REGION Network 35 (SCL): OPENVALVE
   IF "MODE SELECTION DB"."MODE BUFF" <> 0 AND "TRANSFER DB".BUFF."PREMIXING TO MFG WITH INLINE FILTER PRES" = 2
       AND NOT "TRANSFER DB".PAUSE."PREMIXING TO MFG WITH INLINE FILTER PRES" 
       AND "CONTINUE DB"."PREMIXING PROCESS ERROR" = 0 AND "LEVEL BUFF"."PREMIXING_LOAD CELL" = 0 THEN
       "TRANSFER DB".BIT."PREMIXING TO MFG WITH INLINE FILTER PRES"."PFBV-17 TANK OUTLET VALVE" := TRUE;
       "TRANSFER DB".BIT."PREMIXING TO MFG WITH INLINE FILTER PRES"."PBV-93 TANK OUTLET TO INLINE HOMOGENIZER LINE" := TRUE;
       "TRANSFER DB".BIT."PREMIXING TO MFG WITH INLINE FILTER PRES"."PBV-95 TANK OUTLET TO FILTER PRESS LINE" := TRUE;
       "TRANSFER DB".BIT."PREMIXING TO MFG WITH INLINE FILTER PRES"."FILTER PRESS MOTOR 2 RUN" := TRUE;
       "TRANSFER DB".BIT."PREMIXING TO MFG WITH INLINE FILTER PRES"."PBV-100 FILTER PRESS INLET" := TRUE;
       "TRANSFER DB".BIT."PREMIXING TO MFG WITH INLINE FILTER PRES"."PBV-97 FILTER PRESS OUTLET" := TRUE;
       "TRANSFER DB".BIT."PREMIXING TO MFG WITH INLINE FILTER PRES"."PBV-98 INLINE HOMOGENIZER TO FILTER PRESS OUTLET LINE" := TRUE;
       "TRANSFER DB".BIT."PREMIXING TO MFG WITH INLINE FILTER PRES"."PBV-91 PREMIX TO MFG TRANSFER LINE" := TRUE;
       "TRANSFER DB".BIT."PREMIXING TO MFG WITH INLINE FILTER PRES"."PBV-102 PREMIX TO MFG TRANSFER (TOP DISH)" := TRUE;

   ELSE
       "TRANSFER DB".BIT."PREMIXING TO MFG WITH INLINE FILTER PRES"."PFBV-17 TANK OUTLET VALVE" := FALSE;
       "TRANSFER DB".BIT."PREMIXING TO MFG WITH INLINE FILTER PRES"."PBV-93 TANK OUTLET TO INLINE HOMOGENIZER LINE" := FALSE;
       "TRANSFER DB".BIT."PREMIXING TO MFG WITH INLINE FILTER PRES"."PBV-95 TANK OUTLET TO FILTER PRESS LINE" := FALSE;
       "TRANSFER DB".BIT."PREMIXING TO MFG WITH INLINE FILTER PRES"."FILTER PRESS MOTOR 2 RUN" := FALSE;
       "TRANSFER DB".BIT."PREMIXING TO MFG WITH INLINE FILTER PRES"."PBV-100 FILTER PRESS INLET" := FALSE;
       "TRANSFER DB".BIT."PREMIXING TO MFG WITH INLINE FILTER PRES"."PBV-97 FILTER PRESS OUTLET" := FALSE;
       "TRANSFER DB".BIT."PREMIXING TO MFG WITH INLINE FILTER PRES"."PBV-98 INLINE HOMOGENIZER TO FILTER PRESS OUTLET LINE" := FALSE;
       "TRANSFER DB".BIT."PREMIXING TO MFG WITH INLINE FILTER PRES"."PBV-91 PREMIX TO MFG TRANSFER LINE" := FALSE;
       "TRANSFER DB".BIT."PREMIXING TO MFG WITH INLINE FILTER PRES"."PBV-102 PREMIX TO MFG TRANSFER (TOP DISH)" := FALSE;
       ;
   END_IF;
END_REGION

REGION Network 36: LOAD CELL_CUTOFF
   RUNG wire#powerrail
      { S7_Templates := "SrcType := Int" } NE_Contact(in1 := "MODE SELECTION DB"."MODE BUFF", in2 := 0)
      { S7_Templates := "SrcType := Int" } EQ_Contact(in1 := "TRANSFER DB".BUFF."PREMIXING TO MFG WITH INLINE FILTER PRES", in2 := 2)
      I_Contact( "TRANSFER DB".PAUSE."PREMIXING TO MFG WITH INLINE FILTER PRES" )
      { S7_Templates := "SrcType := Int" } NE_Contact(in1 := "CONTINUE DB"."PREMIXING PROCESS ERROR", in2 := 1)
      { S7_Templates := "SrcType := Int" } EQ_Contact(in1 := "LEVEL BUFF"."PREMIXING_LOAD CELL", in2 := 1)
      Move(in := 3, out1 => "TRANSFER DB".BUFF."PREMIXING TO MFG WITH INLINE FILTER PRES")
   END_RUNG
   // the same network as SCL:
   IF ("MODE SELECTION DB"."MODE BUFF" <> 0) AND ("TRANSFER DB".BUFF."PREMIXING TO MFG WITH INLINE FILTER PRES" = 2) AND NOT "TRANSFER DB".PAUSE."PREMIXING TO MFG WITH INLINE FILTER PRES" AND ("CONTINUE DB"."PREMIXING PROCESS ERROR" <> 1) AND ("LEVEL BUFF"."PREMIXING_LOAD CELL" = 1) THEN
       "TRANSFER DB".BUFF."PREMIXING TO MFG WITH INLINE FILTER PRES" := 3;
   END_IF;
END_REGION

REGION Network 37: PROCESS OVER & STOP
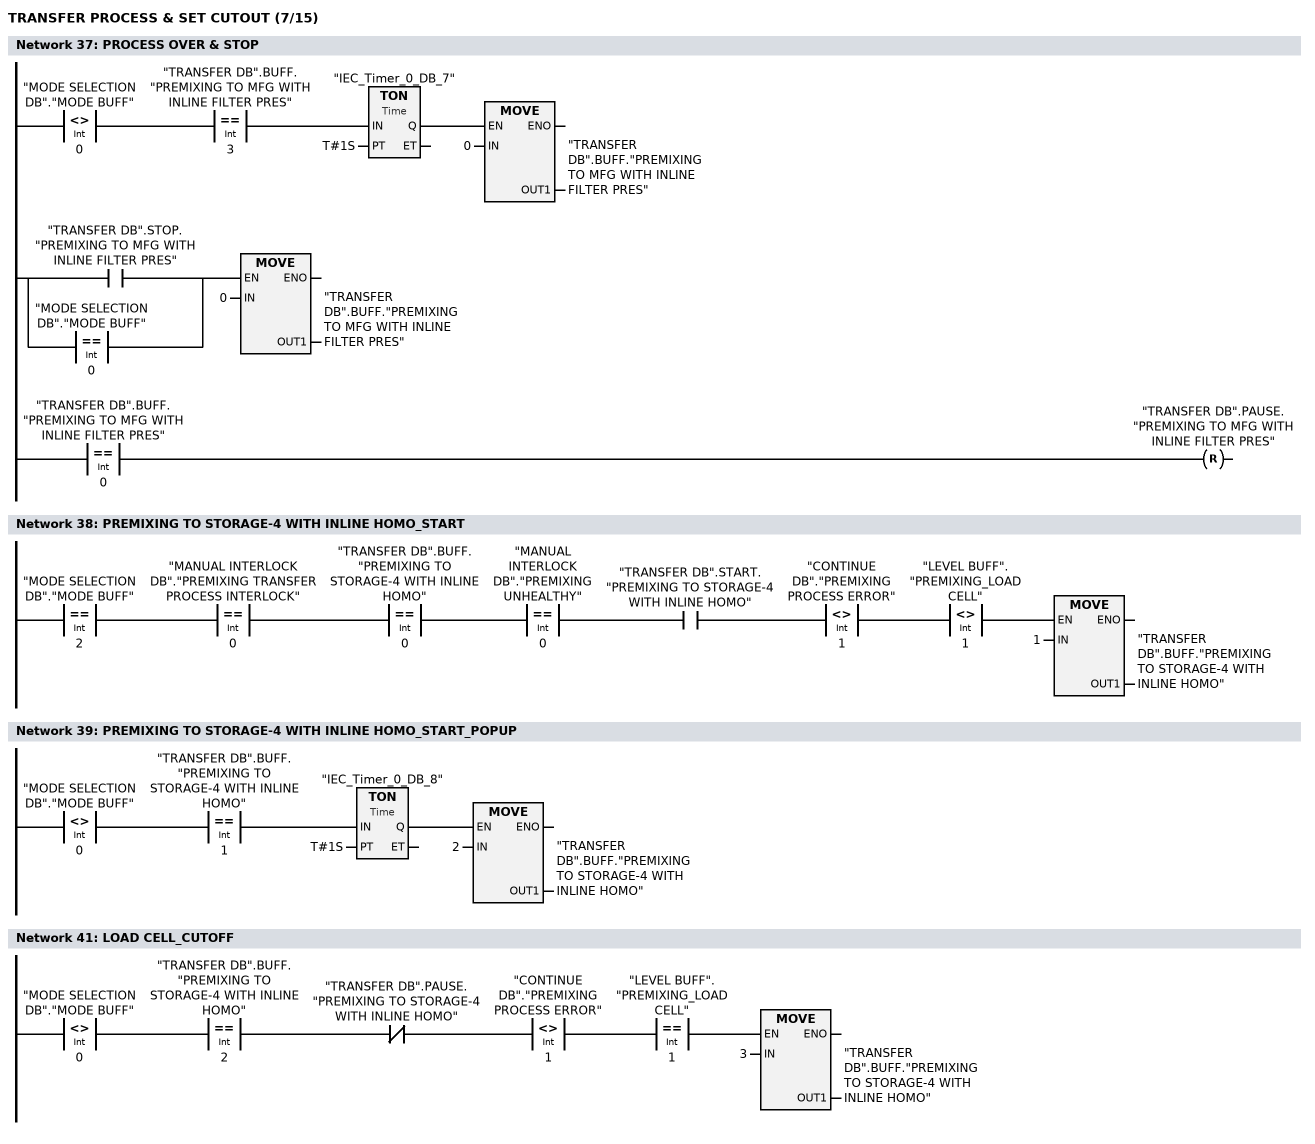
   RUNG wire#powerrail
      { S7_Templates := "SrcType := Int" } NE_Contact(in1 := "MODE SELECTION DB"."MODE BUFF", in2 := 0)
      { S7_Templates := "SrcType := Int" } EQ_Contact(in1 := "TRANSFER DB".BUFF."PREMIXING TO MFG WITH INLINE FILTER PRES", in2 := 3)
      { S7_Templates := "time_type := Time" } "IEC_Timer_0_DB_7".TON(pt := T#1S, et =>)
      Move(in := 0, out1 => "TRANSFER DB".BUFF."PREMIXING TO MFG WITH INLINE FILTER PRES")
   END_RUNG
   RUNG wire#powerrail
      Contact( "TRANSFER DB".STOP."PREMIXING TO MFG WITH INLINE FILTER PRES" )
      wire#w1
      Move(in := 0, out1 => "TRANSFER DB".BUFF."PREMIXING TO MFG WITH INLINE FILTER PRES")
   END_RUNG
   RUNG wire#powerrail
      { S7_Templates := "SrcType := Int" } EQ_Contact(in1 := "MODE SELECTION DB"."MODE BUFF", in2 := 0)
   END_RUNG wire#w1
   RUNG wire#powerrail
      { S7_Templates := "SrcType := Int" } EQ_Contact(in1 := "TRANSFER DB".BUFF."PREMIXING TO MFG WITH INLINE FILTER PRES", in2 := 0)
      R_Coil( "TRANSFER DB".PAUSE."PREMIXING TO MFG WITH INLINE FILTER PRES" )
   END_RUNG
   // the same network as SCL:
   "IEC_Timer_0_DB_7".TON(IN := ("MODE SELECTION DB"."MODE BUFF" <> 0) AND ("TRANSFER DB".BUFF."PREMIXING TO MFG WITH INLINE FILTER PRES" = 3),
                          PT := T#1S);
   IF "IEC_Timer_0_DB_7".Q THEN "TRANSFER DB".BUFF."PREMIXING TO MFG WITH INLINE FILTER PRES" := 0; END_IF;
   IF "TRANSFER DB".STOP."PREMIXING TO MFG WITH INLINE FILTER PRES" OR ("MODE SELECTION DB"."MODE BUFF" = 0) THEN
       "TRANSFER DB".BUFF."PREMIXING TO MFG WITH INLINE FILTER PRES" := 0;
   END_IF;
   IF "TRANSFER DB".BUFF."PREMIXING TO MFG WITH INLINE FILTER PRES" = 0 THEN
       "TRANSFER DB".PAUSE."PREMIXING TO MFG WITH INLINE FILTER PRES" := FALSE;
   END_IF;
END_REGION

REGION Network 38: PREMIXING TO STORAGE-4 WITH INLINE HOMO_START
   RUNG wire#powerrail
      { S7_Templates := "SrcType := Int" } EQ_Contact(in1 := "MODE SELECTION DB"."MODE BUFF", in2 := 2)
      { S7_Templates := "SrcType := Int" } EQ_Contact(in1 := "MANUAL INTERLOCK DB"."PREMIXING TRANSFER PROCESS INTERLOCK", in2 := 0)
      { S7_Templates := "SrcType := Int" } EQ_Contact(in1 := "TRANSFER DB".BUFF."PREMIXING TO STORAGE-4 WITH INLINE HOMO", in2 := 0)
      { S7_Templates := "SrcType := Int" } EQ_Contact(in1 := "MANUAL INTERLOCK DB"."PREMIXING UNHEALTHY", in2 := 0)
      Contact( "TRANSFER DB".START."PREMIXING TO STORAGE-4 WITH INLINE HOMO" )
      { S7_Templates := "SrcType := Int" } NE_Contact(in1 := "CONTINUE DB"."PREMIXING PROCESS ERROR", in2 := 1)
      { S7_Templates := "SrcType := Int" } NE_Contact(in1 := "LEVEL BUFF"."PREMIXING_LOAD CELL", in2 := 1)
      Move(in := 1, out1 => "TRANSFER DB".BUFF."PREMIXING TO STORAGE-4 WITH INLINE HOMO")
   END_RUNG
   // the same network as SCL:
   IF ("MODE SELECTION DB"."MODE BUFF" = 2) AND ("MANUAL INTERLOCK DB"."PREMIXING TRANSFER PROCESS INTERLOCK" = 0) AND ("TRANSFER DB".BUFF."PREMIXING TO STORAGE-4 WITH INLINE HOMO" = 0) AND ("MANUAL INTERLOCK DB"."PREMIXING UNHEALTHY" = 0) AND "TRANSFER DB".START."PREMIXING TO STORAGE-4 WITH INLINE HOMO" AND ("CONTINUE DB"."PREMIXING PROCESS ERROR" <> 1) AND ("LEVEL BUFF"."PREMIXING_LOAD CELL" <> 1) THEN
       "TRANSFER DB".BUFF."PREMIXING TO STORAGE-4 WITH INLINE HOMO" := 1;
   END_IF;
END_REGION

REGION Network 39: PREMIXING TO STORAGE-4 WITH INLINE HOMO_START_POPUP
   RUNG wire#powerrail
      { S7_Templates := "SrcType := Int" } NE_Contact(in1 := "MODE SELECTION DB"."MODE BUFF", in2 := 0)
      { S7_Templates := "SrcType := Int" } EQ_Contact(in1 := "TRANSFER DB".BUFF."PREMIXING TO STORAGE-4 WITH INLINE HOMO", in2 := 1)
      { S7_Templates := "time_type := Time" } "IEC_Timer_0_DB_8".TON(pt := T#1S, et =>)
      Move(in := 2, out1 => "TRANSFER DB".BUFF."PREMIXING TO STORAGE-4 WITH INLINE HOMO")
   END_RUNG
   // the same network as SCL:
   "IEC_Timer_0_DB_8".TON(IN := ("MODE SELECTION DB"."MODE BUFF" <> 0) AND ("TRANSFER DB".BUFF."PREMIXING TO STORAGE-4 WITH INLINE HOMO" = 1),
                          PT := T#1S);
   IF "IEC_Timer_0_DB_8".Q THEN "TRANSFER DB".BUFF."PREMIXING TO STORAGE-4 WITH INLINE HOMO" := 2; END_IF;
END_REGION

REGION Network 40 (SCL): OPENVALVE
   IF "MODE SELECTION DB"."MODE BUFF" <> 0 AND "TRANSFER DB".BUFF."PREMIXING TO STORAGE-4 WITH INLINE HOMO" = 2
       AND NOT "TRANSFER DB".PAUSE."PREMIXING TO STORAGE-4 WITH INLINE HOMO"
       AND "CONTINUE DB"."PREMIXING PROCESS ERROR" = 0 AND "LEVEL BUFF"."PREMIXING_LOAD CELL" = 0 THEN
       "TRANSFER DB".BIT."PREMIXING TO STORAGE-4 WITH INLINE HOMO"."PFBV-17 TANK OUTLET VALVE" := TRUE;
       "TRANSFER DB".BIT."PREMIXING TO STORAGE-4 WITH INLINE HOMO"."PBV-93 TANK OUTLET TO INLINE HOMOGENIZER LINE" := TRUE;
       "TRANSFER DB".BIT."PREMIXING TO STORAGE-4 WITH INLINE HOMO"."PBV-94 INLINE HOMOGENIZER INLET LINE" := TRUE;
       "TRANSFER DB".BIT."PREMIXING TO STORAGE-4 WITH INLINE HOMO"."INLINE 2 HOMOGENIZER MOTOR 2 RUN" := TRUE;
       "TRANSFER DB".BIT."PREMIXING TO STORAGE-4 WITH INLINE HOMO"."PBV-96 INLINE HOMOGENIZER RECIRCULATION LINE" := TRUE;
       "TRANSFER DB".BIT."PREMIXING TO STORAGE-4 WITH INLINE HOMO"."PBV-92 PREMIX TO STORAGE – 4 TRANSFER LINE" := TRUE;

   ELSE
       "TRANSFER DB".BIT."PREMIXING TO STORAGE-4 WITH INLINE HOMO"."PFBV-17 TANK OUTLET VALVE" := FALSE;
       "TRANSFER DB".BIT."PREMIXING TO STORAGE-4 WITH INLINE HOMO"."PBV-93 TANK OUTLET TO INLINE HOMOGENIZER LINE" := FALSE;
       "TRANSFER DB".BIT."PREMIXING TO STORAGE-4 WITH INLINE HOMO"."PBV-94 INLINE HOMOGENIZER INLET LINE" := FALSE;
       "TRANSFER DB".BIT."PREMIXING TO STORAGE-4 WITH INLINE HOMO"."INLINE 2 HOMOGENIZER MOTOR 2 RUN" := FALSE;
       "TRANSFER DB".BIT."PREMIXING TO STORAGE-4 WITH INLINE HOMO"."PBV-96 INLINE HOMOGENIZER RECIRCULATION LINE" := FALSE;
       "TRANSFER DB".BIT."PREMIXING TO STORAGE-4 WITH INLINE HOMO"."PBV-92 PREMIX TO STORAGE – 4 TRANSFER LINE" := FALSE;
       ;
   END_IF;
END_REGION

REGION Network 41: LOAD CELL_CUTOFF
   RUNG wire#powerrail
      { S7_Templates := "SrcType := Int" } NE_Contact(in1 := "MODE SELECTION DB"."MODE BUFF", in2 := 0)
      { S7_Templates := "SrcType := Int" } EQ_Contact(in1 := "TRANSFER DB".BUFF."PREMIXING TO STORAGE-4 WITH INLINE HOMO", in2 := 2)
      I_Contact( "TRANSFER DB".PAUSE."PREMIXING TO STORAGE-4 WITH INLINE HOMO" )
      { S7_Templates := "SrcType := Int" } NE_Contact(in1 := "CONTINUE DB"."PREMIXING PROCESS ERROR", in2 := 1)
      { S7_Templates := "SrcType := Int" } EQ_Contact(in1 := "LEVEL BUFF"."PREMIXING_LOAD CELL", in2 := 1)
      Move(in := 3, out1 => "TRANSFER DB".BUFF."PREMIXING TO STORAGE-4 WITH INLINE HOMO")
   END_RUNG
   // the same network as SCL:
   IF ("MODE SELECTION DB"."MODE BUFF" <> 0) AND ("TRANSFER DB".BUFF."PREMIXING TO STORAGE-4 WITH INLINE HOMO" = 2) AND NOT "TRANSFER DB".PAUSE."PREMIXING TO STORAGE-4 WITH INLINE HOMO" AND ("CONTINUE DB"."PREMIXING PROCESS ERROR" <> 1) AND ("LEVEL BUFF"."PREMIXING_LOAD CELL" = 1) THEN
       "TRANSFER DB".BUFF."PREMIXING TO STORAGE-4 WITH INLINE HOMO" := 3;
   END_IF;
END_REGION

REGION Network 42: PROCESS OVER & STOP
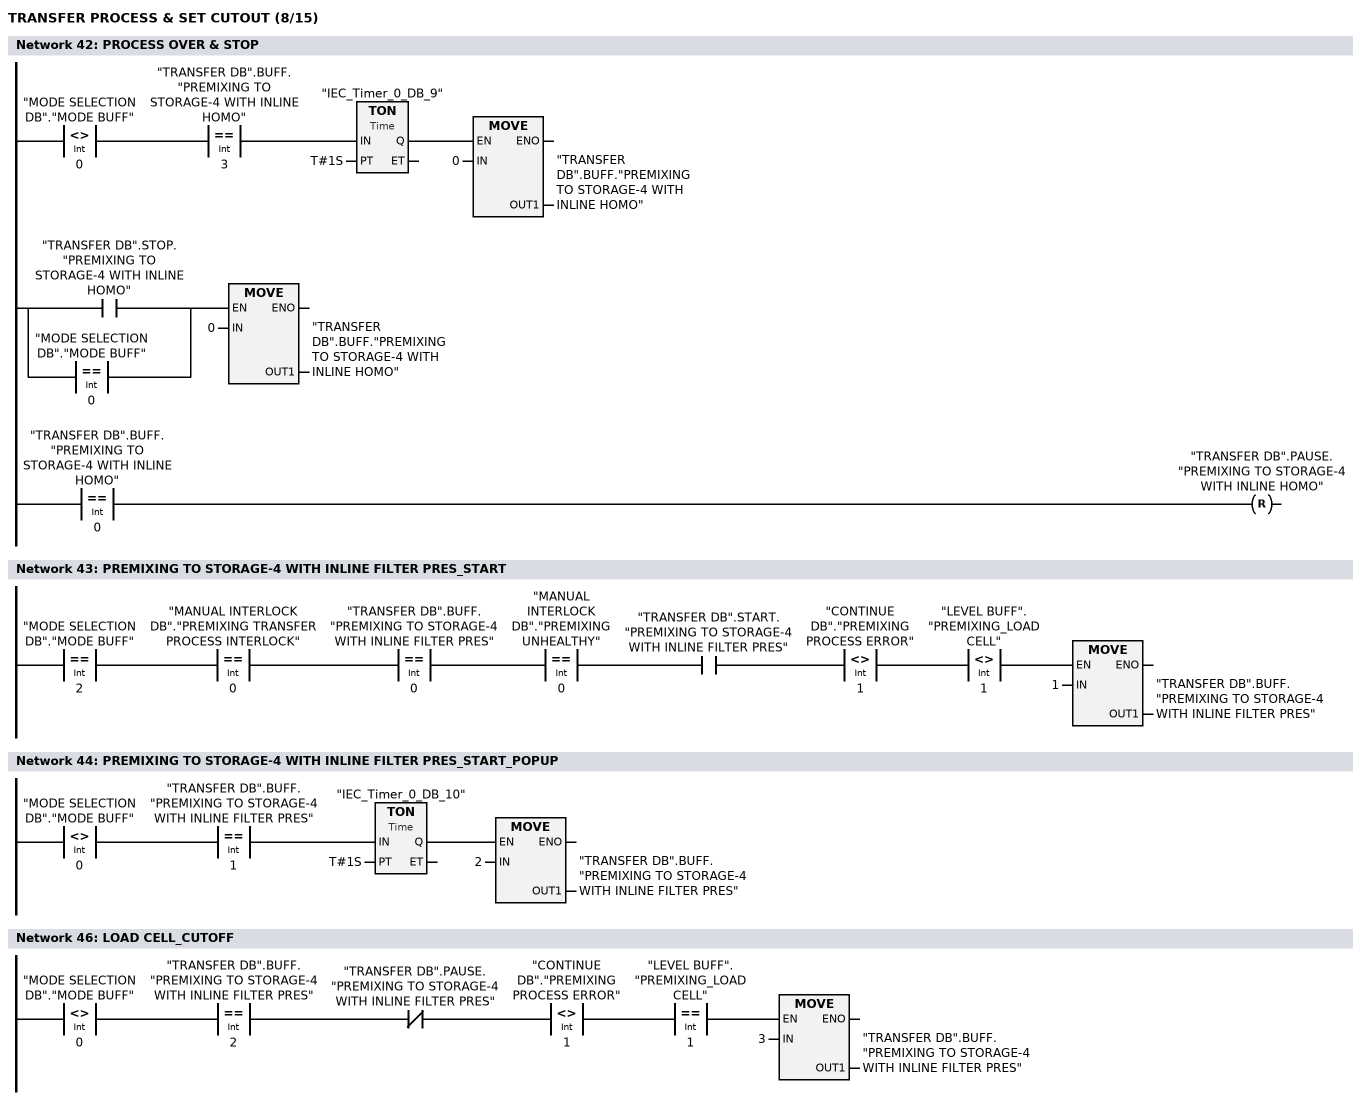
   RUNG wire#powerrail
      { S7_Templates := "SrcType := Int" } NE_Contact(in1 := "MODE SELECTION DB"."MODE BUFF", in2 := 0)
      { S7_Templates := "SrcType := Int" } EQ_Contact(in1 := "TRANSFER DB".BUFF."PREMIXING TO STORAGE-4 WITH INLINE HOMO", in2 := 3)
      { S7_Templates := "time_type := Time" } "IEC_Timer_0_DB_9".TON(pt := T#1S, et =>)
      Move(in := 0, out1 => "TRANSFER DB".BUFF."PREMIXING TO STORAGE-4 WITH INLINE HOMO")
   END_RUNG
   RUNG wire#powerrail
      Contact( "TRANSFER DB".STOP."PREMIXING TO STORAGE-4 WITH INLINE HOMO" )
      wire#w1
      Move(in := 0, out1 => "TRANSFER DB".BUFF."PREMIXING TO STORAGE-4 WITH INLINE HOMO")
   END_RUNG
   RUNG wire#powerrail
      { S7_Templates := "SrcType := Int" } EQ_Contact(in1 := "MODE SELECTION DB"."MODE BUFF", in2 := 0)
   END_RUNG wire#w1
   RUNG wire#powerrail
      { S7_Templates := "SrcType := Int" } EQ_Contact(in1 := "TRANSFER DB".BUFF."PREMIXING TO STORAGE-4 WITH INLINE HOMO", in2 := 0)
      R_Coil( "TRANSFER DB".PAUSE."PREMIXING TO STORAGE-4 WITH INLINE HOMO" )
   END_RUNG
   // the same network as SCL:
   "IEC_Timer_0_DB_9".TON(IN := ("MODE SELECTION DB"."MODE BUFF" <> 0) AND ("TRANSFER DB".BUFF."PREMIXING TO STORAGE-4 WITH INLINE HOMO" = 3),
                          PT := T#1S);
   IF "IEC_Timer_0_DB_9".Q THEN "TRANSFER DB".BUFF."PREMIXING TO STORAGE-4 WITH INLINE HOMO" := 0; END_IF;
   IF "TRANSFER DB".STOP."PREMIXING TO STORAGE-4 WITH INLINE HOMO" OR ("MODE SELECTION DB"."MODE BUFF" = 0) THEN
       "TRANSFER DB".BUFF."PREMIXING TO STORAGE-4 WITH INLINE HOMO" := 0;
   END_IF;
   IF "TRANSFER DB".BUFF."PREMIXING TO STORAGE-4 WITH INLINE HOMO" = 0 THEN
       "TRANSFER DB".PAUSE."PREMIXING TO STORAGE-4 WITH INLINE HOMO" := FALSE;
   END_IF;
END_REGION

REGION Network 43: PREMIXING TO STORAGE-4 WITH INLINE FILTER PRES_START
   RUNG wire#powerrail
      { S7_Templates := "SrcType := Int" } EQ_Contact(in1 := "MODE SELECTION DB"."MODE BUFF", in2 := 2)
      { S7_Templates := "SrcType := Int" } EQ_Contact(in1 := "MANUAL INTERLOCK DB"."PREMIXING TRANSFER PROCESS INTERLOCK", in2 := 0)
      { S7_Templates := "SrcType := Int" } EQ_Contact(in1 := "TRANSFER DB".BUFF."PREMIXING TO STORAGE-4 WITH INLINE FILTER PRES", in2 := 0)
      { S7_Templates := "SrcType := Int" } EQ_Contact(in1 := "MANUAL INTERLOCK DB"."PREMIXING UNHEALTHY", in2 := 0)
      Contact( "TRANSFER DB".START."PREMIXING TO STORAGE-4 WITH INLINE FILTER PRES" )
      { S7_Templates := "SrcType := Int" } NE_Contact(in1 := "CONTINUE DB"."PREMIXING PROCESS ERROR", in2 := 1)
      { S7_Templates := "SrcType := Int" } NE_Contact(in1 := "LEVEL BUFF"."PREMIXING_LOAD CELL", in2 := 1)
      Move(in := 1, out1 => "TRANSFER DB".BUFF."PREMIXING TO STORAGE-4 WITH INLINE FILTER PRES")
   END_RUNG
   // the same network as SCL:
   IF ("MODE SELECTION DB"."MODE BUFF" = 2) AND ("MANUAL INTERLOCK DB"."PREMIXING TRANSFER PROCESS INTERLOCK" = 0) AND ("TRANSFER DB".BUFF."PREMIXING TO STORAGE-4 WITH INLINE FILTER PRES" = 0) AND ("MANUAL INTERLOCK DB"."PREMIXING UNHEALTHY" = 0) AND "TRANSFER DB".START."PREMIXING TO STORAGE-4 WITH INLINE FILTER PRES" AND ("CONTINUE DB"."PREMIXING PROCESS ERROR" <> 1) AND ("LEVEL BUFF"."PREMIXING_LOAD CELL" <> 1) THEN
       "TRANSFER DB".BUFF."PREMIXING TO STORAGE-4 WITH INLINE FILTER PRES" := 1;
   END_IF;
END_REGION

REGION Network 44: PREMIXING TO STORAGE-4 WITH INLINE FILTER PRES_START_POPUP
   RUNG wire#powerrail
      { S7_Templates := "SrcType := Int" } NE_Contact(in1 := "MODE SELECTION DB"."MODE BUFF", in2 := 0)
      { S7_Templates := "SrcType := Int" } EQ_Contact(in1 := "TRANSFER DB".BUFF."PREMIXING TO STORAGE-4 WITH INLINE FILTER PRES", in2 := 1)
      { S7_Templates := "time_type := Time" } "IEC_Timer_0_DB_10".TON(pt := T#1S, et =>)
      Move(in := 2, out1 => "TRANSFER DB".BUFF."PREMIXING TO STORAGE-4 WITH INLINE FILTER PRES")
   END_RUNG
   // the same network as SCL:
   "IEC_Timer_0_DB_10".TON(IN := ("MODE SELECTION DB"."MODE BUFF" <> 0) AND ("TRANSFER DB".BUFF."PREMIXING TO STORAGE-4 WITH INLINE FILTER PRES" = 1),
                           PT := T#1S);
   IF "IEC_Timer_0_DB_10".Q THEN
       "TRANSFER DB".BUFF."PREMIXING TO STORAGE-4 WITH INLINE FILTER PRES" := 2;
   END_IF;
END_REGION

REGION Network 45 (SCL): OPENVALVE
   IF "MODE SELECTION DB"."MODE BUFF" <> 0 AND "TRANSFER DB".BUFF."PREMIXING TO STORAGE-4 WITH INLINE FILTER PRES" = 2
       AND NOT "TRANSFER DB".PAUSE."PREMIXING TO STORAGE-4 WITH INLINE FILTER PRES" 
       AND "CONTINUE DB"."PREMIXING PROCESS ERROR" = 0 AND "LEVEL BUFF"."PREMIXING_LOAD CELL" = 0 THEN
       "TRANSFER DB".BIT."PREMIXING TO STORAGE-4 WITH INLINE FILTER PRES"."PFBV-17 TANK OUTLET VALVE" := TRUE;
       "TRANSFER DB".BIT."PREMIXING TO STORAGE-4 WITH INLINE FILTER PRES"."PBV-93 TANK OUTLET TO INLINE HOMOGENIZER LINE" := TRUE;
       "TRANSFER DB".BIT."PREMIXING TO STORAGE-4 WITH INLINE FILTER PRES"."PBV-95 TANK OUTLET TO FILTER PRESS LINE" := TRUE;
       "TRANSFER DB".BIT."PREMIXING TO STORAGE-4 WITH INLINE FILTER PRES"."FILTER PRESS MOTOR 2 RUN" := TRUE;
       "TRANSFER DB".BIT."PREMIXING TO STORAGE-4 WITH INLINE FILTER PRES"."PBV-100 FILTER PRESS INLET" := TRUE;
       "TRANSFER DB".BIT."PREMIXING TO STORAGE-4 WITH INLINE FILTER PRES"."PBV-97 FILTER PRESS OUTLET" := TRUE;
       "TRANSFER DB".BIT."PREMIXING TO STORAGE-4 WITH INLINE FILTER PRES"."PBV-98 INLINE HOMOGENIZER TO FILTER PRESS OUTLET LINE" := TRUE;
       "TRANSFER DB".BIT."PREMIXING TO STORAGE-4 WITH INLINE FILTER PRES"."PBV-92 PREMIX TO STORAGE – 4 TRANSFER LINE" := TRUE;

   ELSE
       "TRANSFER DB".BIT."PREMIXING TO STORAGE-4 WITH INLINE FILTER PRES"."PFBV-17 TANK OUTLET VALVE" := FALSE;
       "TRANSFER DB".BIT."PREMIXING TO STORAGE-4 WITH INLINE FILTER PRES"."PBV-93 TANK OUTLET TO INLINE HOMOGENIZER LINE" := FALSE;
       "TRANSFER DB".BIT."PREMIXING TO STORAGE-4 WITH INLINE FILTER PRES"."PBV-95 TANK OUTLET TO FILTER PRESS LINE" := FALSE;
       "TRANSFER DB".BIT."PREMIXING TO STORAGE-4 WITH INLINE FILTER PRES"."FILTER PRESS MOTOR 2 RUN" := FALSE;
       "TRANSFER DB".BIT."PREMIXING TO STORAGE-4 WITH INLINE FILTER PRES"."PBV-100 FILTER PRESS INLET" := FALSE;
       "TRANSFER DB".BIT."PREMIXING TO STORAGE-4 WITH INLINE FILTER PRES"."PBV-97 FILTER PRESS OUTLET" := FALSE;
       "TRANSFER DB".BIT."PREMIXING TO STORAGE-4 WITH INLINE FILTER PRES"."PBV-98 INLINE HOMOGENIZER TO FILTER PRESS OUTLET LINE" := FALSE;
       "TRANSFER DB".BIT."PREMIXING TO STORAGE-4 WITH INLINE FILTER PRES"."PBV-92 PREMIX TO STORAGE – 4 TRANSFER LINE" := FALSE;
       ;
   END_IF;
END_REGION

REGION Network 46: LOAD CELL_CUTOFF
   RUNG wire#powerrail
      { S7_Templates := "SrcType := Int" } NE_Contact(in1 := "MODE SELECTION DB"."MODE BUFF", in2 := 0)
      { S7_Templates := "SrcType := Int" } EQ_Contact(in1 := "TRANSFER DB".BUFF."PREMIXING TO STORAGE-4 WITH INLINE FILTER PRES", in2 := 2)
      I_Contact( "TRANSFER DB".PAUSE."PREMIXING TO STORAGE-4 WITH INLINE FILTER PRES" )
      { S7_Templates := "SrcType := Int" } NE_Contact(in1 := "CONTINUE DB"."PREMIXING PROCESS ERROR", in2 := 1)
      { S7_Templates := "SrcType := Int" } EQ_Contact(in1 := "LEVEL BUFF"."PREMIXING_LOAD CELL", in2 := 1)
      Move(in := 3, out1 => "TRANSFER DB".BUFF."PREMIXING TO STORAGE-4 WITH INLINE FILTER PRES")
   END_RUNG
   // the same network as SCL:
   IF ("MODE SELECTION DB"."MODE BUFF" <> 0) AND ("TRANSFER DB".BUFF."PREMIXING TO STORAGE-4 WITH INLINE FILTER PRES" = 2) AND NOT "TRANSFER DB".PAUSE."PREMIXING TO STORAGE-4 WITH INLINE FILTER PRES" AND ("CONTINUE DB"."PREMIXING PROCESS ERROR" <> 1) AND ("LEVEL BUFF"."PREMIXING_LOAD CELL" = 1) THEN
       "TRANSFER DB".BUFF."PREMIXING TO STORAGE-4 WITH INLINE FILTER PRES" := 3;
   END_IF;
END_REGION

REGION Network 47: PROCESS OVER & STOP
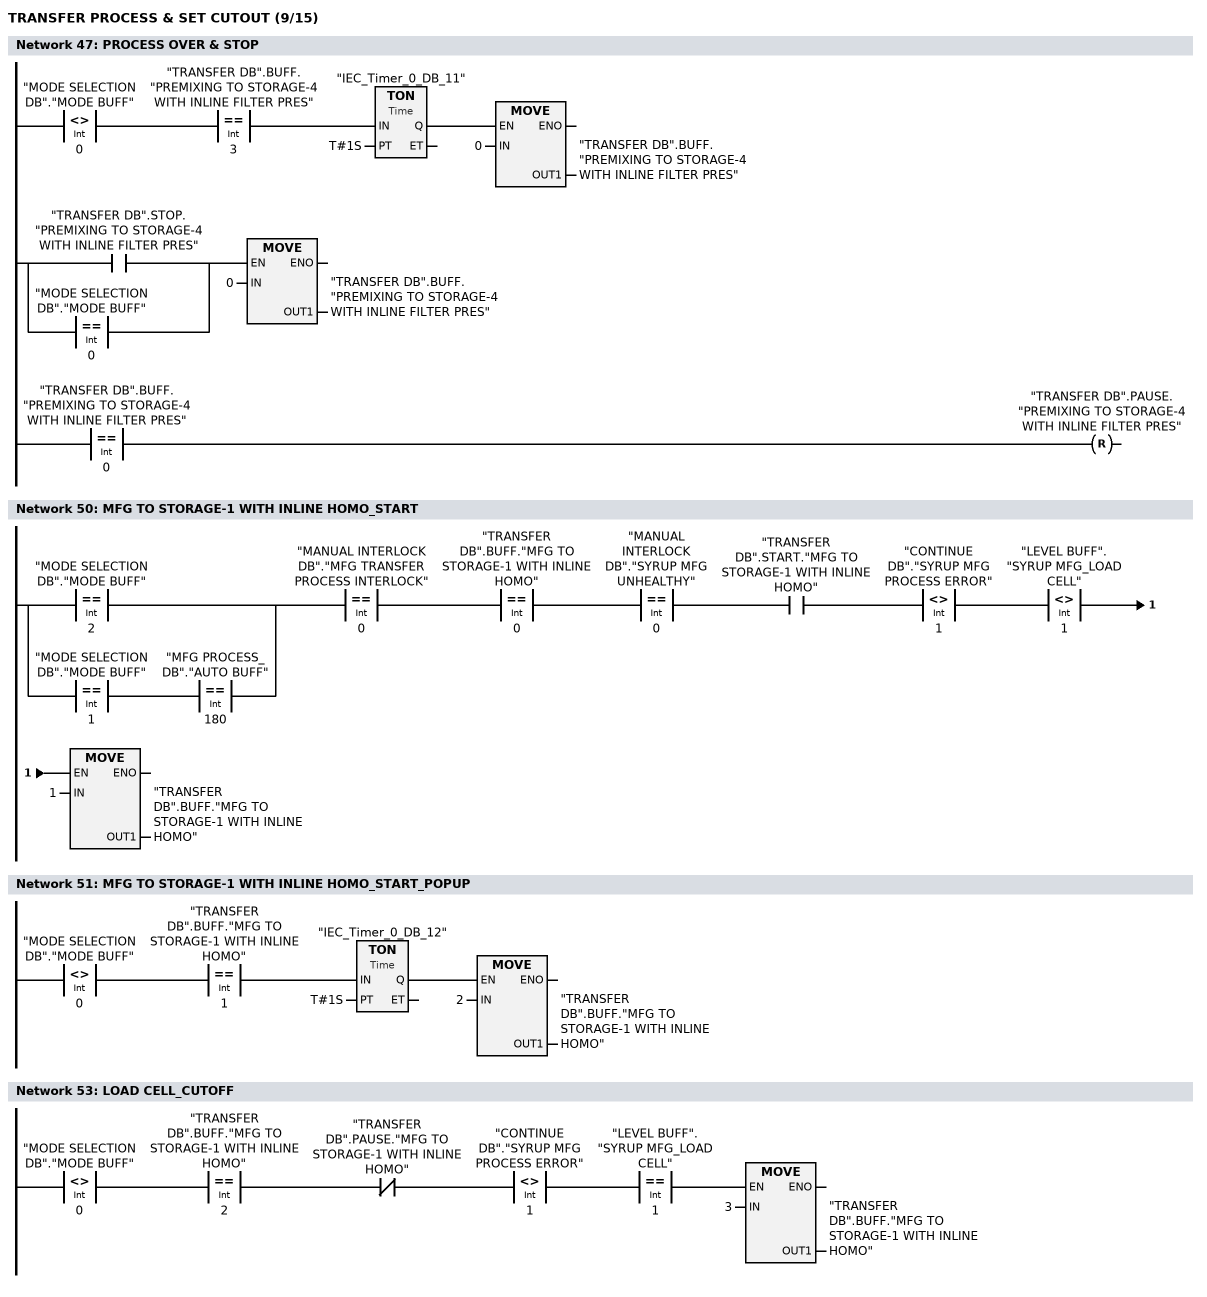
   RUNG wire#powerrail
      { S7_Templates := "SrcType := Int" } NE_Contact(in1 := "MODE SELECTION DB"."MODE BUFF", in2 := 0)
      { S7_Templates := "SrcType := Int" } EQ_Contact(in1 := "TRANSFER DB".BUFF."PREMIXING TO STORAGE-4 WITH INLINE FILTER PRES", in2 := 3)
      { S7_Templates := "time_type := Time" } "IEC_Timer_0_DB_11".TON(pt := T#1S, et =>)
      Move(in := 0, out1 => "TRANSFER DB".BUFF."PREMIXING TO STORAGE-4 WITH INLINE FILTER PRES")
   END_RUNG
   RUNG wire#powerrail
      Contact( "TRANSFER DB".STOP."PREMIXING TO STORAGE-4 WITH INLINE FILTER PRES" )
      wire#w1
      Move(in := 0, out1 => "TRANSFER DB".BUFF."PREMIXING TO STORAGE-4 WITH INLINE FILTER PRES")
   END_RUNG
   RUNG wire#powerrail
      { S7_Templates := "SrcType := Int" } EQ_Contact(in1 := "MODE SELECTION DB"."MODE BUFF", in2 := 0)
   END_RUNG wire#w1
   RUNG wire#powerrail
      { S7_Templates := "SrcType := Int" } EQ_Contact(in1 := "TRANSFER DB".BUFF."PREMIXING TO STORAGE-4 WITH INLINE FILTER PRES", in2 := 0)
      R_Coil( "TRANSFER DB".PAUSE."PREMIXING TO STORAGE-4 WITH INLINE FILTER PRES" )
   END_RUNG
   // the same network as SCL:
   "IEC_Timer_0_DB_11".TON(IN := ("MODE SELECTION DB"."MODE BUFF" <> 0) AND ("TRANSFER DB".BUFF."PREMIXING TO STORAGE-4 WITH INLINE FILTER PRES" = 3),
                           PT := T#1S);
   IF "IEC_Timer_0_DB_11".Q THEN
       "TRANSFER DB".BUFF."PREMIXING TO STORAGE-4 WITH INLINE FILTER PRES" := 0;
   END_IF;
   IF "TRANSFER DB".STOP."PREMIXING TO STORAGE-4 WITH INLINE FILTER PRES" OR ("MODE SELECTION DB"."MODE BUFF" = 0) THEN
       "TRANSFER DB".BUFF."PREMIXING TO STORAGE-4 WITH INLINE FILTER PRES" := 0;
   END_IF;
   IF "TRANSFER DB".BUFF."PREMIXING TO STORAGE-4 WITH INLINE FILTER PRES" = 0 THEN
       "TRANSFER DB".PAUSE."PREMIXING TO STORAGE-4 WITH INLINE FILTER PRES" := FALSE;
   END_IF;
END_REGION

REGION Network 49: ////////////////////////////////////////////////////////////////////// TRANSFER PROCESS- MFG //////////////////////////////////////////////////////////////////////////////////
END_REGION

REGION Network 50: MFG TO STORAGE-1 WITH INLINE HOMO_START
   RUNG wire#powerrail
      { S7_Templates := "SrcType := Int" } EQ_Contact(in1 := "MODE SELECTION DB"."MODE BUFF", in2 := 2)
      wire#w1
      { S7_Templates := "SrcType := Int" } EQ_Contact(in1 := "MANUAL INTERLOCK DB"."MFG TRANSFER PROCESS INTERLOCK", in2 := 0)
      { S7_Templates := "SrcType := Int" } EQ_Contact(in1 := "TRANSFER DB".BUFF."MFG TO STORAGE-1 WITH INLINE HOMO", in2 := 0)
      { S7_Templates := "SrcType := Int" } EQ_Contact(in1 := "MANUAL INTERLOCK DB"."SYRUP MFG UNHEALTHY", in2 := 0)
      Contact( "TRANSFER DB".START."MFG TO STORAGE-1 WITH INLINE HOMO" )
      { S7_Templates := "SrcType := Int" } NE_Contact(in1 := "CONTINUE DB"."SYRUP MFG PROCESS ERROR", in2 := 1)
      { S7_Templates := "SrcType := Int" } NE_Contact(in1 := "LEVEL BUFF"."SYRUP MFG_LOAD CELL", in2 := 1)
      Move(in := 1, out1 => "TRANSFER DB".BUFF."MFG TO STORAGE-1 WITH INLINE HOMO")
   END_RUNG
   RUNG wire#powerrail
      { S7_Templates := "SrcType := Int" } EQ_Contact(in1 := "MODE SELECTION DB"."MODE BUFF", in2 := 1)
      { S7_Templates := "SrcType := Int" } EQ_Contact(in1 := "MFG PROCESS_DB"."AUTO BUFF", in2 := 180)
   END_RUNG wire#w1
   // the same network as SCL:
   IF (("MODE SELECTION DB"."MODE BUFF" = 2) OR (("MODE SELECTION DB"."MODE BUFF" = 1) AND ("MFG PROCESS_DB"."AUTO BUFF" = 180))) AND ("MANUAL INTERLOCK DB"."MFG TRANSFER PROCESS INTERLOCK" = 0) AND ("TRANSFER DB".BUFF."MFG TO STORAGE-1 WITH INLINE HOMO" = 0) AND ("MANUAL INTERLOCK DB"."SYRUP MFG UNHEALTHY" = 0) AND "TRANSFER DB".START."MFG TO STORAGE-1 WITH INLINE HOMO" AND ("CONTINUE DB"."SYRUP MFG PROCESS ERROR" <> 1) AND ("LEVEL BUFF"."SYRUP MFG_LOAD CELL" <> 1) THEN
       "TRANSFER DB".BUFF."MFG TO STORAGE-1 WITH INLINE HOMO" := 1;
   END_IF;
END_REGION

REGION Network 51: MFG TO STORAGE-1 WITH INLINE HOMO_START_POPUP
   RUNG wire#powerrail
      { S7_Templates := "SrcType := Int" } NE_Contact(in1 := "MODE SELECTION DB"."MODE BUFF", in2 := 0)
      { S7_Templates := "SrcType := Int" } EQ_Contact(in1 := "TRANSFER DB".BUFF."MFG TO STORAGE-1 WITH INLINE HOMO", in2 := 1)
      { S7_Templates := "time_type := Time" } "IEC_Timer_0_DB_12".TON(pt := T#1S, et =>)
      Move(in := 2, out1 => "TRANSFER DB".BUFF."MFG TO STORAGE-1 WITH INLINE HOMO")
   END_RUNG
   // the same network as SCL:
   "IEC_Timer_0_DB_12".TON(IN := ("MODE SELECTION DB"."MODE BUFF" <> 0) AND ("TRANSFER DB".BUFF."MFG TO STORAGE-1 WITH INLINE HOMO" = 1),
                           PT := T#1S);
   IF "IEC_Timer_0_DB_12".Q THEN "TRANSFER DB".BUFF."MFG TO STORAGE-1 WITH INLINE HOMO" := 2; END_IF;
END_REGION

REGION Network 52 (SCL): OPENVALVE
   IF ("MODE SELECTION DB"."MODE BUFF" <> 0 AND "TRANSFER DB".BUFF."MFG TO STORAGE-1 WITH INLINE HOMO" = 2
       AND NOT "TRANSFER DB".PAUSE."MFG TO STORAGE-1 WITH INLINE HOMO"
       AND "CONTINUE DB"."SYRUP MFG PROCESS ERROR" = 0 AND "LEVEL BUFF"."SYRUP MFG_LOAD CELL" = 0)
       OR ("MODE SELECTION DB"."MODE BUFF"=1 AND "MFG PROCESS_DB"."AUTO BUFF"=0
       AND "MFG TRANSFER CYCLE DB".TRANSFER."TRANSFER BUFF"."MFG TO STORAGE-1 WITH INLINE HOMO"=10 AND "CONTINUE DB"."SYRUP MFG PROCESS ERROR" <>1
       AND "MFG TRANSFER CYCLE DB".TRANSFER.SELECT."SELECT BUFF"=1)
   THEN
       "TRANSFER DB".BIT."MFG TO STORAGE-1 WITH INLINE HOMO"."PFBV-59 TANK OUTLET VALVE" := TRUE;
       "TRANSFER DB".BIT."MFG TO STORAGE-1 WITH INLINE HOMO"."PBV-114 TANK OUTLET TO INLINE HOMOGENIZER LINE" := TRUE;
       "TRANSFER DB".BIT."MFG TO STORAGE-1 WITH INLINE HOMO"."PBV-110 INLINE HOMOGENIZER TO INLET LINE" := TRUE;
       "TRANSFER DB".BIT."MFG TO STORAGE-1 WITH INLINE HOMO"."PAV-56 INLINE HOMO. SEAL COOLING INLET" := TRUE;
       "TRANSFER DB".BIT."MFG TO STORAGE-1 WITH INLINE HOMO"."INLINE 1 HOMOGENIZER MOTOR1 RUN" := TRUE;
       "TRANSFER DB".BIT."MFG TO STORAGE-1 WITH INLINE HOMO"."PBV-109 HOMO. RECIRCULATION INLET" := TRUE;
       "TRANSFER DB".BIT."MFG TO STORAGE-1 WITH INLINE HOMO"."PBV-115 MFG TO STORAGE – 1 TRANSFER LINE" := TRUE;
   ELSE
       "TRANSFER DB".BIT."MFG TO STORAGE-1 WITH INLINE HOMO"."PFBV-59 TANK OUTLET VALVE" := FALSE;
       "TRANSFER DB".BIT."MFG TO STORAGE-1 WITH INLINE HOMO"."PBV-114 TANK OUTLET TO INLINE HOMOGENIZER LINE" := FALSE;
       "TRANSFER DB".BIT."MFG TO STORAGE-1 WITH INLINE HOMO"."PBV-110 INLINE HOMOGENIZER TO INLET LINE" := FALSE;
       "TRANSFER DB".BIT."MFG TO STORAGE-1 WITH INLINE HOMO"."PAV-56 INLINE HOMO. SEAL COOLING INLET" := FALSE;
       "TRANSFER DB".BIT."MFG TO STORAGE-1 WITH INLINE HOMO"."INLINE 1 HOMOGENIZER MOTOR1 RUN" := FALSE;
       "TRANSFER DB".BIT."MFG TO STORAGE-1 WITH INLINE HOMO"."PBV-109 HOMO. RECIRCULATION INLET" := FALSE;
       "TRANSFER DB".BIT."MFG TO STORAGE-1 WITH INLINE HOMO"."PBV-115 MFG TO STORAGE – 1 TRANSFER LINE" := FALSE;
       ;
   END_IF;
END_REGION

REGION Network 53: LOAD CELL_CUTOFF
   RUNG wire#powerrail
      { S7_Templates := "SrcType := Int" } NE_Contact(in1 := "MODE SELECTION DB"."MODE BUFF", in2 := 0)
      { S7_Templates := "SrcType := Int" } EQ_Contact(in1 := "TRANSFER DB".BUFF."MFG TO STORAGE-1 WITH INLINE HOMO", in2 := 2)
      I_Contact( "TRANSFER DB".PAUSE."MFG TO STORAGE-1 WITH INLINE HOMO" )
      { S7_Templates := "SrcType := Int" } NE_Contact(in1 := "CONTINUE DB"."SYRUP MFG PROCESS ERROR", in2 := 1)
      { S7_Templates := "SrcType := Int" } EQ_Contact(in1 := "LEVEL BUFF"."SYRUP MFG_LOAD CELL", in2 := 1)
      Move(in := 3, out1 => "TRANSFER DB".BUFF."MFG TO STORAGE-1 WITH INLINE HOMO")
   END_RUNG
   // the same network as SCL:
   IF ("MODE SELECTION DB"."MODE BUFF" <> 0) AND ("TRANSFER DB".BUFF."MFG TO STORAGE-1 WITH INLINE HOMO" = 2) AND NOT "TRANSFER DB".PAUSE."MFG TO STORAGE-1 WITH INLINE HOMO" AND ("CONTINUE DB"."SYRUP MFG PROCESS ERROR" <> 1) AND ("LEVEL BUFF"."SYRUP MFG_LOAD CELL" = 1) THEN
       "TRANSFER DB".BUFF."MFG TO STORAGE-1 WITH INLINE HOMO" := 3;
   END_IF;
END_REGION

REGION Network 54: PROCESS OVER & STOP
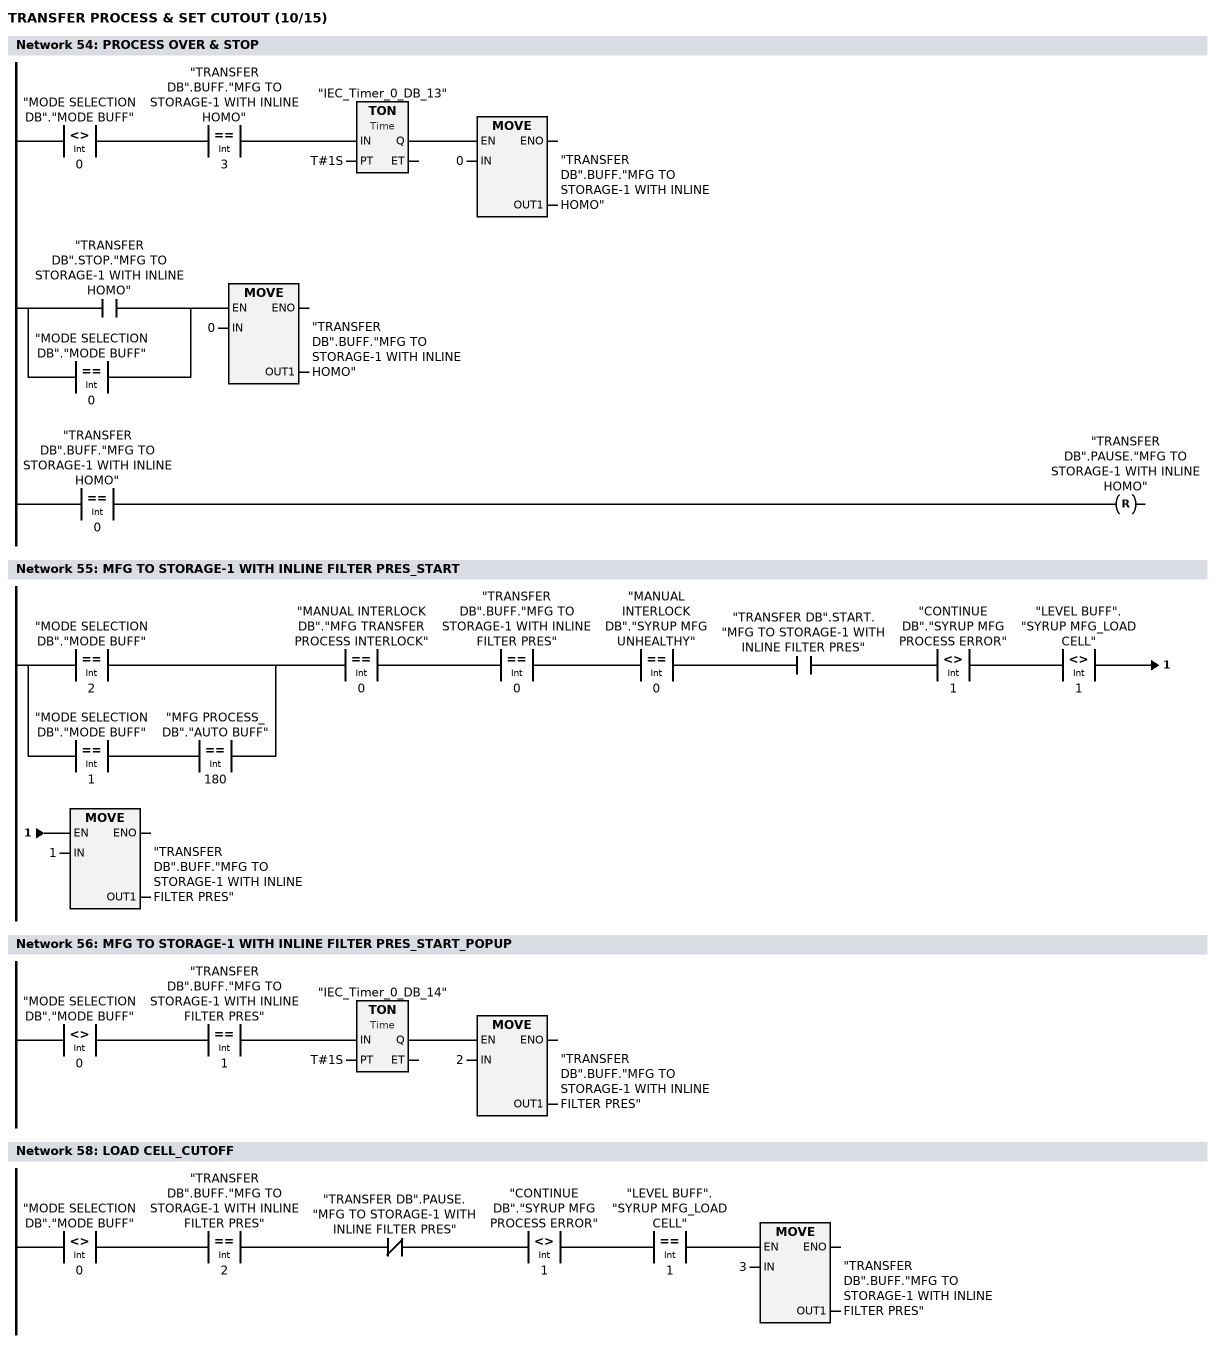
   RUNG wire#powerrail
      { S7_Templates := "SrcType := Int" } NE_Contact(in1 := "MODE SELECTION DB"."MODE BUFF", in2 := 0)
      { S7_Templates := "SrcType := Int" } EQ_Contact(in1 := "TRANSFER DB".BUFF."MFG TO STORAGE-1 WITH INLINE HOMO", in2 := 3)
      { S7_Templates := "time_type := Time" } "IEC_Timer_0_DB_13".TON(pt := T#1S, et =>)
      Move(in := 0, out1 => "TRANSFER DB".BUFF."MFG TO STORAGE-1 WITH INLINE HOMO")
   END_RUNG
   RUNG wire#powerrail
      Contact( "TRANSFER DB".STOP."MFG TO STORAGE-1 WITH INLINE HOMO" )
      wire#w1
      Move(in := 0, out1 => "TRANSFER DB".BUFF."MFG TO STORAGE-1 WITH INLINE HOMO")
   END_RUNG
   RUNG wire#powerrail
      { S7_Templates := "SrcType := Int" } EQ_Contact(in1 := "MODE SELECTION DB"."MODE BUFF", in2 := 0)
   END_RUNG wire#w1
   RUNG wire#powerrail
      { S7_Templates := "SrcType := Int" } EQ_Contact(in1 := "TRANSFER DB".BUFF."MFG TO STORAGE-1 WITH INLINE HOMO", in2 := 0)
      R_Coil( "TRANSFER DB".PAUSE."MFG TO STORAGE-1 WITH INLINE HOMO" )
   END_RUNG
   // the same network as SCL:
   "IEC_Timer_0_DB_13".TON(IN := ("MODE SELECTION DB"."MODE BUFF" <> 0) AND ("TRANSFER DB".BUFF."MFG TO STORAGE-1 WITH INLINE HOMO" = 3),
                           PT := T#1S);
   IF "IEC_Timer_0_DB_13".Q THEN "TRANSFER DB".BUFF."MFG TO STORAGE-1 WITH INLINE HOMO" := 0; END_IF;
   IF "TRANSFER DB".STOP."MFG TO STORAGE-1 WITH INLINE HOMO" OR ("MODE SELECTION DB"."MODE BUFF" = 0) THEN
       "TRANSFER DB".BUFF."MFG TO STORAGE-1 WITH INLINE HOMO" := 0;
   END_IF;
   IF "TRANSFER DB".BUFF."MFG TO STORAGE-1 WITH INLINE HOMO" = 0 THEN
       "TRANSFER DB".PAUSE."MFG TO STORAGE-1 WITH INLINE HOMO" := FALSE;
   END_IF;
END_REGION

REGION Network 55: MFG TO STORAGE-1 WITH INLINE FILTER PRES_START
   RUNG wire#powerrail
      { S7_Templates := "SrcType := Int" } EQ_Contact(in1 := "MODE SELECTION DB"."MODE BUFF", in2 := 2)
      wire#w1
      { S7_Templates := "SrcType := Int" } EQ_Contact(in1 := "MANUAL INTERLOCK DB"."MFG TRANSFER PROCESS INTERLOCK", in2 := 0)
      { S7_Templates := "SrcType := Int" } EQ_Contact(in1 := "TRANSFER DB".BUFF."MFG TO STORAGE-1 WITH INLINE FILTER PRES", in2 := 0)
      { S7_Templates := "SrcType := Int" } EQ_Contact(in1 := "MANUAL INTERLOCK DB"."SYRUP MFG UNHEALTHY", in2 := 0)
      Contact( "TRANSFER DB".START."MFG TO STORAGE-1 WITH INLINE FILTER PRES" )
      { S7_Templates := "SrcType := Int" } NE_Contact(in1 := "CONTINUE DB"."SYRUP MFG PROCESS ERROR", in2 := 1)
      { S7_Templates := "SrcType := Int" } NE_Contact(in1 := "LEVEL BUFF"."SYRUP MFG_LOAD CELL", in2 := 1)
      Move(in := 1, out1 => "TRANSFER DB".BUFF."MFG TO STORAGE-1 WITH INLINE FILTER PRES")
   END_RUNG
   RUNG wire#powerrail
      { S7_Templates := "SrcType := Int" } EQ_Contact(in1 := "MODE SELECTION DB"."MODE BUFF", in2 := 1)
      { S7_Templates := "SrcType := Int" } EQ_Contact(in1 := "MFG PROCESS_DB"."AUTO BUFF", in2 := 180)
   END_RUNG wire#w1
   // the same network as SCL:
   IF (("MODE SELECTION DB"."MODE BUFF" = 2) OR (("MODE SELECTION DB"."MODE BUFF" = 1) AND ("MFG PROCESS_DB"."AUTO BUFF" = 180))) AND ("MANUAL INTERLOCK DB"."MFG TRANSFER PROCESS INTERLOCK" = 0) AND ("TRANSFER DB".BUFF."MFG TO STORAGE-1 WITH INLINE FILTER PRES" = 0) AND ("MANUAL INTERLOCK DB"."SYRUP MFG UNHEALTHY" = 0) AND "TRANSFER DB".START."MFG TO STORAGE-1 WITH INLINE FILTER PRES" AND ("CONTINUE DB"."SYRUP MFG PROCESS ERROR" <> 1) AND ("LEVEL BUFF"."SYRUP MFG_LOAD CELL" <> 1) THEN
       "TRANSFER DB".BUFF."MFG TO STORAGE-1 WITH INLINE FILTER PRES" := 1;
   END_IF;
END_REGION

REGION Network 56: MFG TO STORAGE-1 WITH INLINE FILTER PRES_START_POPUP
   RUNG wire#powerrail
      { S7_Templates := "SrcType := Int" } NE_Contact(in1 := "MODE SELECTION DB"."MODE BUFF", in2 := 0)
      { S7_Templates := "SrcType := Int" } EQ_Contact(in1 := "TRANSFER DB".BUFF."MFG TO STORAGE-1 WITH INLINE FILTER PRES", in2 := 1)
      { S7_Templates := "time_type := Time" } "IEC_Timer_0_DB_14".TON(pt := T#1S, et =>)
      Move(in := 2, out1 => "TRANSFER DB".BUFF."MFG TO STORAGE-1 WITH INLINE FILTER PRES")
   END_RUNG
   // the same network as SCL:
   "IEC_Timer_0_DB_14".TON(IN := ("MODE SELECTION DB"."MODE BUFF" <> 0) AND ("TRANSFER DB".BUFF."MFG TO STORAGE-1 WITH INLINE FILTER PRES" = 1),
                           PT := T#1S);
   IF "IEC_Timer_0_DB_14".Q THEN "TRANSFER DB".BUFF."MFG TO STORAGE-1 WITH INLINE FILTER PRES" := 2; END_IF;
END_REGION

REGION Network 57 (SCL): OPENVALVE
   IF ("MODE SELECTION DB"."MODE BUFF" <> 0 AND "TRANSFER DB".BUFF."MFG TO STORAGE-1 WITH INLINE FILTER PRES" = 2
       AND NOT "TRANSFER DB".PAUSE."MFG TO STORAGE-1 WITH INLINE FILTER PRES"
       AND "CONTINUE DB"."SYRUP MFG PROCESS ERROR" = 0 AND "LEVEL BUFF"."SYRUP MFG_LOAD CELL" = 0)
       OR ("MODE SELECTION DB"."MODE BUFF"=1 AND "MFG PROCESS_DB"."AUTO BUFF"=0
       AND "MFG TRANSFER CYCLE DB".TRANSFER."TRANSFER BUFF"."MFG TO STORAGE-1 WITH INLINE FILTER PRES"=10 AND "CONTINUE DB"."SYRUP MFG PROCESS ERROR" <>1
       AND "MFG TRANSFER CYCLE DB".TRANSFER.SELECT."SELECT BUFF"=2)
   THEN
       "TRANSFER DB".BIT."MFG TO STORAGE-1 WITH INLINE FILTER PRES"."PFBV-59 TANK OUTLET VALVE" := TRUE;
       "TRANSFER DB".BIT."MFG TO STORAGE-1 WITH INLINE FILTER PRES"."PBV-114 TANK OUTLET TO INLINE HOMOGENIZER LINE" := TRUE;
       "TRANSFER DB".BIT."MFG TO STORAGE-1 WITH INLINE FILTER PRES"."PBV-108 INLINE HOMOGENIZER TO FILTER PRESS INLET LINE" := TRUE;
       "TRANSFER DB".BIT."MFG TO STORAGE-1 WITH INLINE FILTER PRES"."FILTER PRESS MOTOR 1 RUN" := TRUE;
       "TRANSFER DB".BIT."MFG TO STORAGE-1 WITH INLINE FILTER PRES"."PBV-118 FILTER PRESS INLET" := TRUE;
       "TRANSFER DB".BIT."MFG TO STORAGE-1 WITH INLINE FILTER PRES"."PBV-111 FILTER PRESS OUTLER VALVE" := TRUE;
       "TRANSFER DB".BIT."MFG TO STORAGE-1 WITH INLINE FILTER PRES"."PBV-112 FILTER PRESS TO TRANSFER LINE" := TRUE;
       "TRANSFER DB".BIT."MFG TO STORAGE-1 WITH INLINE FILTER PRES"."PBV-115 MFG TO STORAGE – 1 TRANSFER LINE" := TRUE;
   ELSE
       "TRANSFER DB".BIT."MFG TO STORAGE-1 WITH INLINE FILTER PRES"."PFBV-59 TANK OUTLET VALVE" := FALSE;
       "TRANSFER DB".BIT."MFG TO STORAGE-1 WITH INLINE FILTER PRES"."PBV-114 TANK OUTLET TO INLINE HOMOGENIZER LINE" := FALSE;
       "TRANSFER DB".BIT."MFG TO STORAGE-1 WITH INLINE FILTER PRES"."PBV-108 INLINE HOMOGENIZER TO FILTER PRESS INLET LINE" := FALSE;
       "TRANSFER DB".BIT."MFG TO STORAGE-1 WITH INLINE FILTER PRES"."FILTER PRESS MOTOR 1 RUN" := FALSE;
       "TRANSFER DB".BIT."MFG TO STORAGE-1 WITH INLINE FILTER PRES"."PBV-118 FILTER PRESS INLET" := FALSE;
       "TRANSFER DB".BIT."MFG TO STORAGE-1 WITH INLINE FILTER PRES"."PBV-111 FILTER PRESS OUTLER VALVE" := FALSE;
       "TRANSFER DB".BIT."MFG TO STORAGE-1 WITH INLINE FILTER PRES"."PBV-112 FILTER PRESS TO TRANSFER LINE" := FALSE;
       "TRANSFER DB".BIT."MFG TO STORAGE-1 WITH INLINE FILTER PRES"."PBV-115 MFG TO STORAGE – 1 TRANSFER LINE" := FALSE;
       ;
   END_IF;
END_REGION

REGION Network 58: LOAD CELL_CUTOFF
   RUNG wire#powerrail
      { S7_Templates := "SrcType := Int" } NE_Contact(in1 := "MODE SELECTION DB"."MODE BUFF", in2 := 0)
      { S7_Templates := "SrcType := Int" } EQ_Contact(in1 := "TRANSFER DB".BUFF."MFG TO STORAGE-1 WITH INLINE FILTER PRES", in2 := 2)
      I_Contact( "TRANSFER DB".PAUSE."MFG TO STORAGE-1 WITH INLINE FILTER PRES" )
      { S7_Templates := "SrcType := Int" } NE_Contact(in1 := "CONTINUE DB"."SYRUP MFG PROCESS ERROR", in2 := 1)
      { S7_Templates := "SrcType := Int" } EQ_Contact(in1 := "LEVEL BUFF"."SYRUP MFG_LOAD CELL", in2 := 1)
      Move(in := 3, out1 => "TRANSFER DB".BUFF."MFG TO STORAGE-1 WITH INLINE FILTER PRES")
   END_RUNG
   // the same network as SCL:
   IF ("MODE SELECTION DB"."MODE BUFF" <> 0) AND ("TRANSFER DB".BUFF."MFG TO STORAGE-1 WITH INLINE FILTER PRES" = 2) AND NOT "TRANSFER DB".PAUSE."MFG TO STORAGE-1 WITH INLINE FILTER PRES" AND ("CONTINUE DB"."SYRUP MFG PROCESS ERROR" <> 1) AND ("LEVEL BUFF"."SYRUP MFG_LOAD CELL" = 1) THEN
       "TRANSFER DB".BUFF."MFG TO STORAGE-1 WITH INLINE FILTER PRES" := 3;
   END_IF;
END_REGION

REGION Network 59: PROCESS OVER & STOP
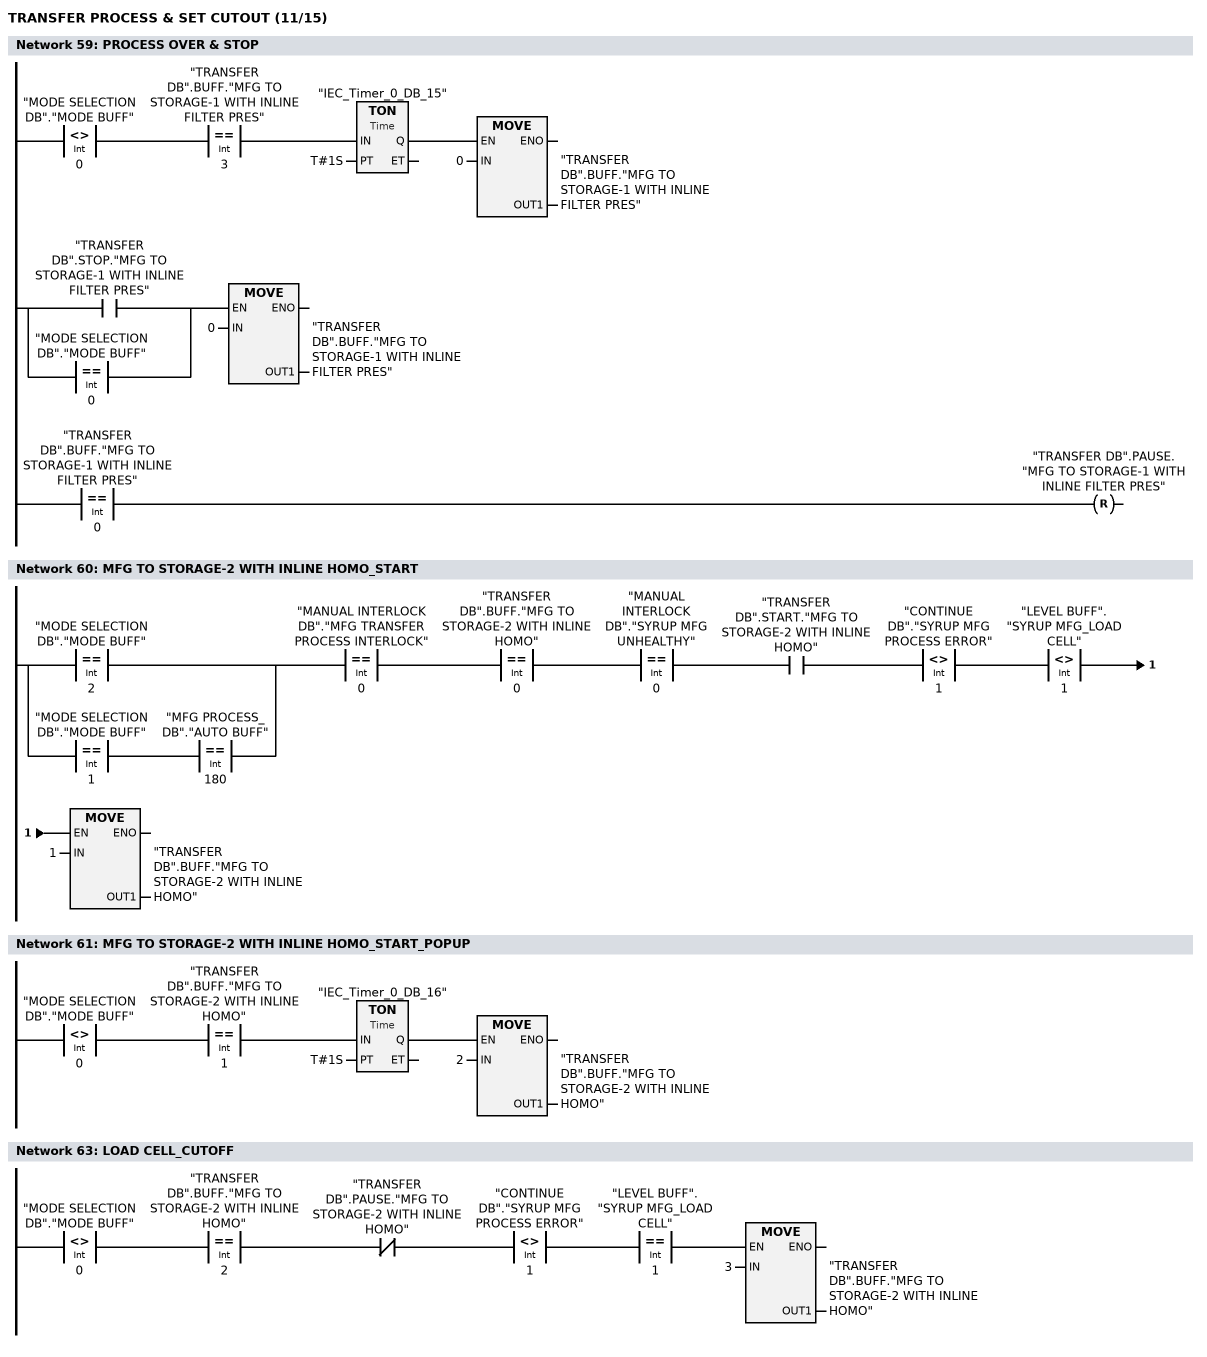
   RUNG wire#powerrail
      { S7_Templates := "SrcType := Int" } NE_Contact(in1 := "MODE SELECTION DB"."MODE BUFF", in2 := 0)
      { S7_Templates := "SrcType := Int" } EQ_Contact(in1 := "TRANSFER DB".BUFF."MFG TO STORAGE-1 WITH INLINE FILTER PRES", in2 := 3)
      { S7_Templates := "time_type := Time" } "IEC_Timer_0_DB_15".TON(pt := T#1S, et =>)
      Move(in := 0, out1 => "TRANSFER DB".BUFF."MFG TO STORAGE-1 WITH INLINE FILTER PRES")
   END_RUNG
   RUNG wire#powerrail
      Contact( "TRANSFER DB".STOP."MFG TO STORAGE-1 WITH INLINE FILTER PRES" )
      wire#w1
      Move(in := 0, out1 => "TRANSFER DB".BUFF."MFG TO STORAGE-1 WITH INLINE FILTER PRES")
   END_RUNG
   RUNG wire#powerrail
      { S7_Templates := "SrcType := Int" } EQ_Contact(in1 := "MODE SELECTION DB"."MODE BUFF", in2 := 0)
   END_RUNG wire#w1
   RUNG wire#powerrail
      { S7_Templates := "SrcType := Int" } EQ_Contact(in1 := "TRANSFER DB".BUFF."MFG TO STORAGE-1 WITH INLINE FILTER PRES", in2 := 0)
      R_Coil( "TRANSFER DB".PAUSE."MFG TO STORAGE-1 WITH INLINE FILTER PRES" )
   END_RUNG
   // the same network as SCL:
   "IEC_Timer_0_DB_15".TON(IN := ("MODE SELECTION DB"."MODE BUFF" <> 0) AND ("TRANSFER DB".BUFF."MFG TO STORAGE-1 WITH INLINE FILTER PRES" = 3),
                           PT := T#1S);
   IF "IEC_Timer_0_DB_15".Q THEN "TRANSFER DB".BUFF."MFG TO STORAGE-1 WITH INLINE FILTER PRES" := 0; END_IF;
   IF "TRANSFER DB".STOP."MFG TO STORAGE-1 WITH INLINE FILTER PRES" OR ("MODE SELECTION DB"."MODE BUFF" = 0) THEN
       "TRANSFER DB".BUFF."MFG TO STORAGE-1 WITH INLINE FILTER PRES" := 0;
   END_IF;
   IF "TRANSFER DB".BUFF."MFG TO STORAGE-1 WITH INLINE FILTER PRES" = 0 THEN
       "TRANSFER DB".PAUSE."MFG TO STORAGE-1 WITH INLINE FILTER PRES" := FALSE;
   END_IF;
END_REGION

REGION Network 60: MFG TO STORAGE-2 WITH INLINE HOMO_START
   RUNG wire#powerrail
      { S7_Templates := "SrcType := Int" } EQ_Contact(in1 := "MODE SELECTION DB"."MODE BUFF", in2 := 2)
      wire#w1
      { S7_Templates := "SrcType := Int" } EQ_Contact(in1 := "MANUAL INTERLOCK DB"."MFG TRANSFER PROCESS INTERLOCK", in2 := 0)
      { S7_Templates := "SrcType := Int" } EQ_Contact(in1 := "TRANSFER DB".BUFF."MFG TO STORAGE-2 WITH INLINE HOMO", in2 := 0)
      { S7_Templates := "SrcType := Int" } EQ_Contact(in1 := "MANUAL INTERLOCK DB"."SYRUP MFG UNHEALTHY", in2 := 0)
      Contact( "TRANSFER DB".START."MFG TO STORAGE-2 WITH INLINE HOMO" )
      { S7_Templates := "SrcType := Int" } NE_Contact(in1 := "CONTINUE DB"."SYRUP MFG PROCESS ERROR", in2 := 1)
      { S7_Templates := "SrcType := Int" } NE_Contact(in1 := "LEVEL BUFF"."SYRUP MFG_LOAD CELL", in2 := 1)
      Move(in := 1, out1 => "TRANSFER DB".BUFF."MFG TO STORAGE-2 WITH INLINE HOMO")
   END_RUNG
   RUNG wire#powerrail
      { S7_Templates := "SrcType := Int" } EQ_Contact(in1 := "MODE SELECTION DB"."MODE BUFF", in2 := 1)
      { S7_Templates := "SrcType := Int" } EQ_Contact(in1 := "MFG PROCESS_DB"."AUTO BUFF", in2 := 180)
   END_RUNG wire#w1
   // the same network as SCL:
   IF (("MODE SELECTION DB"."MODE BUFF" = 2) OR (("MODE SELECTION DB"."MODE BUFF" = 1) AND ("MFG PROCESS_DB"."AUTO BUFF" = 180))) AND ("MANUAL INTERLOCK DB"."MFG TRANSFER PROCESS INTERLOCK" = 0) AND ("TRANSFER DB".BUFF."MFG TO STORAGE-2 WITH INLINE HOMO" = 0) AND ("MANUAL INTERLOCK DB"."SYRUP MFG UNHEALTHY" = 0) AND "TRANSFER DB".START."MFG TO STORAGE-2 WITH INLINE HOMO" AND ("CONTINUE DB"."SYRUP MFG PROCESS ERROR" <> 1) AND ("LEVEL BUFF"."SYRUP MFG_LOAD CELL" <> 1) THEN
       "TRANSFER DB".BUFF."MFG TO STORAGE-2 WITH INLINE HOMO" := 1;
   END_IF;
END_REGION

REGION Network 61: MFG TO STORAGE-2 WITH INLINE HOMO_START_POPUP
   RUNG wire#powerrail
      { S7_Templates := "SrcType := Int" } NE_Contact(in1 := "MODE SELECTION DB"."MODE BUFF", in2 := 0)
      { S7_Templates := "SrcType := Int" } EQ_Contact(in1 := "TRANSFER DB".BUFF."MFG TO STORAGE-2 WITH INLINE HOMO", in2 := 1)
      { S7_Templates := "time_type := Time" } "IEC_Timer_0_DB_16".TON(pt := T#1S, et =>)
      Move(in := 2, out1 => "TRANSFER DB".BUFF."MFG TO STORAGE-2 WITH INLINE HOMO")
   END_RUNG
   // the same network as SCL:
   "IEC_Timer_0_DB_16".TON(IN := ("MODE SELECTION DB"."MODE BUFF" <> 0) AND ("TRANSFER DB".BUFF."MFG TO STORAGE-2 WITH INLINE HOMO" = 1),
                           PT := T#1S);
   IF "IEC_Timer_0_DB_16".Q THEN "TRANSFER DB".BUFF."MFG TO STORAGE-2 WITH INLINE HOMO" := 2; END_IF;
END_REGION

REGION Network 62 (SCL): OPENVALVE
   IF ("MODE SELECTION DB"."MODE BUFF" <> 0 AND "TRANSFER DB".BUFF."MFG TO STORAGE-2 WITH INLINE HOMO" = 2
       AND NOT "TRANSFER DB".PAUSE."MFG TO STORAGE-2 WITH INLINE HOMO"
       AND "CONTINUE DB"."SYRUP MFG PROCESS ERROR" = 0 AND "LEVEL BUFF"."SYRUP MFG_LOAD CELL" = 0)
       OR ("MODE SELECTION DB"."MODE BUFF"=1 AND "MFG PROCESS_DB"."AUTO BUFF"=0
       AND "MFG TRANSFER CYCLE DB".TRANSFER."TRANSFER BUFF"."MFG TO STORAGE-2 WITH INLINE HOMO"=10 AND "CONTINUE DB"."SYRUP MFG PROCESS ERROR" <>1
       AND "MFG TRANSFER CYCLE DB".TRANSFER.SELECT."SELECT BUFF"=3)
   THEN
       "TRANSFER DB".BIT."MFG TO STORAGE-2 WITH INLINE HOMO"."PFBV-59 TANK OUTLET VALVE" := TRUE;
       "TRANSFER DB".BIT."MFG TO STORAGE-2 WITH INLINE HOMO"."PBV-114 TANK OUTLET TO INLINE HOMOGENIZER LINE" := TRUE;
       "TRANSFER DB".BIT."MFG TO STORAGE-2 WITH INLINE HOMO"."PBV-110 INLINE HOMOGENIZER TO INLET LINE" := TRUE;
       "TRANSFER DB".BIT."MFG TO STORAGE-2 WITH INLINE HOMO"."PAV-56 INLINE HOMO. SEAL COOLING INLET" := TRUE;
       "TRANSFER DB".BIT."MFG TO STORAGE-2 WITH INLINE HOMO"."INLINE 1 HOMOGENIZER MOTOR1 RUN" := TRUE;
       "TRANSFER DB".BIT."MFG TO STORAGE-2 WITH INLINE HOMO"."PBV-109 HOMO. RECIRCULATION INLET" := TRUE;
       "TRANSFER DB".BIT."MFG TO STORAGE-2 WITH INLINE HOMO"."PBV-116 MFG TO STORAGE – 2 TRANSFER LINE" := TRUE;
   ELSE
       "TRANSFER DB".BIT."MFG TO STORAGE-2 WITH INLINE HOMO"."PFBV-59 TANK OUTLET VALVE" := FALSE;
       "TRANSFER DB".BIT."MFG TO STORAGE-2 WITH INLINE HOMO"."PBV-114 TANK OUTLET TO INLINE HOMOGENIZER LINE" := FALSE;
       "TRANSFER DB".BIT."MFG TO STORAGE-2 WITH INLINE HOMO"."PBV-110 INLINE HOMOGENIZER TO INLET LINE" := FALSE;
       "TRANSFER DB".BIT."MFG TO STORAGE-2 WITH INLINE HOMO"."PAV-56 INLINE HOMO. SEAL COOLING INLET" := FALSE;
       "TRANSFER DB".BIT."MFG TO STORAGE-2 WITH INLINE HOMO"."INLINE 1 HOMOGENIZER MOTOR1 RUN" := FALSE;
       "TRANSFER DB".BIT."MFG TO STORAGE-2 WITH INLINE HOMO"."PBV-109 HOMO. RECIRCULATION INLET" := FALSE;
       "TRANSFER DB".BIT."MFG TO STORAGE-2 WITH INLINE HOMO"."PBV-116 MFG TO STORAGE – 2 TRANSFER LINE" := FALSE;
       ;
   END_IF;
END_REGION

REGION Network 63: LOAD CELL_CUTOFF
   RUNG wire#powerrail
      { S7_Templates := "SrcType := Int" } NE_Contact(in1 := "MODE SELECTION DB"."MODE BUFF", in2 := 0)
      { S7_Templates := "SrcType := Int" } EQ_Contact(in1 := "TRANSFER DB".BUFF."MFG TO STORAGE-2 WITH INLINE HOMO", in2 := 2)
      I_Contact( "TRANSFER DB".PAUSE."MFG TO STORAGE-2 WITH INLINE HOMO" )
      { S7_Templates := "SrcType := Int" } NE_Contact(in1 := "CONTINUE DB"."SYRUP MFG PROCESS ERROR", in2 := 1)
      { S7_Templates := "SrcType := Int" } EQ_Contact(in1 := "LEVEL BUFF"."SYRUP MFG_LOAD CELL", in2 := 1)
      Move(in := 3, out1 => "TRANSFER DB".BUFF."MFG TO STORAGE-2 WITH INLINE HOMO")
   END_RUNG
   // the same network as SCL:
   IF ("MODE SELECTION DB"."MODE BUFF" <> 0) AND ("TRANSFER DB".BUFF."MFG TO STORAGE-2 WITH INLINE HOMO" = 2) AND NOT "TRANSFER DB".PAUSE."MFG TO STORAGE-2 WITH INLINE HOMO" AND ("CONTINUE DB"."SYRUP MFG PROCESS ERROR" <> 1) AND ("LEVEL BUFF"."SYRUP MFG_LOAD CELL" = 1) THEN
       "TRANSFER DB".BUFF."MFG TO STORAGE-2 WITH INLINE HOMO" := 3;
   END_IF;
END_REGION

REGION Network 64: PROCESS OVER & STOP
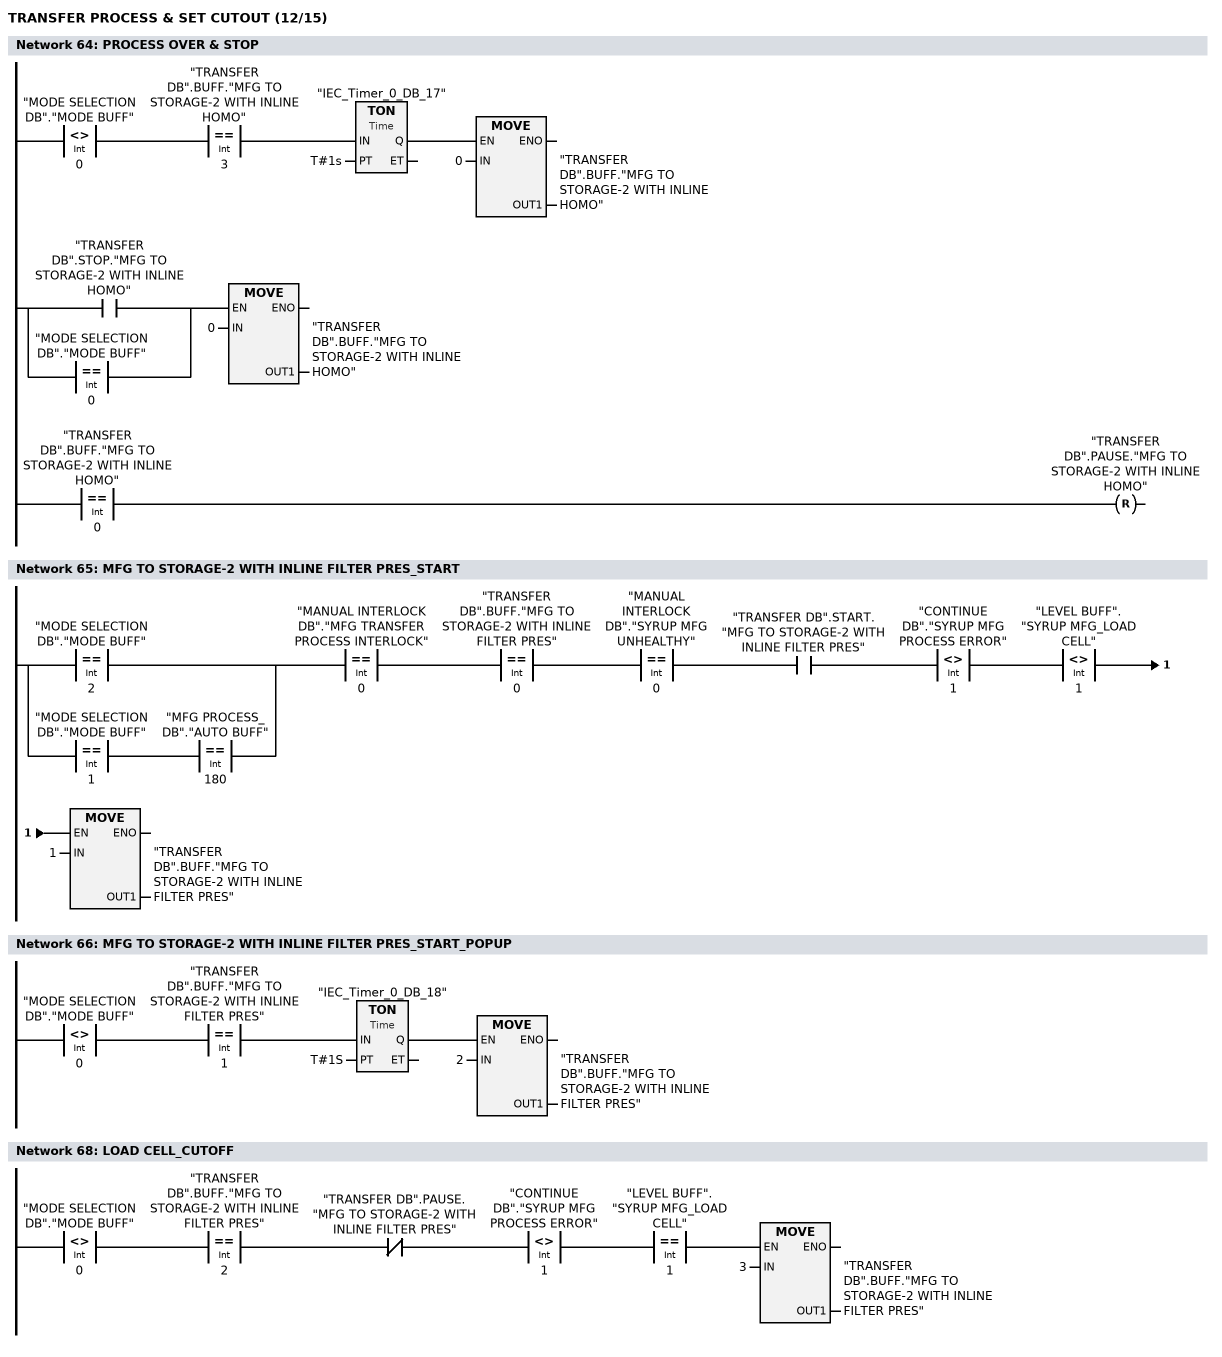
   RUNG wire#powerrail
      { S7_Templates := "SrcType := Int" } NE_Contact(in1 := "MODE SELECTION DB"."MODE BUFF", in2 := 0)
      { S7_Templates := "SrcType := Int" } EQ_Contact(in1 := "TRANSFER DB".BUFF."MFG TO STORAGE-2 WITH INLINE HOMO", in2 := 3)
      { S7_Templates := "time_type := Time" } "IEC_Timer_0_DB_17".TON(pt := T#1s, et =>)
      Move(in := 0, out1 => "TRANSFER DB".BUFF."MFG TO STORAGE-2 WITH INLINE HOMO")
   END_RUNG
   RUNG wire#powerrail
      Contact( "TRANSFER DB".STOP."MFG TO STORAGE-2 WITH INLINE HOMO" )
      wire#w1
      Move(in := 0, out1 => "TRANSFER DB".BUFF."MFG TO STORAGE-2 WITH INLINE HOMO")
   END_RUNG
   RUNG wire#powerrail
      { S7_Templates := "SrcType := Int" } EQ_Contact(in1 := "MODE SELECTION DB"."MODE BUFF", in2 := 0)
   END_RUNG wire#w1
   RUNG wire#powerrail
      { S7_Templates := "SrcType := Int" } EQ_Contact(in1 := "TRANSFER DB".BUFF."MFG TO STORAGE-2 WITH INLINE HOMO", in2 := 0)
      R_Coil( "TRANSFER DB".PAUSE."MFG TO STORAGE-2 WITH INLINE HOMO" )
   END_RUNG
   // the same network as SCL:
   "IEC_Timer_0_DB_17".TON(IN := ("MODE SELECTION DB"."MODE BUFF" <> 0) AND ("TRANSFER DB".BUFF."MFG TO STORAGE-2 WITH INLINE HOMO" = 3),
                           PT := T#1s);
   IF "IEC_Timer_0_DB_17".Q THEN "TRANSFER DB".BUFF."MFG TO STORAGE-2 WITH INLINE HOMO" := 0; END_IF;
   IF "TRANSFER DB".STOP."MFG TO STORAGE-2 WITH INLINE HOMO" OR ("MODE SELECTION DB"."MODE BUFF" = 0) THEN
       "TRANSFER DB".BUFF."MFG TO STORAGE-2 WITH INLINE HOMO" := 0;
   END_IF;
   IF "TRANSFER DB".BUFF."MFG TO STORAGE-2 WITH INLINE HOMO" = 0 THEN
       "TRANSFER DB".PAUSE."MFG TO STORAGE-2 WITH INLINE HOMO" := FALSE;
   END_IF;
END_REGION

REGION Network 65: MFG TO STORAGE-2 WITH INLINE FILTER PRES_START
   RUNG wire#powerrail
      { S7_Templates := "SrcType := Int" } EQ_Contact(in1 := "MODE SELECTION DB"."MODE BUFF", in2 := 2)
      wire#w1
      { S7_Templates := "SrcType := Int" } EQ_Contact(in1 := "MANUAL INTERLOCK DB"."MFG TRANSFER PROCESS INTERLOCK", in2 := 0)
      { S7_Templates := "SrcType := Int" } EQ_Contact(in1 := "TRANSFER DB".BUFF."MFG TO STORAGE-2 WITH INLINE FILTER PRES", in2 := 0)
      { S7_Templates := "SrcType := Int" } EQ_Contact(in1 := "MANUAL INTERLOCK DB"."SYRUP MFG UNHEALTHY", in2 := 0)
      Contact( "TRANSFER DB".START."MFG TO STORAGE-2 WITH INLINE FILTER PRES" )
      { S7_Templates := "SrcType := Int" } NE_Contact(in1 := "CONTINUE DB"."SYRUP MFG PROCESS ERROR", in2 := 1)
      { S7_Templates := "SrcType := Int" } NE_Contact(in1 := "LEVEL BUFF"."SYRUP MFG_LOAD CELL", in2 := 1)
      Move(in := 1, out1 => "TRANSFER DB".BUFF."MFG TO STORAGE-2 WITH INLINE FILTER PRES")
   END_RUNG
   RUNG wire#powerrail
      { S7_Templates := "SrcType := Int" } EQ_Contact(in1 := "MODE SELECTION DB"."MODE BUFF", in2 := 1)
      { S7_Templates := "SrcType := Int" } EQ_Contact(in1 := "MFG PROCESS_DB"."AUTO BUFF", in2 := 180)
   END_RUNG wire#w1
   // the same network as SCL:
   IF (("MODE SELECTION DB"."MODE BUFF" = 2) OR (("MODE SELECTION DB"."MODE BUFF" = 1) AND ("MFG PROCESS_DB"."AUTO BUFF" = 180))) AND ("MANUAL INTERLOCK DB"."MFG TRANSFER PROCESS INTERLOCK" = 0) AND ("TRANSFER DB".BUFF."MFG TO STORAGE-2 WITH INLINE FILTER PRES" = 0) AND ("MANUAL INTERLOCK DB"."SYRUP MFG UNHEALTHY" = 0) AND "TRANSFER DB".START."MFG TO STORAGE-2 WITH INLINE FILTER PRES" AND ("CONTINUE DB"."SYRUP MFG PROCESS ERROR" <> 1) AND ("LEVEL BUFF"."SYRUP MFG_LOAD CELL" <> 1) THEN
       "TRANSFER DB".BUFF."MFG TO STORAGE-2 WITH INLINE FILTER PRES" := 1;
   END_IF;
END_REGION

REGION Network 66: MFG TO STORAGE-2 WITH INLINE FILTER PRES_START_POPUP
   RUNG wire#powerrail
      { S7_Templates := "SrcType := Int" } NE_Contact(in1 := "MODE SELECTION DB"."MODE BUFF", in2 := 0)
      { S7_Templates := "SrcType := Int" } EQ_Contact(in1 := "TRANSFER DB".BUFF."MFG TO STORAGE-2 WITH INLINE FILTER PRES", in2 := 1)
      { S7_Templates := "time_type := Time" } "IEC_Timer_0_DB_18".TON(pt := T#1S, et =>)
      Move(in := 2, out1 => "TRANSFER DB".BUFF."MFG TO STORAGE-2 WITH INLINE FILTER PRES")
   END_RUNG
   // the same network as SCL:
   "IEC_Timer_0_DB_18".TON(IN := ("MODE SELECTION DB"."MODE BUFF" <> 0) AND ("TRANSFER DB".BUFF."MFG TO STORAGE-2 WITH INLINE FILTER PRES" = 1),
                           PT := T#1S);
   IF "IEC_Timer_0_DB_18".Q THEN "TRANSFER DB".BUFF."MFG TO STORAGE-2 WITH INLINE FILTER PRES" := 2; END_IF;
END_REGION

REGION Network 67 (SCL): OPENVALVE
   IF ("MODE SELECTION DB"."MODE BUFF" <> 0 AND "TRANSFER DB".BUFF."MFG TO STORAGE-2 WITH INLINE FILTER PRES" = 2
       AND NOT "TRANSFER DB".PAUSE."MFG TO STORAGE-2 WITH INLINE FILTER PRES" 
       AND "CONTINUE DB"."SYRUP MFG PROCESS ERROR" = 0 AND "LEVEL BUFF"."SYRUP MFG_LOAD CELL" = 0)
       OR ("MODE SELECTION DB"."MODE BUFF"=1 AND "MFG PROCESS_DB"."AUTO BUFF"=0
       AND "MFG TRANSFER CYCLE DB".TRANSFER."TRANSFER BUFF"."MFG TO STORAGE-2 WITH INLINE FILTER PRES"=10 AND "CONTINUE DB"."SYRUP MFG PROCESS ERROR" <>1
       AND "MFG TRANSFER CYCLE DB".TRANSFER.SELECT."SELECT BUFF"=4)
   THEN
       "TRANSFER DB".BIT."MFG TO STORAGE-2 WITH INLINE FILTER PRES"."PFBV-59 TANK OUTLET VALVE" := TRUE;
       "TRANSFER DB".BIT."MFG TO STORAGE-2 WITH INLINE FILTER PRES"."PBV-114 TANK OUTLET TO INLINE HOMOGENIZER LINE" := TRUE;
       "TRANSFER DB".BIT."MFG TO STORAGE-2 WITH INLINE FILTER PRES"."PBV-108 INLINE HOMOGENIZER TO FILTER PRESS INLET LINE" := TRUE;
       "TRANSFER DB".BIT."MFG TO STORAGE-2 WITH INLINE FILTER PRES"."FILTER PRESS MOTOR 1 RUN" := TRUE;
       "TRANSFER DB".BIT."MFG TO STORAGE-2 WITH INLINE FILTER PRES"."PBV-118 FILTER PRESS INLET" := TRUE;
       "TRANSFER DB".BIT."MFG TO STORAGE-2 WITH INLINE FILTER PRES"."PBV-111 FILTER PRESS OUTLER VALVE" := TRUE;
       "TRANSFER DB".BIT."MFG TO STORAGE-2 WITH INLINE FILTER PRES"."PBV-112 FILTER PRESS TO TRANSFER LINE" := TRUE;
       "TRANSFER DB".BIT."MFG TO STORAGE-2 WITH INLINE FILTER PRES"."PBV-116 MFG TO STORAGE – 2 TRANSFER LINE" := TRUE;
   ELSE
       "TRANSFER DB".BIT."MFG TO STORAGE-2 WITH INLINE FILTER PRES"."PFBV-59 TANK OUTLET VALVE" := FALSE;
       "TRANSFER DB".BIT."MFG TO STORAGE-2 WITH INLINE FILTER PRES"."PBV-114 TANK OUTLET TO INLINE HOMOGENIZER LINE" := FALSE;
       "TRANSFER DB".BIT."MFG TO STORAGE-2 WITH INLINE FILTER PRES"."PBV-108 INLINE HOMOGENIZER TO FILTER PRESS INLET LINE" := FALSE;
       "TRANSFER DB".BIT."MFG TO STORAGE-2 WITH INLINE FILTER PRES"."FILTER PRESS MOTOR 1 RUN" := FALSE;
       "TRANSFER DB".BIT."MFG TO STORAGE-2 WITH INLINE FILTER PRES"."PBV-118 FILTER PRESS INLET" := FALSE;
       "TRANSFER DB".BIT."MFG TO STORAGE-2 WITH INLINE FILTER PRES"."PBV-111 FILTER PRESS OUTLER VALVE" := FALSE;
       "TRANSFER DB".BIT."MFG TO STORAGE-2 WITH INLINE FILTER PRES"."PBV-112 FILTER PRESS TO TRANSFER LINE" := FALSE;
       "TRANSFER DB".BIT."MFG TO STORAGE-2 WITH INLINE FILTER PRES"."PBV-116 MFG TO STORAGE – 2 TRANSFER LINE" := FALSE;
       ;
   END_IF;
END_REGION

REGION Network 68: LOAD CELL_CUTOFF
   RUNG wire#powerrail
      { S7_Templates := "SrcType := Int" } NE_Contact(in1 := "MODE SELECTION DB"."MODE BUFF", in2 := 0)
      { S7_Templates := "SrcType := Int" } EQ_Contact(in1 := "TRANSFER DB".BUFF."MFG TO STORAGE-2 WITH INLINE FILTER PRES", in2 := 2)
      I_Contact( "TRANSFER DB".PAUSE."MFG TO STORAGE-2 WITH INLINE FILTER PRES" )
      { S7_Templates := "SrcType := Int" } NE_Contact(in1 := "CONTINUE DB"."SYRUP MFG PROCESS ERROR", in2 := 1)
      { S7_Templates := "SrcType := Int" } EQ_Contact(in1 := "LEVEL BUFF"."SYRUP MFG_LOAD CELL", in2 := 1)
      Move(in := 3, out1 => "TRANSFER DB".BUFF."MFG TO STORAGE-2 WITH INLINE FILTER PRES")
   END_RUNG
   // the same network as SCL:
   IF ("MODE SELECTION DB"."MODE BUFF" <> 0) AND ("TRANSFER DB".BUFF."MFG TO STORAGE-2 WITH INLINE FILTER PRES" = 2) AND NOT "TRANSFER DB".PAUSE."MFG TO STORAGE-2 WITH INLINE FILTER PRES" AND ("CONTINUE DB"."SYRUP MFG PROCESS ERROR" <> 1) AND ("LEVEL BUFF"."SYRUP MFG_LOAD CELL" = 1) THEN
       "TRANSFER DB".BUFF."MFG TO STORAGE-2 WITH INLINE FILTER PRES" := 3;
   END_IF;
END_REGION

REGION Network 69: PROCESS OVER & STOP
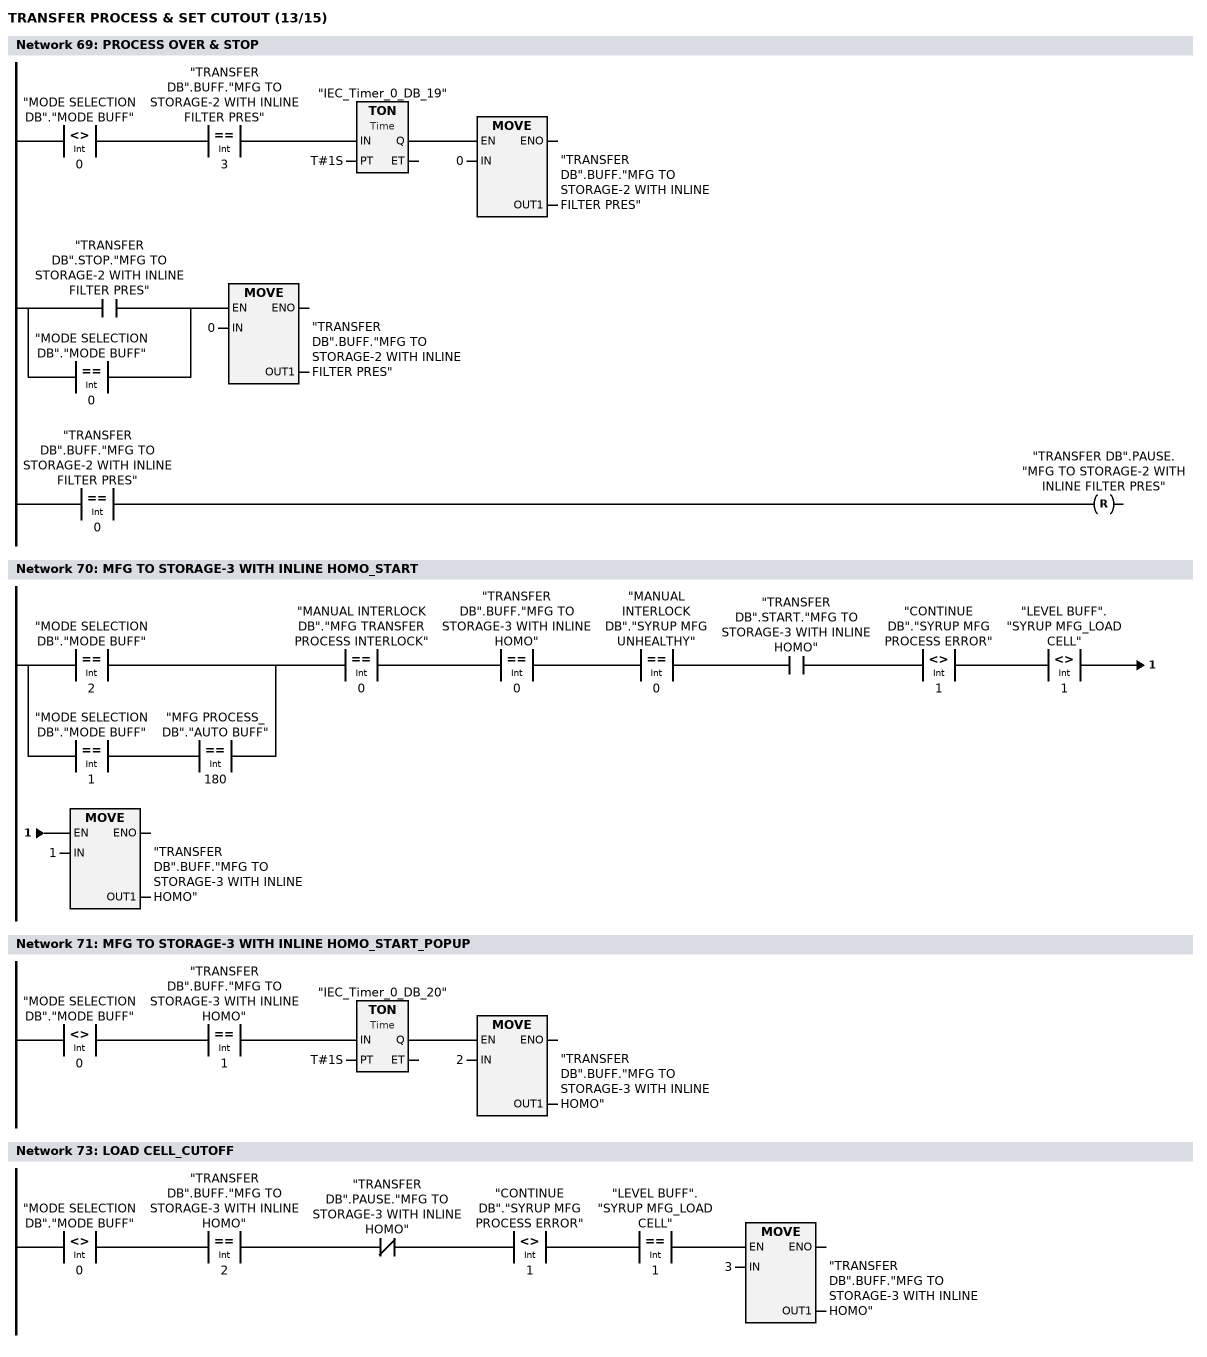
   RUNG wire#powerrail
      { S7_Templates := "SrcType := Int" } NE_Contact(in1 := "MODE SELECTION DB"."MODE BUFF", in2 := 0)
      { S7_Templates := "SrcType := Int" } EQ_Contact(in1 := "TRANSFER DB".BUFF."MFG TO STORAGE-2 WITH INLINE FILTER PRES", in2 := 3)
      { S7_Templates := "time_type := Time" } "IEC_Timer_0_DB_19".TON(pt := T#1S, et =>)
      Move(in := 0, out1 => "TRANSFER DB".BUFF."MFG TO STORAGE-2 WITH INLINE FILTER PRES")
   END_RUNG
   RUNG wire#powerrail
      Contact( "TRANSFER DB".STOP."MFG TO STORAGE-2 WITH INLINE FILTER PRES" )
      wire#w1
      Move(in := 0, out1 => "TRANSFER DB".BUFF."MFG TO STORAGE-2 WITH INLINE FILTER PRES")
   END_RUNG
   RUNG wire#powerrail
      { S7_Templates := "SrcType := Int" } EQ_Contact(in1 := "MODE SELECTION DB"."MODE BUFF", in2 := 0)
   END_RUNG wire#w1
   RUNG wire#powerrail
      { S7_Templates := "SrcType := Int" } EQ_Contact(in1 := "TRANSFER DB".BUFF."MFG TO STORAGE-2 WITH INLINE FILTER PRES", in2 := 0)
      R_Coil( "TRANSFER DB".PAUSE."MFG TO STORAGE-2 WITH INLINE FILTER PRES" )
   END_RUNG
   // the same network as SCL:
   "IEC_Timer_0_DB_19".TON(IN := ("MODE SELECTION DB"."MODE BUFF" <> 0) AND ("TRANSFER DB".BUFF."MFG TO STORAGE-2 WITH INLINE FILTER PRES" = 3),
                           PT := T#1S);
   IF "IEC_Timer_0_DB_19".Q THEN "TRANSFER DB".BUFF."MFG TO STORAGE-2 WITH INLINE FILTER PRES" := 0; END_IF;
   IF "TRANSFER DB".STOP."MFG TO STORAGE-2 WITH INLINE FILTER PRES" OR ("MODE SELECTION DB"."MODE BUFF" = 0) THEN
       "TRANSFER DB".BUFF."MFG TO STORAGE-2 WITH INLINE FILTER PRES" := 0;
   END_IF;
   IF "TRANSFER DB".BUFF."MFG TO STORAGE-2 WITH INLINE FILTER PRES" = 0 THEN
       "TRANSFER DB".PAUSE."MFG TO STORAGE-2 WITH INLINE FILTER PRES" := FALSE;
   END_IF;
END_REGION

REGION Network 70: MFG TO STORAGE-3 WITH INLINE HOMO_START
   RUNG wire#powerrail
      { S7_Templates := "SrcType := Int" } EQ_Contact(in1 := "MODE SELECTION DB"."MODE BUFF", in2 := 2)
      wire#w1
      { S7_Templates := "SrcType := Int" } EQ_Contact(in1 := "MANUAL INTERLOCK DB"."MFG TRANSFER PROCESS INTERLOCK", in2 := 0)
      { S7_Templates := "SrcType := Int" } EQ_Contact(in1 := "TRANSFER DB".BUFF."MFG TO STORAGE-3 WITH INLINE HOMO", in2 := 0)
      { S7_Templates := "SrcType := Int" } EQ_Contact(in1 := "MANUAL INTERLOCK DB"."SYRUP MFG UNHEALTHY", in2 := 0)
      Contact( "TRANSFER DB".START."MFG TO STORAGE-3 WITH INLINE HOMO" )
      { S7_Templates := "SrcType := Int" } NE_Contact(in1 := "CONTINUE DB"."SYRUP MFG PROCESS ERROR", in2 := 1)
      { S7_Templates := "SrcType := Int" } NE_Contact(in1 := "LEVEL BUFF"."SYRUP MFG_LOAD CELL", in2 := 1)
      Move(in := 1, out1 => "TRANSFER DB".BUFF."MFG TO STORAGE-3 WITH INLINE HOMO")
   END_RUNG
   RUNG wire#powerrail
      { S7_Templates := "SrcType := Int" } EQ_Contact(in1 := "MODE SELECTION DB"."MODE BUFF", in2 := 1)
      { S7_Templates := "SrcType := Int" } EQ_Contact(in1 := "MFG PROCESS_DB"."AUTO BUFF", in2 := 180)
   END_RUNG wire#w1
   // the same network as SCL:
   IF (("MODE SELECTION DB"."MODE BUFF" = 2) OR (("MODE SELECTION DB"."MODE BUFF" = 1) AND ("MFG PROCESS_DB"."AUTO BUFF" = 180))) AND ("MANUAL INTERLOCK DB"."MFG TRANSFER PROCESS INTERLOCK" = 0) AND ("TRANSFER DB".BUFF."MFG TO STORAGE-3 WITH INLINE HOMO" = 0) AND ("MANUAL INTERLOCK DB"."SYRUP MFG UNHEALTHY" = 0) AND "TRANSFER DB".START."MFG TO STORAGE-3 WITH INLINE HOMO" AND ("CONTINUE DB"."SYRUP MFG PROCESS ERROR" <> 1) AND ("LEVEL BUFF"."SYRUP MFG_LOAD CELL" <> 1) THEN
       "TRANSFER DB".BUFF."MFG TO STORAGE-3 WITH INLINE HOMO" := 1;
   END_IF;
END_REGION

REGION Network 71: MFG TO STORAGE-3 WITH INLINE HOMO_START_POPUP
   RUNG wire#powerrail
      { S7_Templates := "SrcType := Int" } NE_Contact(in1 := "MODE SELECTION DB"."MODE BUFF", in2 := 0)
      { S7_Templates := "SrcType := Int" } EQ_Contact(in1 := "TRANSFER DB".BUFF."MFG TO STORAGE-3 WITH INLINE HOMO", in2 := 1)
      { S7_Templates := "time_type := Time" } "IEC_Timer_0_DB_20".TON(pt := T#1S, et =>)
      Move(in := 2, out1 => "TRANSFER DB".BUFF."MFG TO STORAGE-3 WITH INLINE HOMO")
   END_RUNG
   // the same network as SCL:
   "IEC_Timer_0_DB_20".TON(IN := ("MODE SELECTION DB"."MODE BUFF" <> 0) AND ("TRANSFER DB".BUFF."MFG TO STORAGE-3 WITH INLINE HOMO" = 1),
                           PT := T#1S);
   IF "IEC_Timer_0_DB_20".Q THEN "TRANSFER DB".BUFF."MFG TO STORAGE-3 WITH INLINE HOMO" := 2; END_IF;
END_REGION

REGION Network 72 (SCL): OPENVALVE
   IF ("MODE SELECTION DB"."MODE BUFF" <> 0 AND "TRANSFER DB".BUFF."MFG TO STORAGE-3 WITH INLINE HOMO" = 2
       AND NOT "TRANSFER DB".PAUSE."MFG TO STORAGE-3 WITH INLINE HOMO"
       AND "CONTINUE DB"."SYRUP MFG PROCESS ERROR" = 0 AND "LEVEL BUFF"."SYRUP MFG_LOAD CELL" = 0)
       OR ("MODE SELECTION DB"."MODE BUFF"=1 AND "MFG PROCESS_DB"."AUTO BUFF"=0
       AND "MFG TRANSFER CYCLE DB".TRANSFER."TRANSFER BUFF"."MFG TO STORAGE-3 WITH INLINE HOMO"=10 AND "CONTINUE DB"."SYRUP MFG PROCESS ERROR" <>1
       AND "MFG TRANSFER CYCLE DB".TRANSFER.SELECT."SELECT BUFF"=5)
   THEN
       "TRANSFER DB".BIT."MFG TO STORAGE-3 WITH INLINE HOMO"."PFBV-59 TANK OUTLET VALVE" := TRUE;
       "TRANSFER DB".BIT."MFG TO STORAGE-3 WITH INLINE HOMO"."PBV-114 TANK OUTLET TO INLINE HOMOGENIZER LINE" := TRUE;
       "TRANSFER DB".BIT."MFG TO STORAGE-3 WITH INLINE HOMO"."PBV-110 INLINE HOMOGENIZER TO INLET LINE" := TRUE;
       "TRANSFER DB".BIT."MFG TO STORAGE-3 WITH INLINE HOMO"."PAV-56 INLINE HOMO. SEAL COOLING INLET" := TRUE;
       "TRANSFER DB".BIT."MFG TO STORAGE-3 WITH INLINE HOMO"."INLINE 1 HOMOGENIZER MOTOR1 RUN" := TRUE;
       "TRANSFER DB".BIT."MFG TO STORAGE-3 WITH INLINE HOMO"."PBV-109 HOMO. RECIRCULATION INLET" := TRUE;
       "TRANSFER DB".BIT."MFG TO STORAGE-3 WITH INLINE HOMO"."PBV-117 MFG TO STORAGE – 3 TRANSFER LINE" := TRUE;
   ELSE
       "TRANSFER DB".BIT."MFG TO STORAGE-3 WITH INLINE HOMO"."PFBV-59 TANK OUTLET VALVE" := FALSE;
       "TRANSFER DB".BIT."MFG TO STORAGE-3 WITH INLINE HOMO"."PBV-114 TANK OUTLET TO INLINE HOMOGENIZER LINE" := FALSE;
       "TRANSFER DB".BIT."MFG TO STORAGE-3 WITH INLINE HOMO"."PBV-110 INLINE HOMOGENIZER TO INLET LINE" := FALSE;
       "TRANSFER DB".BIT."MFG TO STORAGE-3 WITH INLINE HOMO"."PAV-56 INLINE HOMO. SEAL COOLING INLET" := FALSE;
       "TRANSFER DB".BIT."MFG TO STORAGE-3 WITH INLINE HOMO"."INLINE 1 HOMOGENIZER MOTOR1 RUN" := FALSE;
       "TRANSFER DB".BIT."MFG TO STORAGE-3 WITH INLINE HOMO"."PBV-109 HOMO. RECIRCULATION INLET" := FALSE;
       "TRANSFER DB".BIT."MFG TO STORAGE-3 WITH INLINE HOMO"."PBV-117 MFG TO STORAGE – 3 TRANSFER LINE" := FALSE;
       ;
   END_IF;
END_REGION

REGION Network 73: LOAD CELL_CUTOFF
   RUNG wire#powerrail
      { S7_Templates := "SrcType := Int" } NE_Contact(in1 := "MODE SELECTION DB"."MODE BUFF", in2 := 0)
      { S7_Templates := "SrcType := Int" } EQ_Contact(in1 := "TRANSFER DB".BUFF."MFG TO STORAGE-3 WITH INLINE HOMO", in2 := 2)
      I_Contact( "TRANSFER DB".PAUSE."MFG TO STORAGE-3 WITH INLINE HOMO" )
      { S7_Templates := "SrcType := Int" } NE_Contact(in1 := "CONTINUE DB"."SYRUP MFG PROCESS ERROR", in2 := 1)
      { S7_Templates := "SrcType := Int" } EQ_Contact(in1 := "LEVEL BUFF"."SYRUP MFG_LOAD CELL", in2 := 1)
      Move(in := 3, out1 => "TRANSFER DB".BUFF."MFG TO STORAGE-3 WITH INLINE HOMO")
   END_RUNG
   // the same network as SCL:
   IF ("MODE SELECTION DB"."MODE BUFF" <> 0) AND ("TRANSFER DB".BUFF."MFG TO STORAGE-3 WITH INLINE HOMO" = 2) AND NOT "TRANSFER DB".PAUSE."MFG TO STORAGE-3 WITH INLINE HOMO" AND ("CONTINUE DB"."SYRUP MFG PROCESS ERROR" <> 1) AND ("LEVEL BUFF"."SYRUP MFG_LOAD CELL" = 1) THEN
       "TRANSFER DB".BUFF."MFG TO STORAGE-3 WITH INLINE HOMO" := 3;
   END_IF;
END_REGION

REGION Network 74: PROCESS OVER & STOP
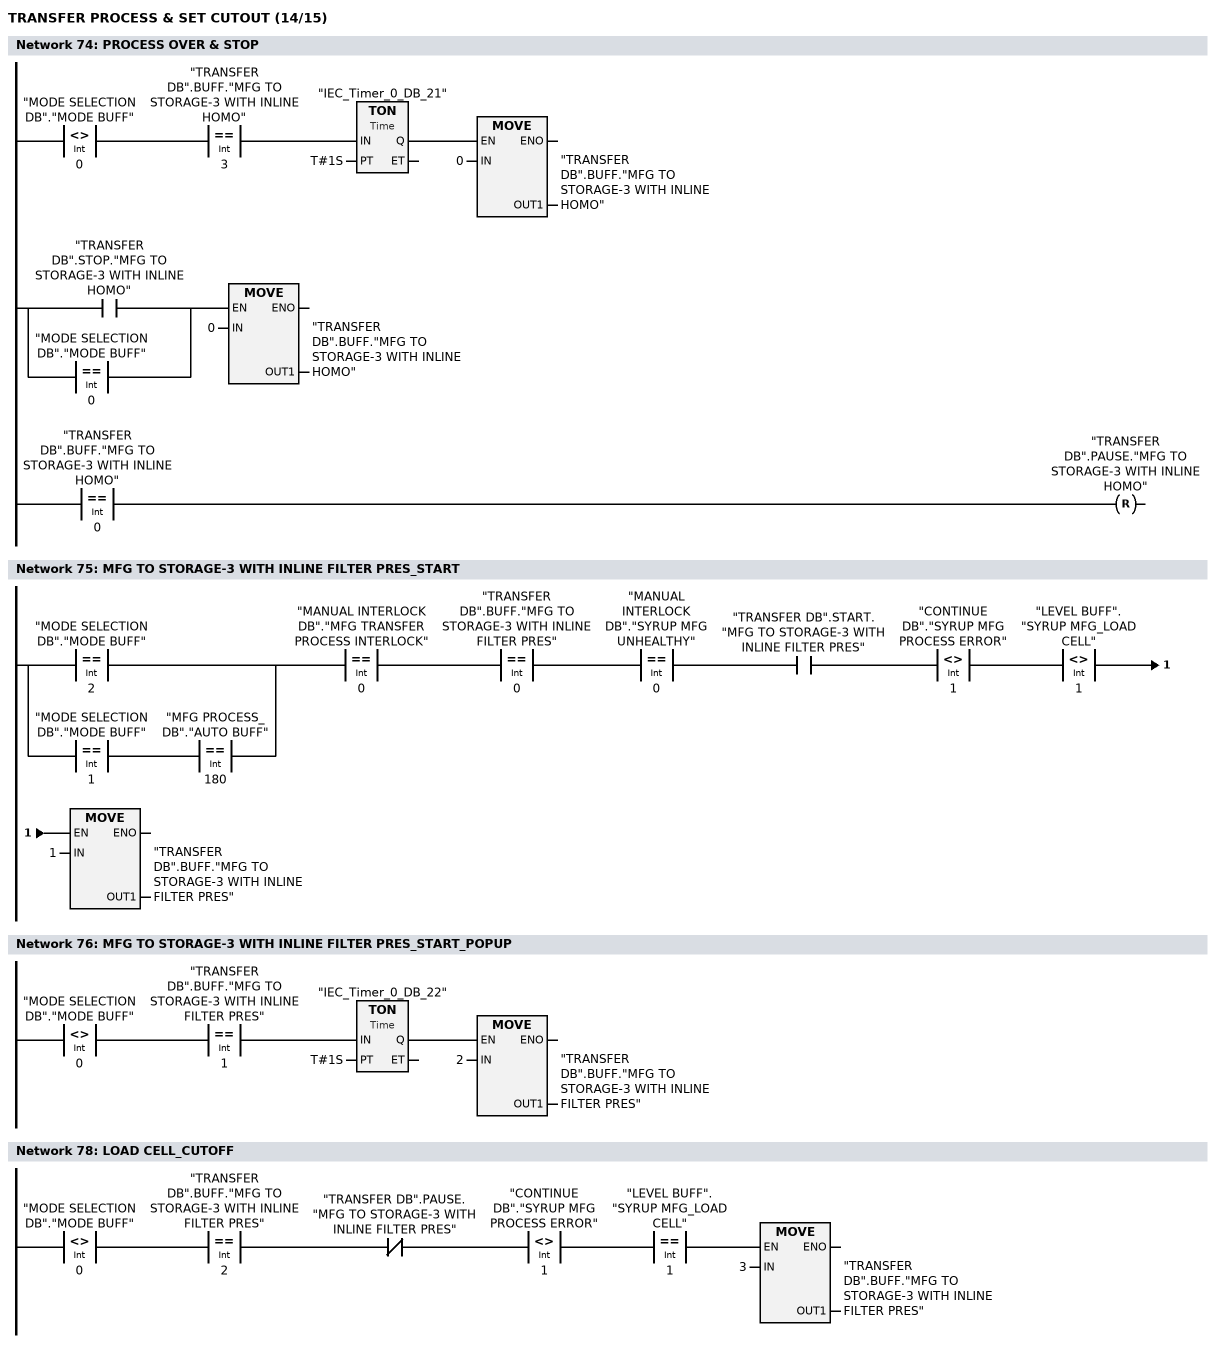
   RUNG wire#powerrail
      { S7_Templates := "SrcType := Int" } NE_Contact(in1 := "MODE SELECTION DB"."MODE BUFF", in2 := 0)
      { S7_Templates := "SrcType := Int" } EQ_Contact(in1 := "TRANSFER DB".BUFF."MFG TO STORAGE-3 WITH INLINE HOMO", in2 := 3)
      { S7_Templates := "time_type := Time" } "IEC_Timer_0_DB_21".TON(pt := T#1S, et =>)
      Move(in := 0, out1 => "TRANSFER DB".BUFF."MFG TO STORAGE-3 WITH INLINE HOMO")
   END_RUNG
   RUNG wire#powerrail
      Contact( "TRANSFER DB".STOP."MFG TO STORAGE-3 WITH INLINE HOMO" )
      wire#w1
      Move(in := 0, out1 => "TRANSFER DB".BUFF."MFG TO STORAGE-3 WITH INLINE HOMO")
   END_RUNG
   RUNG wire#powerrail
      { S7_Templates := "SrcType := Int" } EQ_Contact(in1 := "MODE SELECTION DB"."MODE BUFF", in2 := 0)
   END_RUNG wire#w1
   RUNG wire#powerrail
      { S7_Templates := "SrcType := Int" } EQ_Contact(in1 := "TRANSFER DB".BUFF."MFG TO STORAGE-3 WITH INLINE HOMO", in2 := 0)
      R_Coil( "TRANSFER DB".PAUSE."MFG TO STORAGE-3 WITH INLINE HOMO" )
   END_RUNG
   // the same network as SCL:
   "IEC_Timer_0_DB_21".TON(IN := ("MODE SELECTION DB"."MODE BUFF" <> 0) AND ("TRANSFER DB".BUFF."MFG TO STORAGE-3 WITH INLINE HOMO" = 3),
                           PT := T#1S);
   IF "IEC_Timer_0_DB_21".Q THEN "TRANSFER DB".BUFF."MFG TO STORAGE-3 WITH INLINE HOMO" := 0; END_IF;
   IF "TRANSFER DB".STOP."MFG TO STORAGE-3 WITH INLINE HOMO" OR ("MODE SELECTION DB"."MODE BUFF" = 0) THEN
       "TRANSFER DB".BUFF."MFG TO STORAGE-3 WITH INLINE HOMO" := 0;
   END_IF;
   IF "TRANSFER DB".BUFF."MFG TO STORAGE-3 WITH INLINE HOMO" = 0 THEN
       "TRANSFER DB".PAUSE."MFG TO STORAGE-3 WITH INLINE HOMO" := FALSE;
   END_IF;
END_REGION

REGION Network 75: MFG TO STORAGE-3 WITH INLINE FILTER PRES_START
   RUNG wire#powerrail
      { S7_Templates := "SrcType := Int" } EQ_Contact(in1 := "MODE SELECTION DB"."MODE BUFF", in2 := 2)
      wire#w1
      { S7_Templates := "SrcType := Int" } EQ_Contact(in1 := "MANUAL INTERLOCK DB"."MFG TRANSFER PROCESS INTERLOCK", in2 := 0)
      { S7_Templates := "SrcType := Int" } EQ_Contact(in1 := "TRANSFER DB".BUFF."MFG TO STORAGE-3 WITH INLINE FILTER PRES", in2 := 0)
      { S7_Templates := "SrcType := Int" } EQ_Contact(in1 := "MANUAL INTERLOCK DB"."SYRUP MFG UNHEALTHY", in2 := 0)
      Contact( "TRANSFER DB".START."MFG TO STORAGE-3 WITH INLINE FILTER PRES" )
      { S7_Templates := "SrcType := Int" } NE_Contact(in1 := "CONTINUE DB"."SYRUP MFG PROCESS ERROR", in2 := 1)
      { S7_Templates := "SrcType := Int" } NE_Contact(in1 := "LEVEL BUFF"."SYRUP MFG_LOAD CELL", in2 := 1)
      Move(in := 1, out1 => "TRANSFER DB".BUFF."MFG TO STORAGE-3 WITH INLINE FILTER PRES")
   END_RUNG
   RUNG wire#powerrail
      { S7_Templates := "SrcType := Int" } EQ_Contact(in1 := "MODE SELECTION DB"."MODE BUFF", in2 := 1)
      { S7_Templates := "SrcType := Int" } EQ_Contact(in1 := "MFG PROCESS_DB"."AUTO BUFF", in2 := 180)
   END_RUNG wire#w1
   // the same network as SCL:
   IF (("MODE SELECTION DB"."MODE BUFF" = 2) OR (("MODE SELECTION DB"."MODE BUFF" = 1) AND ("MFG PROCESS_DB"."AUTO BUFF" = 180))) AND ("MANUAL INTERLOCK DB"."MFG TRANSFER PROCESS INTERLOCK" = 0) AND ("TRANSFER DB".BUFF."MFG TO STORAGE-3 WITH INLINE FILTER PRES" = 0) AND ("MANUAL INTERLOCK DB"."SYRUP MFG UNHEALTHY" = 0) AND "TRANSFER DB".START."MFG TO STORAGE-3 WITH INLINE FILTER PRES" AND ("CONTINUE DB"."SYRUP MFG PROCESS ERROR" <> 1) AND ("LEVEL BUFF"."SYRUP MFG_LOAD CELL" <> 1) THEN
       "TRANSFER DB".BUFF."MFG TO STORAGE-3 WITH INLINE FILTER PRES" := 1;
   END_IF;
END_REGION

REGION Network 76: MFG TO STORAGE-3 WITH INLINE FILTER PRES_START_POPUP
   RUNG wire#powerrail
      { S7_Templates := "SrcType := Int" } NE_Contact(in1 := "MODE SELECTION DB"."MODE BUFF", in2 := 0)
      { S7_Templates := "SrcType := Int" } EQ_Contact(in1 := "TRANSFER DB".BUFF."MFG TO STORAGE-3 WITH INLINE FILTER PRES", in2 := 1)
      { S7_Templates := "time_type := Time" } "IEC_Timer_0_DB_22".TON(pt := T#1S, et =>)
      Move(in := 2, out1 => "TRANSFER DB".BUFF."MFG TO STORAGE-3 WITH INLINE FILTER PRES")
   END_RUNG
   // the same network as SCL:
   "IEC_Timer_0_DB_22".TON(IN := ("MODE SELECTION DB"."MODE BUFF" <> 0) AND ("TRANSFER DB".BUFF."MFG TO STORAGE-3 WITH INLINE FILTER PRES" = 1),
                           PT := T#1S);
   IF "IEC_Timer_0_DB_22".Q THEN "TRANSFER DB".BUFF."MFG TO STORAGE-3 WITH INLINE FILTER PRES" := 2; END_IF;
END_REGION

REGION Network 77 (SCL): OPENVALVE
   IF ("MODE SELECTION DB"."MODE BUFF" <> 0 AND "TRANSFER DB".BUFF."MFG TO STORAGE-3 WITH INLINE FILTER PRES" = 2
       AND NOT "TRANSFER DB".PAUSE."MFG TO STORAGE-3 WITH INLINE FILTER PRES"
       AND "CONTINUE DB"."SYRUP MFG PROCESS ERROR" = 0 AND "LEVEL BUFF"."SYRUP MFG_LOAD CELL" = 0)
       OR ("MODE SELECTION DB"."MODE BUFF"=1 AND "MFG PROCESS_DB"."AUTO BUFF"=0
       AND "MFG TRANSFER CYCLE DB".TRANSFER."TRANSFER BUFF"."MFG TO STORAGE-3 WITH INLINE FILTER PRES"=10 AND "CONTINUE DB"."SYRUP MFG PROCESS ERROR" <>1
       AND "MFG TRANSFER CYCLE DB".TRANSFER.SELECT."SELECT BUFF"=6)
   THEN
       "TRANSFER DB".BIT."MFG TO STORAGE-3 WITH INLINE FILTER PRES"."PFBV-59 TANK OUTLET VALVE" := TRUE;
       "TRANSFER DB".BIT."MFG TO STORAGE-3 WITH INLINE FILTER PRES"."PBV-114 TANK OUTLET TO INLINE HOMOGENIZER LINE" := TRUE;
       "TRANSFER DB".BIT."MFG TO STORAGE-3 WITH INLINE FILTER PRES"."PBV-108 INLINE HOMOGENIZER TO FILTER PRESS INLET LINE" := TRUE;
       "TRANSFER DB".BIT."MFG TO STORAGE-3 WITH INLINE FILTER PRES"."FILTER PRESS MOTOR 1 RUN" := TRUE;
       "TRANSFER DB".BIT."MFG TO STORAGE-3 WITH INLINE FILTER PRES"."PBV-118 FILTER PRESS INLET" := TRUE;
       "TRANSFER DB".BIT."MFG TO STORAGE-3 WITH INLINE FILTER PRES"."PBV-111 FILTER PRESS OUTLER VALVE" := TRUE;
       "TRANSFER DB".BIT."MFG TO STORAGE-3 WITH INLINE FILTER PRES"."PBV-112 FILTER PRESS TO TRANSFER LINE" := TRUE;
       "TRANSFER DB".BIT."MFG TO STORAGE-3 WITH INLINE FILTER PRES"."PBV-117 MFG TO STORAGE – 3 TRANSFER LINE" := TRUE;
   ELSE
       "TRANSFER DB".BIT."MFG TO STORAGE-3 WITH INLINE FILTER PRES"."PFBV-59 TANK OUTLET VALVE" := FALSE;
       "TRANSFER DB".BIT."MFG TO STORAGE-3 WITH INLINE FILTER PRES"."PBV-114 TANK OUTLET TO INLINE HOMOGENIZER LINE" := FALSE;
       "TRANSFER DB".BIT."MFG TO STORAGE-3 WITH INLINE FILTER PRES"."PBV-108 INLINE HOMOGENIZER TO FILTER PRESS INLET LINE" := FALSE;
       "TRANSFER DB".BIT."MFG TO STORAGE-3 WITH INLINE FILTER PRES"."FILTER PRESS MOTOR 1 RUN" := FALSE;
       "TRANSFER DB".BIT."MFG TO STORAGE-3 WITH INLINE FILTER PRES"."PBV-118 FILTER PRESS INLET" := FALSE;
       "TRANSFER DB".BIT."MFG TO STORAGE-3 WITH INLINE FILTER PRES"."PBV-111 FILTER PRESS OUTLER VALVE" := FALSE;
       "TRANSFER DB".BIT."MFG TO STORAGE-3 WITH INLINE FILTER PRES"."PBV-112 FILTER PRESS TO TRANSFER LINE" := FALSE;
       "TRANSFER DB".BIT."MFG TO STORAGE-3 WITH INLINE FILTER PRES"."PBV-117 MFG TO STORAGE – 3 TRANSFER LINE" := FALSE;
       ;
   END_IF;
END_REGION

REGION Network 78: LOAD CELL_CUTOFF
   RUNG wire#powerrail
      { S7_Templates := "SrcType := Int" } NE_Contact(in1 := "MODE SELECTION DB"."MODE BUFF", in2 := 0)
      { S7_Templates := "SrcType := Int" } EQ_Contact(in1 := "TRANSFER DB".BUFF."MFG TO STORAGE-3 WITH INLINE FILTER PRES", in2 := 2)
      I_Contact( "TRANSFER DB".PAUSE."MFG TO STORAGE-3 WITH INLINE FILTER PRES" )
      { S7_Templates := "SrcType := Int" } NE_Contact(in1 := "CONTINUE DB"."SYRUP MFG PROCESS ERROR", in2 := 1)
      { S7_Templates := "SrcType := Int" } EQ_Contact(in1 := "LEVEL BUFF"."SYRUP MFG_LOAD CELL", in2 := 1)
      Move(in := 3, out1 => "TRANSFER DB".BUFF."MFG TO STORAGE-3 WITH INLINE FILTER PRES")
   END_RUNG
   // the same network as SCL:
   IF ("MODE SELECTION DB"."MODE BUFF" <> 0) AND ("TRANSFER DB".BUFF."MFG TO STORAGE-3 WITH INLINE FILTER PRES" = 2) AND NOT "TRANSFER DB".PAUSE."MFG TO STORAGE-3 WITH INLINE FILTER PRES" AND ("CONTINUE DB"."SYRUP MFG PROCESS ERROR" <> 1) AND ("LEVEL BUFF"."SYRUP MFG_LOAD CELL" = 1) THEN
       "TRANSFER DB".BUFF."MFG TO STORAGE-3 WITH INLINE FILTER PRES" := 3;
   END_IF;
END_REGION

REGION Network 79: PROCESS OVER & STOP
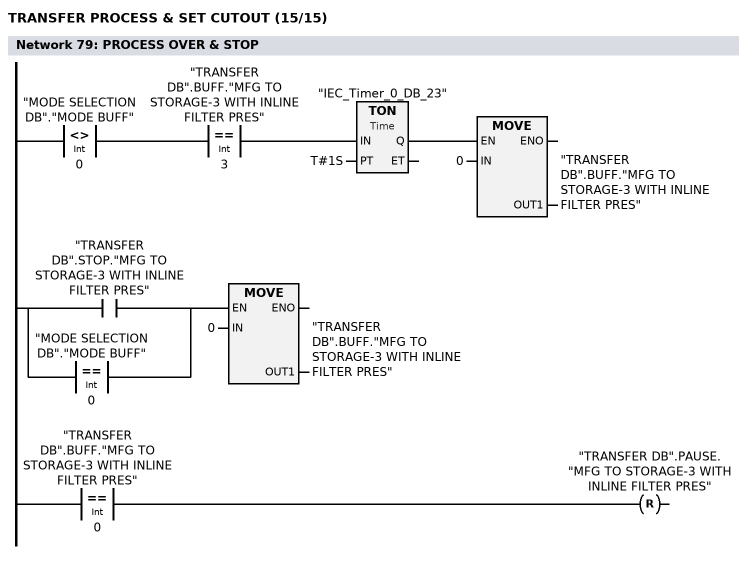
   RUNG wire#powerrail
      { S7_Templates := "SrcType := Int" } NE_Contact(in1 := "MODE SELECTION DB"."MODE BUFF", in2 := 0)
      { S7_Templates := "SrcType := Int" } EQ_Contact(in1 := "TRANSFER DB".BUFF."MFG TO STORAGE-3 WITH INLINE FILTER PRES", in2 := 3)
      { S7_Templates := "time_type := Time" } "IEC_Timer_0_DB_23".TON(pt := T#1S, et =>)
      Move(in := 0, out1 => "TRANSFER DB".BUFF."MFG TO STORAGE-3 WITH INLINE FILTER PRES")
   END_RUNG
   RUNG wire#powerrail
      Contact( "TRANSFER DB".STOP."MFG TO STORAGE-3 WITH INLINE FILTER PRES" )
      wire#w1
      Move(in := 0, out1 => "TRANSFER DB".BUFF."MFG TO STORAGE-3 WITH INLINE FILTER PRES")
   END_RUNG
   RUNG wire#powerrail
      { S7_Templates := "SrcType := Int" } EQ_Contact(in1 := "MODE SELECTION DB"."MODE BUFF", in2 := 0)
   END_RUNG wire#w1
   RUNG wire#powerrail
      { S7_Templates := "SrcType := Int" } EQ_Contact(in1 := "TRANSFER DB".BUFF."MFG TO STORAGE-3 WITH INLINE FILTER PRES", in2 := 0)
      R_Coil( "TRANSFER DB".PAUSE."MFG TO STORAGE-3 WITH INLINE FILTER PRES" )
   END_RUNG
   // the same network as SCL:
   "IEC_Timer_0_DB_23".TON(IN := ("MODE SELECTION DB"."MODE BUFF" <> 0) AND ("TRANSFER DB".BUFF."MFG TO STORAGE-3 WITH INLINE FILTER PRES" = 3),
                           PT := T#1S);
   IF "IEC_Timer_0_DB_23".Q THEN "TRANSFER DB".BUFF."MFG TO STORAGE-3 WITH INLINE FILTER PRES" := 0; END_IF;
   IF "TRANSFER DB".STOP."MFG TO STORAGE-3 WITH INLINE FILTER PRES" OR ("MODE SELECTION DB"."MODE BUFF" = 0) THEN
       "TRANSFER DB".BUFF."MFG TO STORAGE-3 WITH INLINE FILTER PRES" := 0;
   END_IF;
   IF "TRANSFER DB".BUFF."MFG TO STORAGE-3 WITH INLINE FILTER PRES" = 0 THEN
       "TRANSFER DB".PAUSE."MFG TO STORAGE-3 WITH INLINE FILTER PRES" := FALSE;
   END_IF;
END_REGION
END_FUNCTION

FUNCTION "TRANSFER SUBOUTPUT" : Void   // FC13, LAD
{ S7_Optimized_Access := 'TRUE' }
// stored: SetENOAutomatically false
BEGIN

REGION Network 1: SYRUP MFG VESSEL BOTTOM STERROR RUN
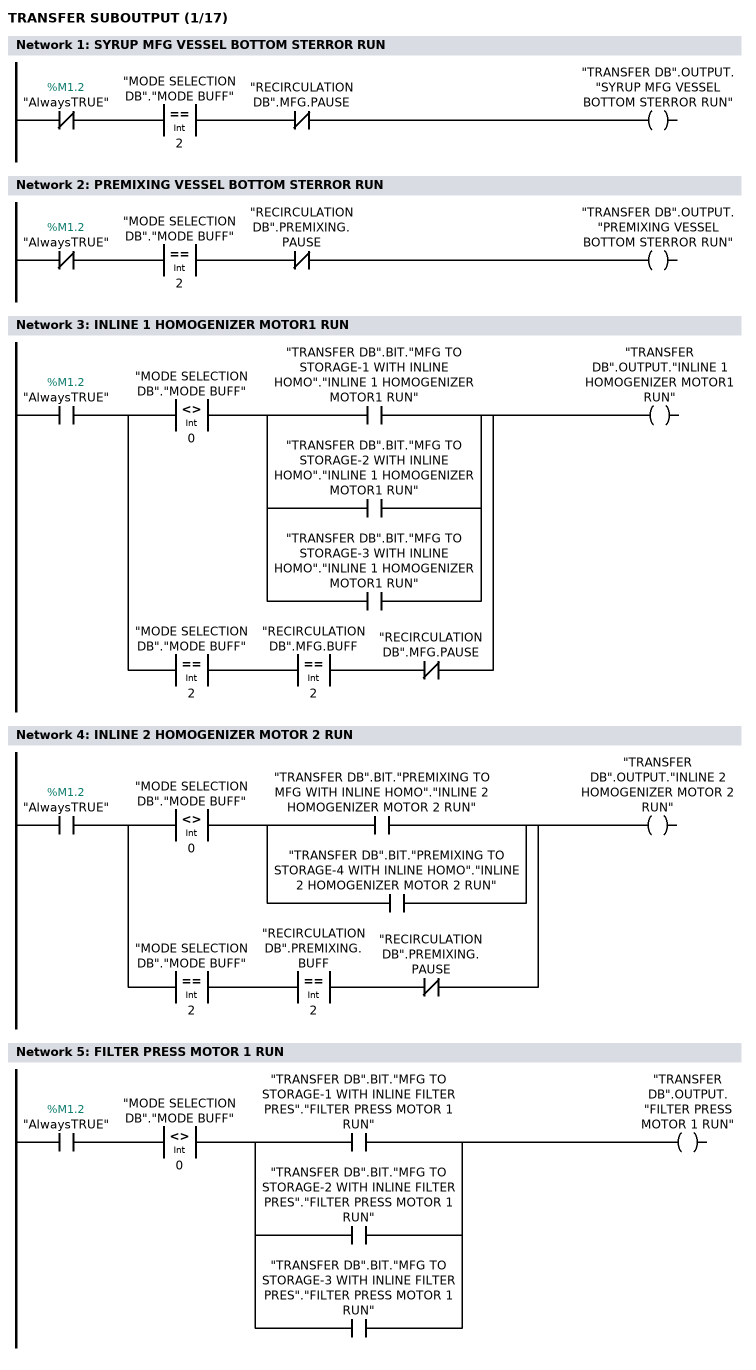
   RUNG wire#powerrail
      I_Contact( "AlwaysTRUE" )
      { S7_Templates := "SrcType := Int" } EQ_Contact(in1 := "MODE SELECTION DB"."MODE BUFF", in2 := 2)
      I_Contact( "RECIRCULATION DB".MFG.PAUSE )
      Coil( "TRANSFER DB".OUTPUT."SYRUP MFG VESSEL BOTTOM STERROR RUN" )
   END_RUNG
   // the same network as SCL:
   "TRANSFER DB".OUTPUT."SYRUP MFG VESSEL BOTTOM STERROR RUN" := NOT "AlwaysTRUE" AND ("MODE SELECTION DB"."MODE BUFF" = 2) AND NOT "RECIRCULATION DB".MFG.PAUSE;
END_REGION

REGION Network 2: PREMIXING VESSEL BOTTOM STERROR RUN
   RUNG wire#powerrail
      I_Contact( "AlwaysTRUE" )
      { S7_Templates := "SrcType := Int" } EQ_Contact(in1 := "MODE SELECTION DB"."MODE BUFF", in2 := 2)
      I_Contact( "RECIRCULATION DB".PREMIXING.PAUSE )
      Coil( "TRANSFER DB".OUTPUT."PREMIXING VESSEL BOTTOM STERROR RUN" )
   END_RUNG
   // the same network as SCL:
   "TRANSFER DB".OUTPUT."PREMIXING VESSEL BOTTOM STERROR RUN" := NOT "AlwaysTRUE" AND ("MODE SELECTION DB"."MODE BUFF" = 2) AND NOT "RECIRCULATION DB".PREMIXING.PAUSE;
END_REGION

REGION Network 3: INLINE 1 HOMOGENIZER MOTOR1 RUN
   RUNG wire#powerrail
      Contact( "AlwaysTRUE" )
      wire#w1
      { S7_Templates := "SrcType := Int" } NE_Contact(in1 := "MODE SELECTION DB"."MODE BUFF", in2 := 0)
      wire#w2
      Contact( "TRANSFER DB".BIT."MFG TO STORAGE-1 WITH INLINE HOMO"."INLINE 1 HOMOGENIZER MOTOR1 RUN" )
      wire#w3
      Coil( "TRANSFER DB".OUTPUT."INLINE 1 HOMOGENIZER MOTOR1 RUN" )
   END_RUNG
   RUNG wire#w2
      Contact( "TRANSFER DB".BIT."MFG TO STORAGE-2 WITH INLINE HOMO"."INLINE 1 HOMOGENIZER MOTOR1 RUN" )
   END_RUNG wire#w3
   RUNG wire#w2
      Contact( "TRANSFER DB".BIT."MFG TO STORAGE-3 WITH INLINE HOMO"."INLINE 1 HOMOGENIZER MOTOR1 RUN" )
   END_RUNG wire#w3
   RUNG wire#w1
      { S7_Templates := "SrcType := Int" } EQ_Contact(in1 := "MODE SELECTION DB"."MODE BUFF", in2 := 2)
      { S7_Templates := "SrcType := Int" } EQ_Contact(in1 := "RECIRCULATION DB".MFG.BUFF, in2 := 2)
      I_Contact( "RECIRCULATION DB".MFG.PAUSE )
   END_RUNG wire#w3
   // the same network as SCL:
   "TRANSFER DB".OUTPUT."INLINE 1 HOMOGENIZER MOTOR1 RUN" := "AlwaysTRUE" AND ((("MODE SELECTION DB"."MODE BUFF" <> 0) AND ("TRANSFER DB".BIT."MFG TO STORAGE-1 WITH INLINE HOMO"."INLINE 1 HOMOGENIZER MOTOR1 RUN" OR "TRANSFER DB".BIT."MFG TO STORAGE-2 WITH INLINE HOMO"."INLINE 1 HOMOGENIZER MOTOR1 RUN" OR "TRANSFER DB".BIT."MFG TO STORAGE-3 WITH INLINE HOMO"."INLINE 1 HOMOGENIZER MOTOR1 RUN")) OR (("MODE SELECTION DB"."MODE BUFF" = 2) AND ("RECIRCULATION DB".MFG.BUFF = 2) AND NOT "RECIRCULATION DB".MFG.PAUSE));
END_REGION

REGION Network 4: INLINE 2 HOMOGENIZER MOTOR 2 RUN
   RUNG wire#powerrail
      Contact( "AlwaysTRUE" )
      wire#w1
      { S7_Templates := "SrcType := Int" } NE_Contact(in1 := "MODE SELECTION DB"."MODE BUFF", in2 := 0)
      wire#w2
      Contact( "TRANSFER DB".BIT."PREMIXING TO MFG WITH INLINE HOMO"."INLINE 2 HOMOGENIZER MOTOR 2 RUN" )
      wire#w3
      Coil( "TRANSFER DB".OUTPUT."INLINE 2 HOMOGENIZER MOTOR 2 RUN" )
   END_RUNG
   RUNG wire#w2
      Contact( "TRANSFER DB".BIT."PREMIXING TO STORAGE-4 WITH INLINE HOMO"."INLINE 2 HOMOGENIZER MOTOR 2 RUN" )
   END_RUNG wire#w3
   RUNG wire#w1
      { S7_Templates := "SrcType := Int" } EQ_Contact(in1 := "MODE SELECTION DB"."MODE BUFF", in2 := 2)
      { S7_Templates := "SrcType := Int" } EQ_Contact(in1 := "RECIRCULATION DB".PREMIXING.BUFF, in2 := 2)
      I_Contact( "RECIRCULATION DB".PREMIXING.PAUSE )
   END_RUNG wire#w3
   // the same network as SCL:
   "TRANSFER DB".OUTPUT."INLINE 2 HOMOGENIZER MOTOR 2 RUN" := "AlwaysTRUE" AND ((("MODE SELECTION DB"."MODE BUFF" <> 0) AND ("TRANSFER DB".BIT."PREMIXING TO MFG WITH INLINE HOMO"."INLINE 2 HOMOGENIZER MOTOR 2 RUN" OR "TRANSFER DB".BIT."PREMIXING TO STORAGE-4 WITH INLINE HOMO"."INLINE 2 HOMOGENIZER MOTOR 2 RUN")) OR (("MODE SELECTION DB"."MODE BUFF" = 2) AND ("RECIRCULATION DB".PREMIXING.BUFF = 2) AND NOT "RECIRCULATION DB".PREMIXING.PAUSE));
END_REGION

REGION Network 5: FILTER PRESS MOTOR 1 RUN
   RUNG wire#powerrail
      Contact( "AlwaysTRUE" )
      { S7_Templates := "SrcType := Int" } NE_Contact(in1 := "MODE SELECTION DB"."MODE BUFF", in2 := 0)
      wire#w1
      Contact( "TRANSFER DB".BIT."MFG TO STORAGE-1 WITH INLINE FILTER PRES"."FILTER PRESS MOTOR 1 RUN" )
      wire#w2
      Coil( "TRANSFER DB".OUTPUT."FILTER PRESS MOTOR 1 RUN" )
   END_RUNG
   RUNG wire#w1
      Contact( "TRANSFER DB".BIT."MFG TO STORAGE-2 WITH INLINE FILTER PRES"."FILTER PRESS MOTOR 1 RUN" )
   END_RUNG wire#w2
   RUNG wire#w1
      Contact( "TRANSFER DB".BIT."MFG TO STORAGE-3 WITH INLINE FILTER PRES"."FILTER PRESS MOTOR 1 RUN" )
   END_RUNG wire#w2
   // the same network as SCL:
   "TRANSFER DB".OUTPUT."FILTER PRESS MOTOR 1 RUN" := "AlwaysTRUE" AND ("MODE SELECTION DB"."MODE BUFF" <> 0) AND ("TRANSFER DB".BIT."MFG TO STORAGE-1 WITH INLINE FILTER PRES"."FILTER PRESS MOTOR 1 RUN" OR "TRANSFER DB".BIT."MFG TO STORAGE-2 WITH INLINE FILTER PRES"."FILTER PRESS MOTOR 1 RUN" OR "TRANSFER DB".BIT."MFG TO STORAGE-3 WITH INLINE FILTER PRES"."FILTER PRESS MOTOR 1 RUN");
END_REGION

REGION Network 6: FILTER PRESS MOTOR 2 RUN
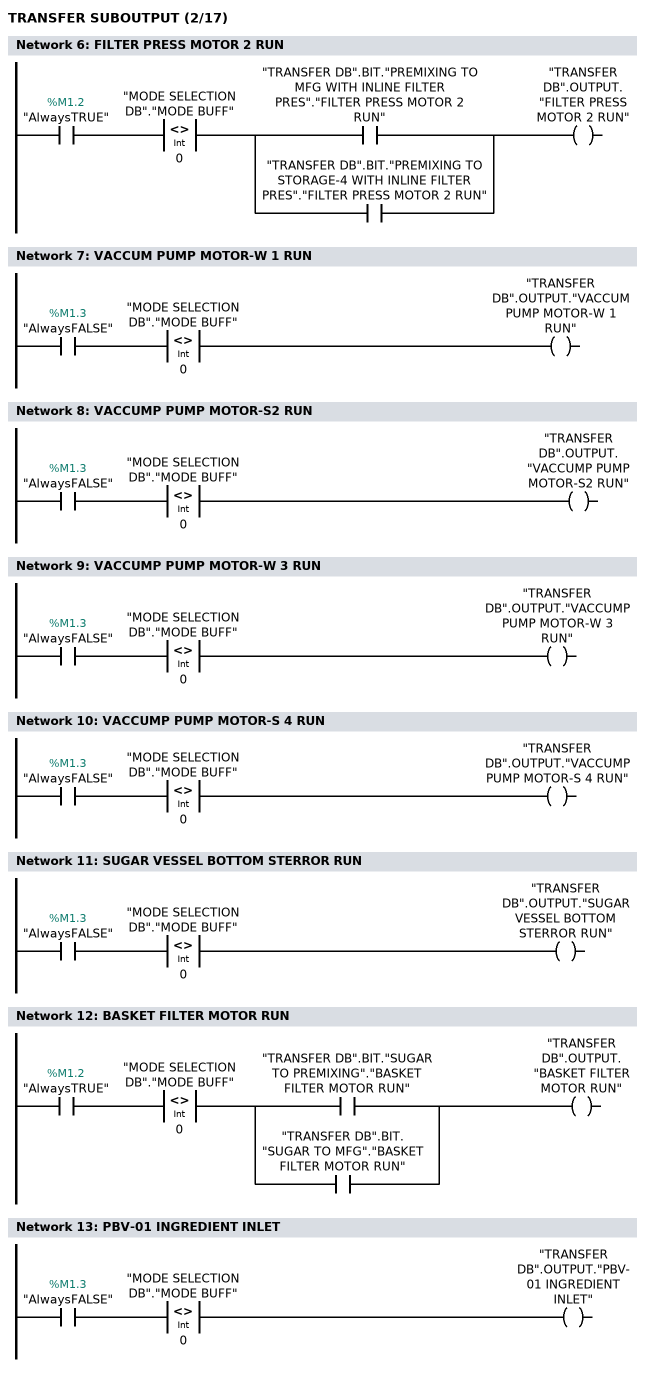
   RUNG wire#powerrail
      Contact( "AlwaysTRUE" )
      { S7_Templates := "SrcType := Int" } NE_Contact(in1 := "MODE SELECTION DB"."MODE BUFF", in2 := 0)
      wire#w1
      Contact( "TRANSFER DB".BIT."PREMIXING TO MFG WITH INLINE FILTER PRES"."FILTER PRESS MOTOR 2 RUN" )
      wire#w2
      Coil( "TRANSFER DB".OUTPUT."FILTER PRESS MOTOR 2 RUN" )
   END_RUNG
   RUNG wire#w1
      Contact( "TRANSFER DB".BIT."PREMIXING TO STORAGE-4 WITH INLINE FILTER PRES"."FILTER PRESS MOTOR 2 RUN" )
   END_RUNG wire#w2
   // the same network as SCL:
   "TRANSFER DB".OUTPUT."FILTER PRESS MOTOR 2 RUN" := "AlwaysTRUE" AND ("MODE SELECTION DB"."MODE BUFF" <> 0) AND ("TRANSFER DB".BIT."PREMIXING TO MFG WITH INLINE FILTER PRES"."FILTER PRESS MOTOR 2 RUN" OR "TRANSFER DB".BIT."PREMIXING TO STORAGE-4 WITH INLINE FILTER PRES"."FILTER PRESS MOTOR 2 RUN");
END_REGION

REGION Network 7: VACCUM PUMP MOTOR-W 1 RUN
   RUNG wire#powerrail
      Contact( "AlwaysFALSE" )
      { S7_Templates := "SrcType := Int" } NE_Contact(in1 := "MODE SELECTION DB"."MODE BUFF", in2 := 0)
      Coil( "TRANSFER DB".OUTPUT."VACCUM PUMP MOTOR-W 1 RUN" )
   END_RUNG
   // the same network as SCL:
   "TRANSFER DB".OUTPUT."VACCUM PUMP MOTOR-W 1 RUN" := "AlwaysFALSE" AND ("MODE SELECTION DB"."MODE BUFF" <> 0);
END_REGION

REGION Network 8: VACCUMP PUMP MOTOR-S2 RUN
   RUNG wire#powerrail
      Contact( "AlwaysFALSE" )
      { S7_Templates := "SrcType := Int" } NE_Contact(in1 := "MODE SELECTION DB"."MODE BUFF", in2 := 0)
      Coil( "TRANSFER DB".OUTPUT."VACCUMP PUMP MOTOR-S2 RUN" )
   END_RUNG
   // the same network as SCL:
   "TRANSFER DB".OUTPUT."VACCUMP PUMP MOTOR-S2 RUN" := "AlwaysFALSE" AND ("MODE SELECTION DB"."MODE BUFF" <> 0);
END_REGION

REGION Network 9: VACCUMP PUMP MOTOR-W 3 RUN
   RUNG wire#powerrail
      Contact( "AlwaysFALSE" )
      { S7_Templates := "SrcType := Int" } NE_Contact(in1 := "MODE SELECTION DB"."MODE BUFF", in2 := 0)
      Coil( "TRANSFER DB".OUTPUT."VACCUMP PUMP MOTOR-W 3 RUN" )
   END_RUNG
   // the same network as SCL:
   "TRANSFER DB".OUTPUT."VACCUMP PUMP MOTOR-W 3 RUN" := "AlwaysFALSE" AND ("MODE SELECTION DB"."MODE BUFF" <> 0);
END_REGION

REGION Network 10: VACCUMP PUMP MOTOR-S 4 RUN
   RUNG wire#powerrail
      Contact( "AlwaysFALSE" )
      { S7_Templates := "SrcType := Int" } NE_Contact(in1 := "MODE SELECTION DB"."MODE BUFF", in2 := 0)
      Coil( "TRANSFER DB".OUTPUT."VACCUMP PUMP MOTOR-S 4 RUN" )
   END_RUNG
   // the same network as SCL:
   "TRANSFER DB".OUTPUT."VACCUMP PUMP MOTOR-S 4 RUN" := "AlwaysFALSE" AND ("MODE SELECTION DB"."MODE BUFF" <> 0);
END_REGION

REGION Network 11: SUGAR VESSEL BOTTOM STERROR RUN
   RUNG wire#powerrail
      Contact( "AlwaysFALSE" )
      { S7_Templates := "SrcType := Int" } NE_Contact(in1 := "MODE SELECTION DB"."MODE BUFF", in2 := 0)
      Coil( "TRANSFER DB".OUTPUT."SUGAR VESSEL BOTTOM STERROR RUN" )
   END_RUNG
   // the same network as SCL:
   "TRANSFER DB".OUTPUT."SUGAR VESSEL BOTTOM STERROR RUN" := "AlwaysFALSE" AND ("MODE SELECTION DB"."MODE BUFF" <> 0);
END_REGION

REGION Network 12: BASKET FILTER MOTOR RUN
   RUNG wire#powerrail
      Contact( "AlwaysTRUE" )
      { S7_Templates := "SrcType := Int" } NE_Contact(in1 := "MODE SELECTION DB"."MODE BUFF", in2 := 0)
      wire#w1
      Contact( "TRANSFER DB".BIT."SUGAR TO PREMIXING"."BASKET FILTER MOTOR RUN" )
      wire#w2
      Coil( "TRANSFER DB".OUTPUT."BASKET FILTER MOTOR RUN" )
   END_RUNG
   RUNG wire#w1
      Contact( "TRANSFER DB".BIT."SUGAR TO MFG"."BASKET FILTER MOTOR RUN" )
   END_RUNG wire#w2
   // the same network as SCL:
   "TRANSFER DB".OUTPUT."BASKET FILTER MOTOR RUN" := "AlwaysTRUE" AND ("MODE SELECTION DB"."MODE BUFF" <> 0) AND ("TRANSFER DB".BIT."SUGAR TO PREMIXING"."BASKET FILTER MOTOR RUN" OR "TRANSFER DB".BIT."SUGAR TO MFG"."BASKET FILTER MOTOR RUN");
END_REGION

REGION Network 13: PBV-01 INGREDIENT INLET
   RUNG wire#powerrail
      Contact( "AlwaysFALSE" )
      { S7_Templates := "SrcType := Int" } NE_Contact(in1 := "MODE SELECTION DB"."MODE BUFF", in2 := 0)
      Coil( "TRANSFER DB".OUTPUT."PBV-01 INGREDIENT INLET" )
   END_RUNG
   // the same network as SCL:
   "TRANSFER DB".OUTPUT."PBV-01 INGREDIENT INLET" := "AlwaysFALSE" AND ("MODE SELECTION DB"."MODE BUFF" <> 0);
END_REGION

REGION Network 14: PBV-02 CIP INLET (SPRAY BALL)
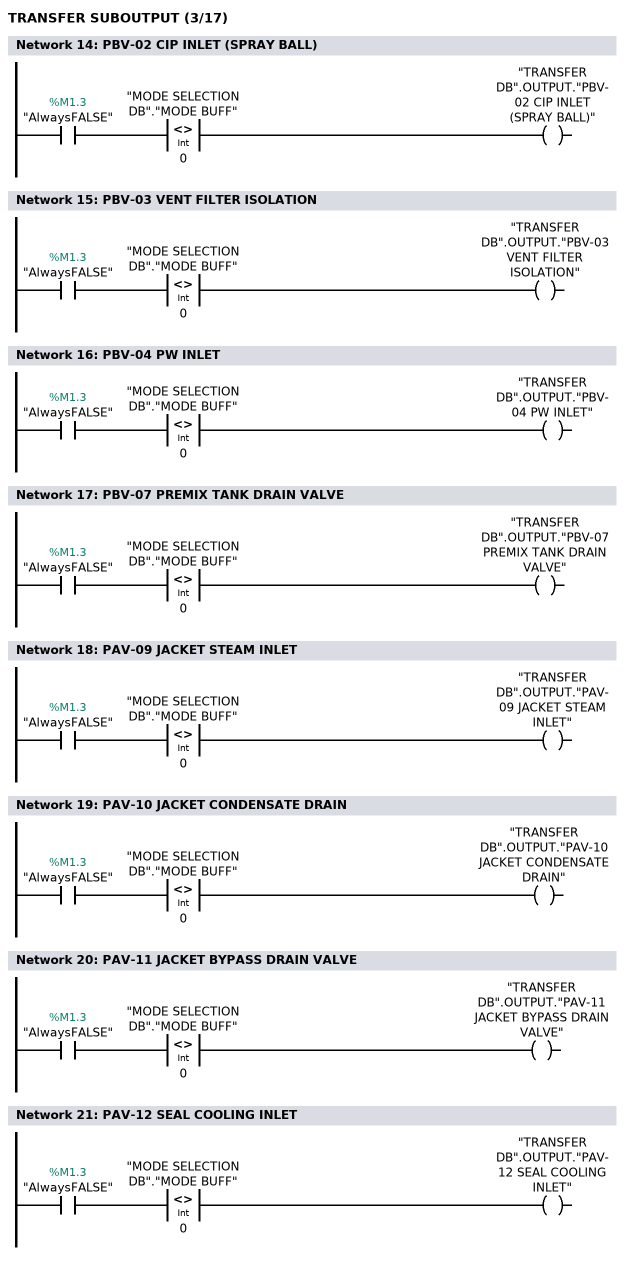
   RUNG wire#powerrail
      Contact( "AlwaysFALSE" )
      { S7_Templates := "SrcType := Int" } NE_Contact(in1 := "MODE SELECTION DB"."MODE BUFF", in2 := 0)
      Coil( "TRANSFER DB".OUTPUT."PBV-02 CIP INLET (SPRAY BALL)" )
   END_RUNG
   // the same network as SCL:
   "TRANSFER DB".OUTPUT."PBV-02 CIP INLET (SPRAY BALL)" := "AlwaysFALSE" AND ("MODE SELECTION DB"."MODE BUFF" <> 0);
END_REGION

REGION Network 15: PBV-03 VENT FILTER ISOLATION
   RUNG wire#powerrail
      Contact( "AlwaysFALSE" )
      { S7_Templates := "SrcType := Int" } NE_Contact(in1 := "MODE SELECTION DB"."MODE BUFF", in2 := 0)
      Coil( "TRANSFER DB".OUTPUT."PBV-03 VENT FILTER ISOLATION" )
   END_RUNG
   // the same network as SCL:
   "TRANSFER DB".OUTPUT."PBV-03 VENT FILTER ISOLATION" := "AlwaysFALSE" AND ("MODE SELECTION DB"."MODE BUFF" <> 0);
END_REGION

REGION Network 16: PBV-04 PW INLET
   RUNG wire#powerrail
      Contact( "AlwaysFALSE" )
      { S7_Templates := "SrcType := Int" } NE_Contact(in1 := "MODE SELECTION DB"."MODE BUFF", in2 := 0)
      Coil( "TRANSFER DB".OUTPUT."PBV-04 PW INLET" )
   END_RUNG
   // the same network as SCL:
   "TRANSFER DB".OUTPUT."PBV-04 PW INLET" := "AlwaysFALSE" AND ("MODE SELECTION DB"."MODE BUFF" <> 0);
END_REGION

REGION Network 17: PBV-07 PREMIX TANK DRAIN VALVE
   RUNG wire#powerrail
      Contact( "AlwaysFALSE" )
      { S7_Templates := "SrcType := Int" } NE_Contact(in1 := "MODE SELECTION DB"."MODE BUFF", in2 := 0)
      Coil( "TRANSFER DB".OUTPUT."PBV-07 PREMIX TANK DRAIN VALVE" )
   END_RUNG
   // the same network as SCL:
   "TRANSFER DB".OUTPUT."PBV-07 PREMIX TANK DRAIN VALVE" := "AlwaysFALSE" AND ("MODE SELECTION DB"."MODE BUFF" <> 0);
END_REGION

REGION Network 18: PAV-09 JACKET STEAM INLET
   RUNG wire#powerrail
      Contact( "AlwaysFALSE" )
      { S7_Templates := "SrcType := Int" } NE_Contact(in1 := "MODE SELECTION DB"."MODE BUFF", in2 := 0)
      Coil( "TRANSFER DB".OUTPUT."PAV-09 JACKET STEAM INLET" )
   END_RUNG
   // the same network as SCL:
   "TRANSFER DB".OUTPUT."PAV-09 JACKET STEAM INLET" := "AlwaysFALSE" AND ("MODE SELECTION DB"."MODE BUFF" <> 0);
END_REGION

REGION Network 19: PAV-10 JACKET CONDENSATE DRAIN
   RUNG wire#powerrail
      Contact( "AlwaysFALSE" )
      { S7_Templates := "SrcType := Int" } NE_Contact(in1 := "MODE SELECTION DB"."MODE BUFF", in2 := 0)
      Coil( "TRANSFER DB".OUTPUT."PAV-10 JACKET CONDENSATE DRAIN" )
   END_RUNG
   // the same network as SCL:
   "TRANSFER DB".OUTPUT."PAV-10 JACKET CONDENSATE DRAIN" := "AlwaysFALSE" AND ("MODE SELECTION DB"."MODE BUFF" <> 0);
END_REGION

REGION Network 20: PAV-11 JACKET BYPASS DRAIN VALVE
   RUNG wire#powerrail
      Contact( "AlwaysFALSE" )
      { S7_Templates := "SrcType := Int" } NE_Contact(in1 := "MODE SELECTION DB"."MODE BUFF", in2 := 0)
      Coil( "TRANSFER DB".OUTPUT."PAV-11 JACKET BYPASS DRAIN VALVE" )
   END_RUNG
   // the same network as SCL:
   "TRANSFER DB".OUTPUT."PAV-11 JACKET BYPASS DRAIN VALVE" := "AlwaysFALSE" AND ("MODE SELECTION DB"."MODE BUFF" <> 0);
END_REGION

REGION Network 21: PAV-12 SEAL COOLING INLET
   RUNG wire#powerrail
      Contact( "AlwaysFALSE" )
      { S7_Templates := "SrcType := Int" } NE_Contact(in1 := "MODE SELECTION DB"."MODE BUFF", in2 := 0)
      Coil( "TRANSFER DB".OUTPUT."PAV-12 SEAL COOLING INLET" )
   END_RUNG
   // the same network as SCL:
   "TRANSFER DB".OUTPUT."PAV-12 SEAL COOLING INLET" := "AlwaysFALSE" AND ("MODE SELECTION DB"."MODE BUFF" <> 0);
END_REGION

REGION Network 22: PAV-13 WATER COOLING INLET
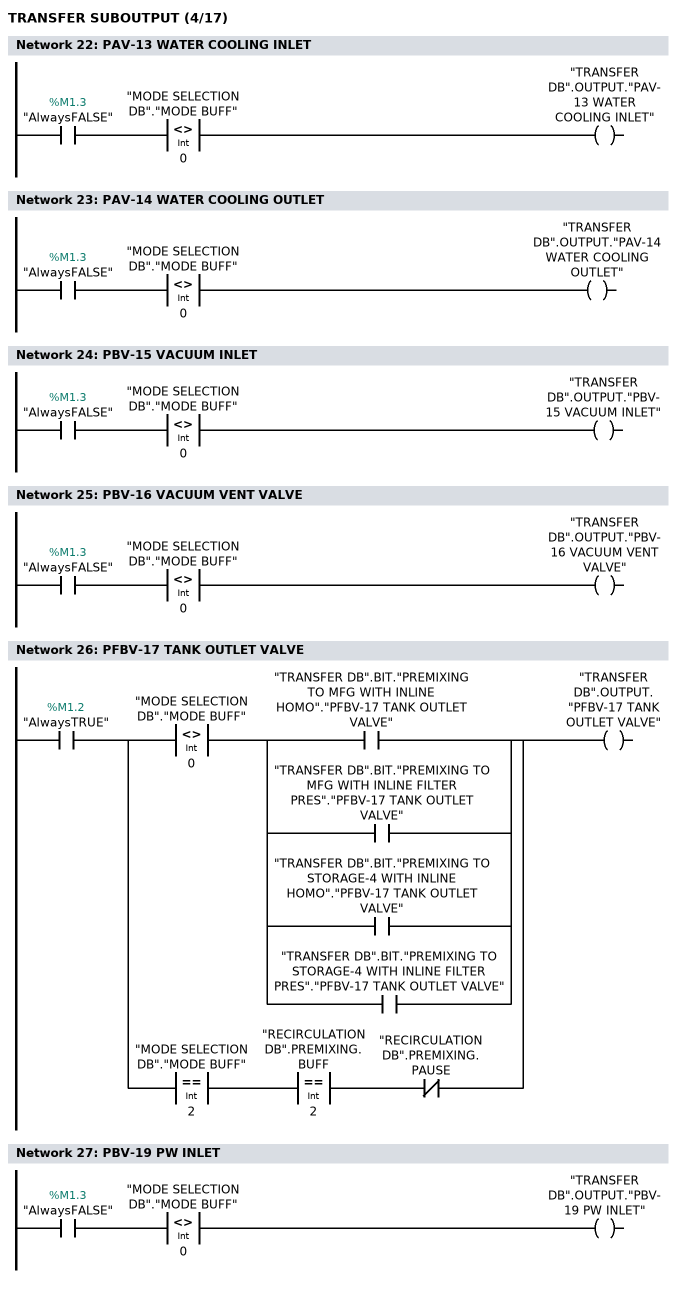
   RUNG wire#powerrail
      Contact( "AlwaysFALSE" )
      { S7_Templates := "SrcType := Int" } NE_Contact(in1 := "MODE SELECTION DB"."MODE BUFF", in2 := 0)
      Coil( "TRANSFER DB".OUTPUT."PAV-13 WATER COOLING INLET" )
   END_RUNG
   // the same network as SCL:
   "TRANSFER DB".OUTPUT."PAV-13 WATER COOLING INLET" := "AlwaysFALSE" AND ("MODE SELECTION DB"."MODE BUFF" <> 0);
END_REGION

REGION Network 23: PAV-14 WATER COOLING OUTLET
   RUNG wire#powerrail
      Contact( "AlwaysFALSE" )
      { S7_Templates := "SrcType := Int" } NE_Contact(in1 := "MODE SELECTION DB"."MODE BUFF", in2 := 0)
      Coil( "TRANSFER DB".OUTPUT."PAV-14 WATER COOLING OUTLET" )
   END_RUNG
   // the same network as SCL:
   "TRANSFER DB".OUTPUT."PAV-14 WATER COOLING OUTLET" := "AlwaysFALSE" AND ("MODE SELECTION DB"."MODE BUFF" <> 0);
END_REGION

REGION Network 24: PBV-15 VACUUM INLET
   RUNG wire#powerrail
      Contact( "AlwaysFALSE" )
      { S7_Templates := "SrcType := Int" } NE_Contact(in1 := "MODE SELECTION DB"."MODE BUFF", in2 := 0)
      Coil( "TRANSFER DB".OUTPUT."PBV-15 VACUUM INLET" )
   END_RUNG
   // the same network as SCL:
   "TRANSFER DB".OUTPUT."PBV-15 VACUUM INLET" := "AlwaysFALSE" AND ("MODE SELECTION DB"."MODE BUFF" <> 0);
END_REGION

REGION Network 25: PBV-16 VACUUM VENT VALVE
   RUNG wire#powerrail
      Contact( "AlwaysFALSE" )
      { S7_Templates := "SrcType := Int" } NE_Contact(in1 := "MODE SELECTION DB"."MODE BUFF", in2 := 0)
      Coil( "TRANSFER DB".OUTPUT."PBV-16 VACUUM VENT VALVE" )
   END_RUNG
   // the same network as SCL:
   "TRANSFER DB".OUTPUT."PBV-16 VACUUM VENT VALVE" := "AlwaysFALSE" AND ("MODE SELECTION DB"."MODE BUFF" <> 0);
END_REGION

REGION Network 26: PFBV-17 TANK OUTLET VALVE
   RUNG wire#powerrail
      Contact( "AlwaysTRUE" )
      wire#w1
      { S7_Templates := "SrcType := Int" } NE_Contact(in1 := "MODE SELECTION DB"."MODE BUFF", in2 := 0)
      wire#w2
      Contact( "TRANSFER DB".BIT."PREMIXING TO MFG WITH INLINE HOMO"."PFBV-17 TANK OUTLET VALVE" )
      wire#w3
      Coil( "TRANSFER DB".OUTPUT."PFBV-17 TANK OUTLET VALVE" )
   END_RUNG
   RUNG wire#w2
      Contact( "TRANSFER DB".BIT."PREMIXING TO MFG WITH INLINE FILTER PRES"."PFBV-17 TANK OUTLET VALVE" )
   END_RUNG wire#w3
   RUNG wire#w2
      Contact( "TRANSFER DB".BIT."PREMIXING TO STORAGE-4 WITH INLINE HOMO"."PFBV-17 TANK OUTLET VALVE" )
   END_RUNG wire#w3
   RUNG wire#w2
      Contact( "TRANSFER DB".BIT."PREMIXING TO STORAGE-4 WITH INLINE FILTER PRES"."PFBV-17 TANK OUTLET VALVE" )
   END_RUNG wire#w3
   RUNG wire#w1
      { S7_Templates := "SrcType := Int" } EQ_Contact(in1 := "MODE SELECTION DB"."MODE BUFF", in2 := 2)
      { S7_Templates := "SrcType := Int" } EQ_Contact(in1 := "RECIRCULATION DB".PREMIXING.BUFF, in2 := 2)
      I_Contact( "RECIRCULATION DB".PREMIXING.PAUSE )
   END_RUNG wire#w3
   // the same network as SCL:
   "TRANSFER DB".OUTPUT."PFBV-17 TANK OUTLET VALVE" := "AlwaysTRUE" AND ((("MODE SELECTION DB"."MODE BUFF" <> 0) AND ("TRANSFER DB".BIT."PREMIXING TO MFG WITH INLINE HOMO"."PFBV-17 TANK OUTLET VALVE" OR "TRANSFER DB".BIT."PREMIXING TO MFG WITH INLINE FILTER PRES"."PFBV-17 TANK OUTLET VALVE" OR "TRANSFER DB".BIT."PREMIXING TO STORAGE-4 WITH INLINE HOMO"."PFBV-17 TANK OUTLET VALVE" OR "TRANSFER DB".BIT."PREMIXING TO STORAGE-4 WITH INLINE FILTER PRES"."PFBV-17 TANK OUTLET VALVE")) OR (("MODE SELECTION DB"."MODE BUFF" = 2) AND ("RECIRCULATION DB".PREMIXING.BUFF = 2) AND NOT "RECIRCULATION DB".PREMIXING.PAUSE));
END_REGION

REGION Network 27: PBV-19 PW INLET
   RUNG wire#powerrail
      Contact( "AlwaysFALSE" )
      { S7_Templates := "SrcType := Int" } NE_Contact(in1 := "MODE SELECTION DB"."MODE BUFF", in2 := 0)
      Coil( "TRANSFER DB".OUTPUT."PBV-19 PW INLET" )
   END_RUNG
   // the same network as SCL:
   "TRANSFER DB".OUTPUT."PBV-19 PW INLET" := "AlwaysFALSE" AND ("MODE SELECTION DB"."MODE BUFF" <> 0);
END_REGION

REGION Network 28: PBV-20 CIP INLET (SPRAY BALL)
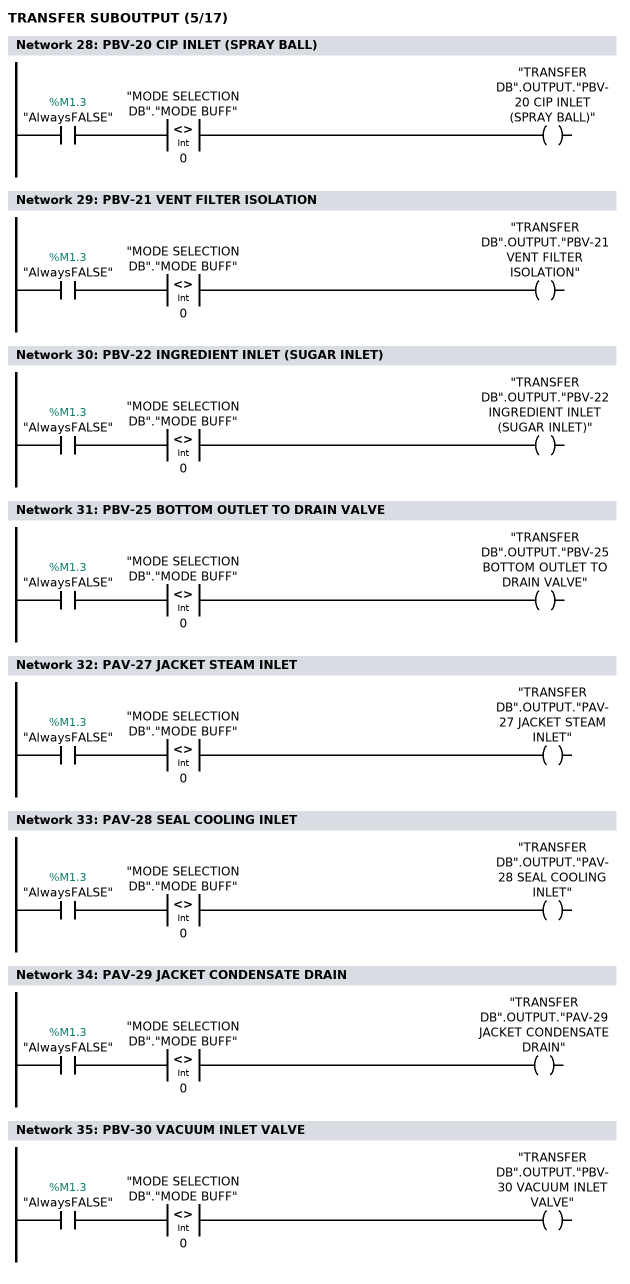
   RUNG wire#powerrail
      Contact( "AlwaysFALSE" )
      { S7_Templates := "SrcType := Int" } NE_Contact(in1 := "MODE SELECTION DB"."MODE BUFF", in2 := 0)
      Coil( "TRANSFER DB".OUTPUT."PBV-20 CIP INLET (SPRAY BALL)" )
   END_RUNG
   // the same network as SCL:
   "TRANSFER DB".OUTPUT."PBV-20 CIP INLET (SPRAY BALL)" := "AlwaysFALSE" AND ("MODE SELECTION DB"."MODE BUFF" <> 0);
END_REGION

REGION Network 29: PBV-21 VENT FILTER ISOLATION
   RUNG wire#powerrail
      Contact( "AlwaysFALSE" )
      { S7_Templates := "SrcType := Int" } NE_Contact(in1 := "MODE SELECTION DB"."MODE BUFF", in2 := 0)
      Coil( "TRANSFER DB".OUTPUT."PBV-21 VENT FILTER ISOLATION" )
   END_RUNG
   // the same network as SCL:
   "TRANSFER DB".OUTPUT."PBV-21 VENT FILTER ISOLATION" := "AlwaysFALSE" AND ("MODE SELECTION DB"."MODE BUFF" <> 0);
END_REGION

REGION Network 30: PBV-22 INGREDIENT INLET (SUGAR INLET)
   RUNG wire#powerrail
      Contact( "AlwaysFALSE" )
      { S7_Templates := "SrcType := Int" } NE_Contact(in1 := "MODE SELECTION DB"."MODE BUFF", in2 := 0)
      Coil( "TRANSFER DB".OUTPUT."PBV-22 INGREDIENT INLET (SUGAR INLET)" )
   END_RUNG
   // the same network as SCL:
   "TRANSFER DB".OUTPUT."PBV-22 INGREDIENT INLET (SUGAR INLET)" := "AlwaysFALSE" AND ("MODE SELECTION DB"."MODE BUFF" <> 0);
END_REGION

REGION Network 31: PBV-25 BOTTOM OUTLET TO DRAIN VALVE
   RUNG wire#powerrail
      Contact( "AlwaysFALSE" )
      { S7_Templates := "SrcType := Int" } NE_Contact(in1 := "MODE SELECTION DB"."MODE BUFF", in2 := 0)
      Coil( "TRANSFER DB".OUTPUT."PBV-25 BOTTOM OUTLET TO DRAIN VALVE" )
   END_RUNG
   // the same network as SCL:
   "TRANSFER DB".OUTPUT."PBV-25 BOTTOM OUTLET TO DRAIN VALVE" := "AlwaysFALSE" AND ("MODE SELECTION DB"."MODE BUFF" <> 0);
END_REGION

REGION Network 32: PAV-27 JACKET STEAM INLET
   RUNG wire#powerrail
      Contact( "AlwaysFALSE" )
      { S7_Templates := "SrcType := Int" } NE_Contact(in1 := "MODE SELECTION DB"."MODE BUFF", in2 := 0)
      Coil( "TRANSFER DB".OUTPUT."PAV-27 JACKET STEAM INLET" )
   END_RUNG
   // the same network as SCL:
   "TRANSFER DB".OUTPUT."PAV-27 JACKET STEAM INLET" := "AlwaysFALSE" AND ("MODE SELECTION DB"."MODE BUFF" <> 0);
END_REGION

REGION Network 33: PAV-28 SEAL COOLING INLET
   RUNG wire#powerrail
      Contact( "AlwaysFALSE" )
      { S7_Templates := "SrcType := Int" } NE_Contact(in1 := "MODE SELECTION DB"."MODE BUFF", in2 := 0)
      Coil( "TRANSFER DB".OUTPUT."PAV-28 SEAL COOLING INLET" )
   END_RUNG
   // the same network as SCL:
   "TRANSFER DB".OUTPUT."PAV-28 SEAL COOLING INLET" := "AlwaysFALSE" AND ("MODE SELECTION DB"."MODE BUFF" <> 0);
END_REGION

REGION Network 34: PAV-29 JACKET CONDENSATE DRAIN
   RUNG wire#powerrail
      Contact( "AlwaysFALSE" )
      { S7_Templates := "SrcType := Int" } NE_Contact(in1 := "MODE SELECTION DB"."MODE BUFF", in2 := 0)
      Coil( "TRANSFER DB".OUTPUT."PAV-29 JACKET CONDENSATE DRAIN" )
   END_RUNG
   // the same network as SCL:
   "TRANSFER DB".OUTPUT."PAV-29 JACKET CONDENSATE DRAIN" := "AlwaysFALSE" AND ("MODE SELECTION DB"."MODE BUFF" <> 0);
END_REGION

REGION Network 35: PBV-30 VACUUM INLET VALVE
   RUNG wire#powerrail
      Contact( "AlwaysFALSE" )
      { S7_Templates := "SrcType := Int" } NE_Contact(in1 := "MODE SELECTION DB"."MODE BUFF", in2 := 0)
      Coil( "TRANSFER DB".OUTPUT."PBV-30 VACUUM INLET VALVE" )
   END_RUNG
   // the same network as SCL:
   "TRANSFER DB".OUTPUT."PBV-30 VACUUM INLET VALVE" := "AlwaysFALSE" AND ("MODE SELECTION DB"."MODE BUFF" <> 0);
END_REGION

REGION Network 36: PBV-31 VACUUM VENT VALVE
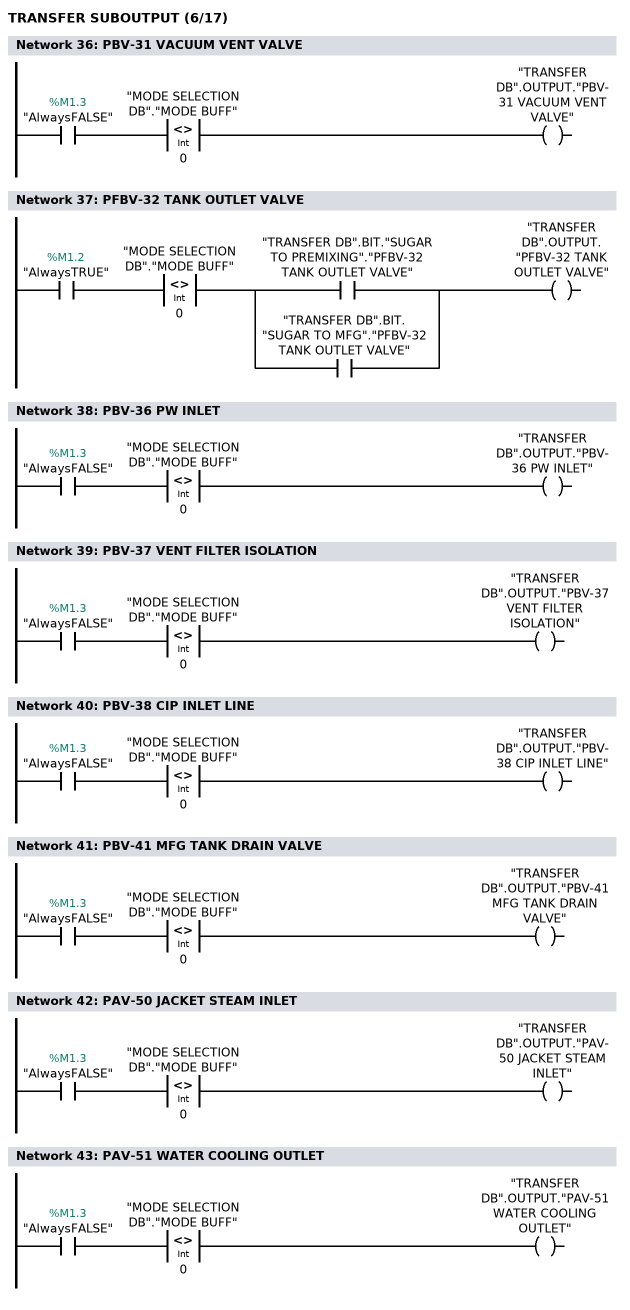
   RUNG wire#powerrail
      Contact( "AlwaysFALSE" )
      { S7_Templates := "SrcType := Int" } NE_Contact(in1 := "MODE SELECTION DB"."MODE BUFF", in2 := 0)
      Coil( "TRANSFER DB".OUTPUT."PBV-31 VACUUM VENT VALVE" )
   END_RUNG
   // the same network as SCL:
   "TRANSFER DB".OUTPUT."PBV-31 VACUUM VENT VALVE" := "AlwaysFALSE" AND ("MODE SELECTION DB"."MODE BUFF" <> 0);
END_REGION

REGION Network 37: PFBV-32 TANK OUTLET VALVE
   RUNG wire#powerrail
      Contact( "AlwaysTRUE" )
      { S7_Templates := "SrcType := Int" } NE_Contact(in1 := "MODE SELECTION DB"."MODE BUFF", in2 := 0)
      wire#w1
      Contact( "TRANSFER DB".BIT."SUGAR TO PREMIXING"."PFBV-32 TANK OUTLET VALVE" )
      wire#w2
      Coil( "TRANSFER DB".OUTPUT."PFBV-32 TANK OUTLET VALVE" )
   END_RUNG
   RUNG wire#w1
      Contact( "TRANSFER DB".BIT."SUGAR TO MFG"."PFBV-32 TANK OUTLET VALVE" )
   END_RUNG wire#w2
   // the same network as SCL:
   "TRANSFER DB".OUTPUT."PFBV-32 TANK OUTLET VALVE" := "AlwaysTRUE" AND ("MODE SELECTION DB"."MODE BUFF" <> 0) AND ("TRANSFER DB".BIT."SUGAR TO PREMIXING"."PFBV-32 TANK OUTLET VALVE" OR "TRANSFER DB".BIT."SUGAR TO MFG"."PFBV-32 TANK OUTLET VALVE");
END_REGION

REGION Network 38: PBV-36 PW INLET
   RUNG wire#powerrail
      Contact( "AlwaysFALSE" )
      { S7_Templates := "SrcType := Int" } NE_Contact(in1 := "MODE SELECTION DB"."MODE BUFF", in2 := 0)
      Coil( "TRANSFER DB".OUTPUT."PBV-36 PW INLET" )
   END_RUNG
   // the same network as SCL:
   "TRANSFER DB".OUTPUT."PBV-36 PW INLET" := "AlwaysFALSE" AND ("MODE SELECTION DB"."MODE BUFF" <> 0);
END_REGION

REGION Network 39: PBV-37 VENT FILTER ISOLATION
   RUNG wire#powerrail
      Contact( "AlwaysFALSE" )
      { S7_Templates := "SrcType := Int" } NE_Contact(in1 := "MODE SELECTION DB"."MODE BUFF", in2 := 0)
      Coil( "TRANSFER DB".OUTPUT."PBV-37 VENT FILTER ISOLATION" )
   END_RUNG
   // the same network as SCL:
   "TRANSFER DB".OUTPUT."PBV-37 VENT FILTER ISOLATION" := "AlwaysFALSE" AND ("MODE SELECTION DB"."MODE BUFF" <> 0);
END_REGION

REGION Network 40: PBV-38 CIP INLET LINE
   RUNG wire#powerrail
      Contact( "AlwaysFALSE" )
      { S7_Templates := "SrcType := Int" } NE_Contact(in1 := "MODE SELECTION DB"."MODE BUFF", in2 := 0)
      Coil( "TRANSFER DB".OUTPUT."PBV-38 CIP INLET LINE" )
   END_RUNG
   // the same network as SCL:
   "TRANSFER DB".OUTPUT."PBV-38 CIP INLET LINE" := "AlwaysFALSE" AND ("MODE SELECTION DB"."MODE BUFF" <> 0);
END_REGION

REGION Network 41: PBV-41 MFG TANK DRAIN VALVE
   RUNG wire#powerrail
      Contact( "AlwaysFALSE" )
      { S7_Templates := "SrcType := Int" } NE_Contact(in1 := "MODE SELECTION DB"."MODE BUFF", in2 := 0)
      Coil( "TRANSFER DB".OUTPUT."PBV-41 MFG TANK DRAIN VALVE" )
   END_RUNG
   // the same network as SCL:
   "TRANSFER DB".OUTPUT."PBV-41 MFG TANK DRAIN VALVE" := "AlwaysFALSE" AND ("MODE SELECTION DB"."MODE BUFF" <> 0);
END_REGION

REGION Network 42: PAV-50 JACKET STEAM INLET
   RUNG wire#powerrail
      Contact( "AlwaysFALSE" )
      { S7_Templates := "SrcType := Int" } NE_Contact(in1 := "MODE SELECTION DB"."MODE BUFF", in2 := 0)
      Coil( "TRANSFER DB".OUTPUT."PAV-50 JACKET STEAM INLET" )
   END_RUNG
   // the same network as SCL:
   "TRANSFER DB".OUTPUT."PAV-50 JACKET STEAM INLET" := "AlwaysFALSE" AND ("MODE SELECTION DB"."MODE BUFF" <> 0);
END_REGION

REGION Network 43: PAV-51 WATER COOLING OUTLET
   RUNG wire#powerrail
      Contact( "AlwaysFALSE" )
      { S7_Templates := "SrcType := Int" } NE_Contact(in1 := "MODE SELECTION DB"."MODE BUFF", in2 := 0)
      Coil( "TRANSFER DB".OUTPUT."PAV-51 WATER COOLING OUTLET" )
   END_RUNG
   // the same network as SCL:
   "TRANSFER DB".OUTPUT."PAV-51 WATER COOLING OUTLET" := "AlwaysFALSE" AND ("MODE SELECTION DB"."MODE BUFF" <> 0);
END_REGION

REGION Network 44: PAV-52 WATER COOLING INLET
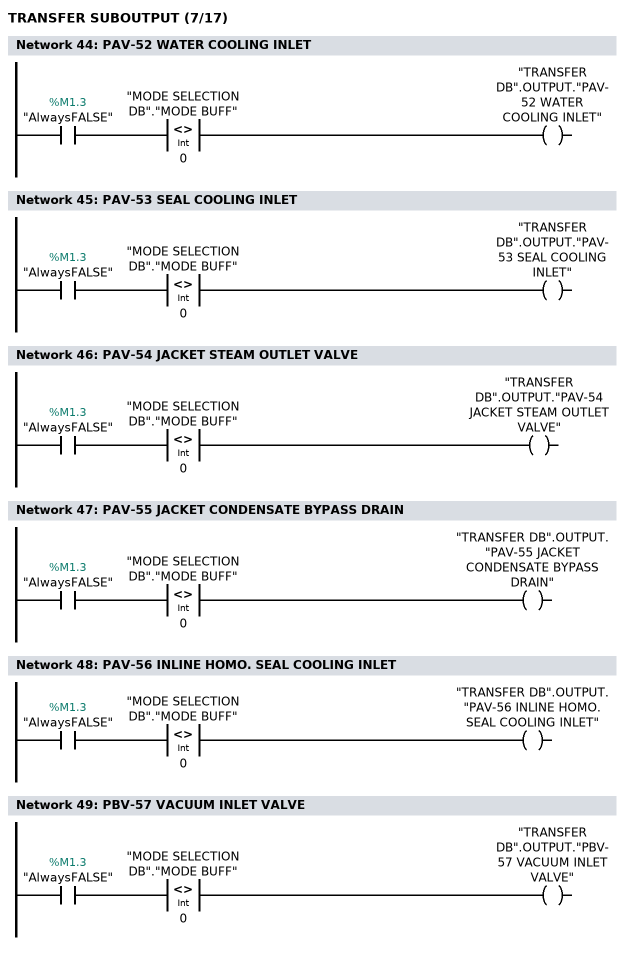
   RUNG wire#powerrail
      Contact( "AlwaysFALSE" )
      { S7_Templates := "SrcType := Int" } NE_Contact(in1 := "MODE SELECTION DB"."MODE BUFF", in2 := 0)
      Coil( "TRANSFER DB".OUTPUT."PAV-52 WATER COOLING INLET" )
   END_RUNG
   // the same network as SCL:
   "TRANSFER DB".OUTPUT."PAV-52 WATER COOLING INLET" := "AlwaysFALSE" AND ("MODE SELECTION DB"."MODE BUFF" <> 0);
END_REGION

REGION Network 45: PAV-53 SEAL COOLING INLET
   RUNG wire#powerrail
      Contact( "AlwaysFALSE" )
      { S7_Templates := "SrcType := Int" } NE_Contact(in1 := "MODE SELECTION DB"."MODE BUFF", in2 := 0)
      Coil( "TRANSFER DB".OUTPUT."PAV-53 SEAL COOLING INLET" )
   END_RUNG
   // the same network as SCL:
   "TRANSFER DB".OUTPUT."PAV-53 SEAL COOLING INLET" := "AlwaysFALSE" AND ("MODE SELECTION DB"."MODE BUFF" <> 0);
END_REGION

REGION Network 46: PAV-54 JACKET STEAM OUTLET VALVE
   RUNG wire#powerrail
      Contact( "AlwaysFALSE" )
      { S7_Templates := "SrcType := Int" } NE_Contact(in1 := "MODE SELECTION DB"."MODE BUFF", in2 := 0)
      Coil( "TRANSFER DB".OUTPUT."PAV-54 JACKET STEAM OUTLET VALVE" )
   END_RUNG
   // the same network as SCL:
   "TRANSFER DB".OUTPUT."PAV-54 JACKET STEAM OUTLET VALVE" := "AlwaysFALSE" AND ("MODE SELECTION DB"."MODE BUFF" <> 0);
END_REGION

REGION Network 47: PAV-55 JACKET CONDENSATE BYPASS DRAIN
   RUNG wire#powerrail
      Contact( "AlwaysFALSE" )
      { S7_Templates := "SrcType := Int" } NE_Contact(in1 := "MODE SELECTION DB"."MODE BUFF", in2 := 0)
      Coil( "TRANSFER DB".OUTPUT."PAV-55 JACKET CONDENSATE BYPASS DRAIN" )
   END_RUNG
   // the same network as SCL:
   "TRANSFER DB".OUTPUT."PAV-55 JACKET CONDENSATE BYPASS DRAIN" := "AlwaysFALSE" AND ("MODE SELECTION DB"."MODE BUFF" <> 0);
END_REGION

REGION Network 48: PAV-56 INLINE HOMO. SEAL COOLING INLET
   RUNG wire#powerrail
      Contact( "AlwaysFALSE" )
      { S7_Templates := "SrcType := Int" } NE_Contact(in1 := "MODE SELECTION DB"."MODE BUFF", in2 := 0)
      Coil( "TRANSFER DB".OUTPUT."PAV-56 INLINE HOMO. SEAL COOLING INLET" )
   END_RUNG
   // the same network as SCL:
   "TRANSFER DB".OUTPUT."PAV-56 INLINE HOMO. SEAL COOLING INLET" := "AlwaysFALSE" AND ("MODE SELECTION DB"."MODE BUFF" <> 0);
END_REGION

REGION Network 49: PBV-57 VACUUM INLET VALVE
   RUNG wire#powerrail
      Contact( "AlwaysFALSE" )
      { S7_Templates := "SrcType := Int" } NE_Contact(in1 := "MODE SELECTION DB"."MODE BUFF", in2 := 0)
      Coil( "TRANSFER DB".OUTPUT."PBV-57 VACUUM INLET VALVE" )
   END_RUNG
   // the same network as SCL:
   "TRANSFER DB".OUTPUT."PBV-57 VACUUM INLET VALVE" := "AlwaysFALSE" AND ("MODE SELECTION DB"."MODE BUFF" <> 0);
END_REGION

REGION Network 50: PFBV-59 TANK OUTLET VALVE
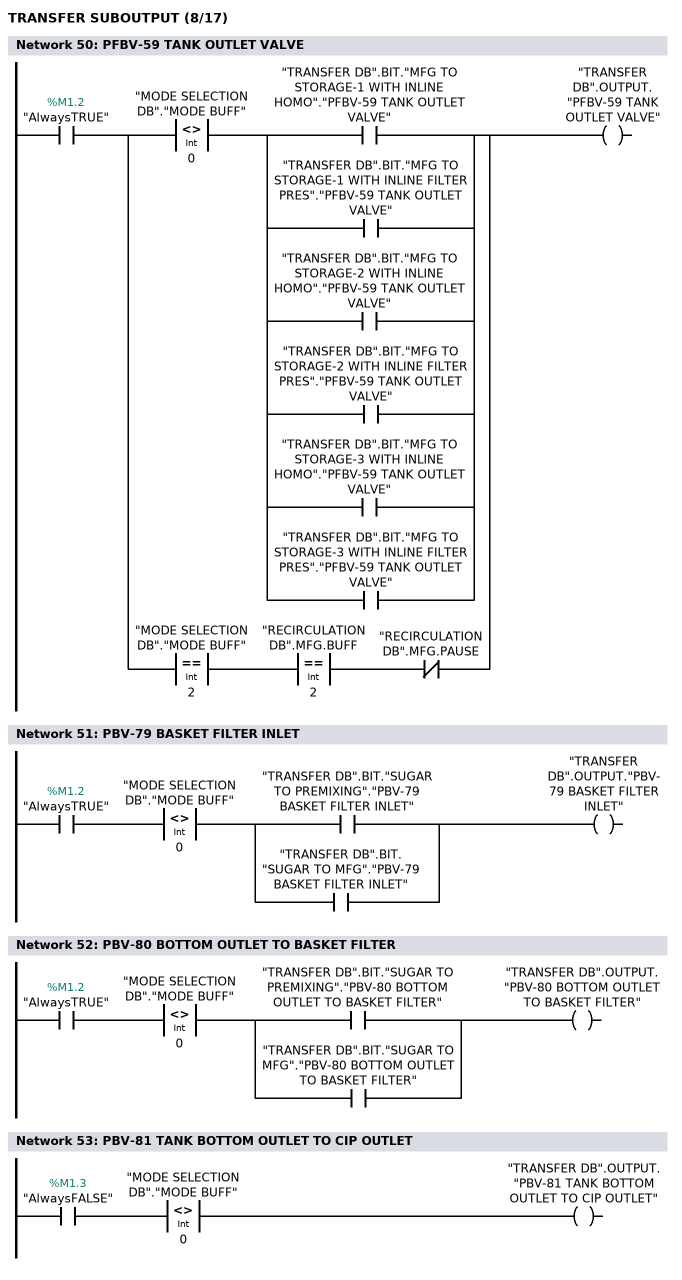
   RUNG wire#powerrail
      Contact( "AlwaysTRUE" )
      wire#w1
      { S7_Templates := "SrcType := Int" } NE_Contact(in1 := "MODE SELECTION DB"."MODE BUFF", in2 := 0)
      wire#w2
      Contact( "TRANSFER DB".BIT."MFG TO STORAGE-1 WITH INLINE HOMO"."PFBV-59 TANK OUTLET VALVE" )
      wire#w3
      Coil( "TRANSFER DB".OUTPUT."PFBV-59 TANK OUTLET VALVE" )
   END_RUNG
   RUNG wire#w2
      Contact( "TRANSFER DB".BIT."MFG TO STORAGE-1 WITH INLINE FILTER PRES"."PFBV-59 TANK OUTLET VALVE" )
   END_RUNG wire#w3
   RUNG wire#w2
      Contact( "TRANSFER DB".BIT."MFG TO STORAGE-2 WITH INLINE HOMO"."PFBV-59 TANK OUTLET VALVE" )
   END_RUNG wire#w3
   RUNG wire#w2
      Contact( "TRANSFER DB".BIT."MFG TO STORAGE-2 WITH INLINE FILTER PRES"."PFBV-59 TANK OUTLET VALVE" )
   END_RUNG wire#w3
   RUNG wire#w2
      Contact( "TRANSFER DB".BIT."MFG TO STORAGE-3 WITH INLINE HOMO"."PFBV-59 TANK OUTLET VALVE" )
   END_RUNG wire#w3
   RUNG wire#w2
      Contact( "TRANSFER DB".BIT."MFG TO STORAGE-3 WITH INLINE FILTER PRES"."PFBV-59 TANK OUTLET VALVE" )
   END_RUNG wire#w3
   RUNG wire#w1
      { S7_Templates := "SrcType := Int" } EQ_Contact(in1 := "MODE SELECTION DB"."MODE BUFF", in2 := 2)
      { S7_Templates := "SrcType := Int" } EQ_Contact(in1 := "RECIRCULATION DB".MFG.BUFF, in2 := 2)
      I_Contact( "RECIRCULATION DB".MFG.PAUSE )
   END_RUNG wire#w3
   // the same network as SCL:
   "TRANSFER DB".OUTPUT."PFBV-59 TANK OUTLET VALVE" := "AlwaysTRUE" AND ((("MODE SELECTION DB"."MODE BUFF" <> 0) AND ("TRANSFER DB".BIT."MFG TO STORAGE-1 WITH INLINE HOMO"."PFBV-59 TANK OUTLET VALVE" OR "TRANSFER DB".BIT."MFG TO STORAGE-1 WITH INLINE FILTER PRES"."PFBV-59 TANK OUTLET VALVE" OR "TRANSFER DB".BIT."MFG TO STORAGE-2 WITH INLINE HOMO"."PFBV-59 TANK OUTLET VALVE" OR "TRANSFER DB".BIT."MFG TO STORAGE-2 WITH INLINE FILTER PRES"."PFBV-59 TANK OUTLET VALVE" OR "TRANSFER DB".BIT."MFG TO STORAGE-3 WITH INLINE HOMO"."PFBV-59 TANK OUTLET VALVE" OR "TRANSFER DB".BIT."MFG TO STORAGE-3 WITH INLINE FILTER PRES"."PFBV-59 TANK OUTLET VALVE")) OR (("MODE SELECTION DB"."MODE BUFF" = 2) AND ("RECIRCULATION DB".MFG.BUFF = 2) AND NOT "RECIRCULATION DB".MFG.PAUSE));
END_REGION

REGION Network 51: PBV-79 BASKET FILTER INLET
   RUNG wire#powerrail
      Contact( "AlwaysTRUE" )
      { S7_Templates := "SrcType := Int" } NE_Contact(in1 := "MODE SELECTION DB"."MODE BUFF", in2 := 0)
      wire#w1
      Contact( "TRANSFER DB".BIT."SUGAR TO PREMIXING"."PBV-79 BASKET FILTER INLET" )
      wire#w2
      Coil( "TRANSFER DB".OUTPUT."PBV-79 BASKET FILTER INLET" )
   END_RUNG
   RUNG wire#w1
      Contact( "TRANSFER DB".BIT."SUGAR TO MFG"."PBV-79 BASKET FILTER INLET" )
   END_RUNG wire#w2
   // the same network as SCL:
   "TRANSFER DB".OUTPUT."PBV-79 BASKET FILTER INLET" := "AlwaysTRUE" AND ("MODE SELECTION DB"."MODE BUFF" <> 0) AND ("TRANSFER DB".BIT."SUGAR TO PREMIXING"."PBV-79 BASKET FILTER INLET" OR "TRANSFER DB".BIT."SUGAR TO MFG"."PBV-79 BASKET FILTER INLET");
END_REGION

REGION Network 52: PBV-80 BOTTOM OUTLET TO BASKET FILTER
   RUNG wire#powerrail
      Contact( "AlwaysTRUE" )
      { S7_Templates := "SrcType := Int" } NE_Contact(in1 := "MODE SELECTION DB"."MODE BUFF", in2 := 0)
      wire#w1
      Contact( "TRANSFER DB".BIT."SUGAR TO PREMIXING"."PBV-80 BOTTOM OUTLET TO BASKET FILTER" )
      wire#w2
      Coil( "TRANSFER DB".OUTPUT."PBV-80 BOTTOM OUTLET TO BASKET FILTER" )
   END_RUNG
   RUNG wire#w1
      Contact( "TRANSFER DB".BIT."SUGAR TO MFG"."PBV-80 BOTTOM OUTLET TO BASKET FILTER" )
   END_RUNG wire#w2
   // the same network as SCL:
   "TRANSFER DB".OUTPUT."PBV-80 BOTTOM OUTLET TO BASKET FILTER" := "AlwaysTRUE" AND ("MODE SELECTION DB"."MODE BUFF" <> 0) AND ("TRANSFER DB".BIT."SUGAR TO PREMIXING"."PBV-80 BOTTOM OUTLET TO BASKET FILTER" OR "TRANSFER DB".BIT."SUGAR TO MFG"."PBV-80 BOTTOM OUTLET TO BASKET FILTER");
END_REGION

REGION Network 53: PBV-81 TANK BOTTOM OUTLET TO CIP OUTLET
   RUNG wire#powerrail
      Contact( "AlwaysFALSE" )
      { S7_Templates := "SrcType := Int" } NE_Contact(in1 := "MODE SELECTION DB"."MODE BUFF", in2 := 0)
      Coil( "TRANSFER DB".OUTPUT."PBV-81 TANK BOTTOM OUTLET TO CIP OUTLET" )
   END_RUNG
   // the same network as SCL:
   "TRANSFER DB".OUTPUT."PBV-81 TANK BOTTOM OUTLET TO CIP OUTLET" := "AlwaysFALSE" AND ("MODE SELECTION DB"."MODE BUFF" <> 0);
END_REGION

